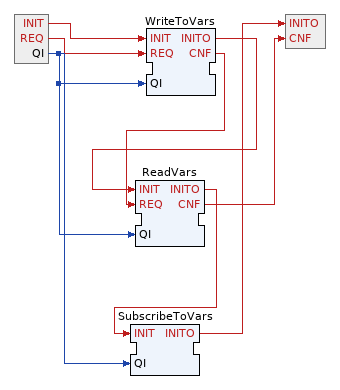
      [picture p47: application OpcUaBothWorking.bytestringNodeIdTestRemote]
      SUBAPPLICATION WriteToVars
        EVENT_INPUT
          INIT;
          REQ;
        END_EVENT
        EVENT_OUTPUT
          INITO;
          CNF;
        END_EVENT
        VAR_INPUT
          QI : BOOL;
        END_VAR
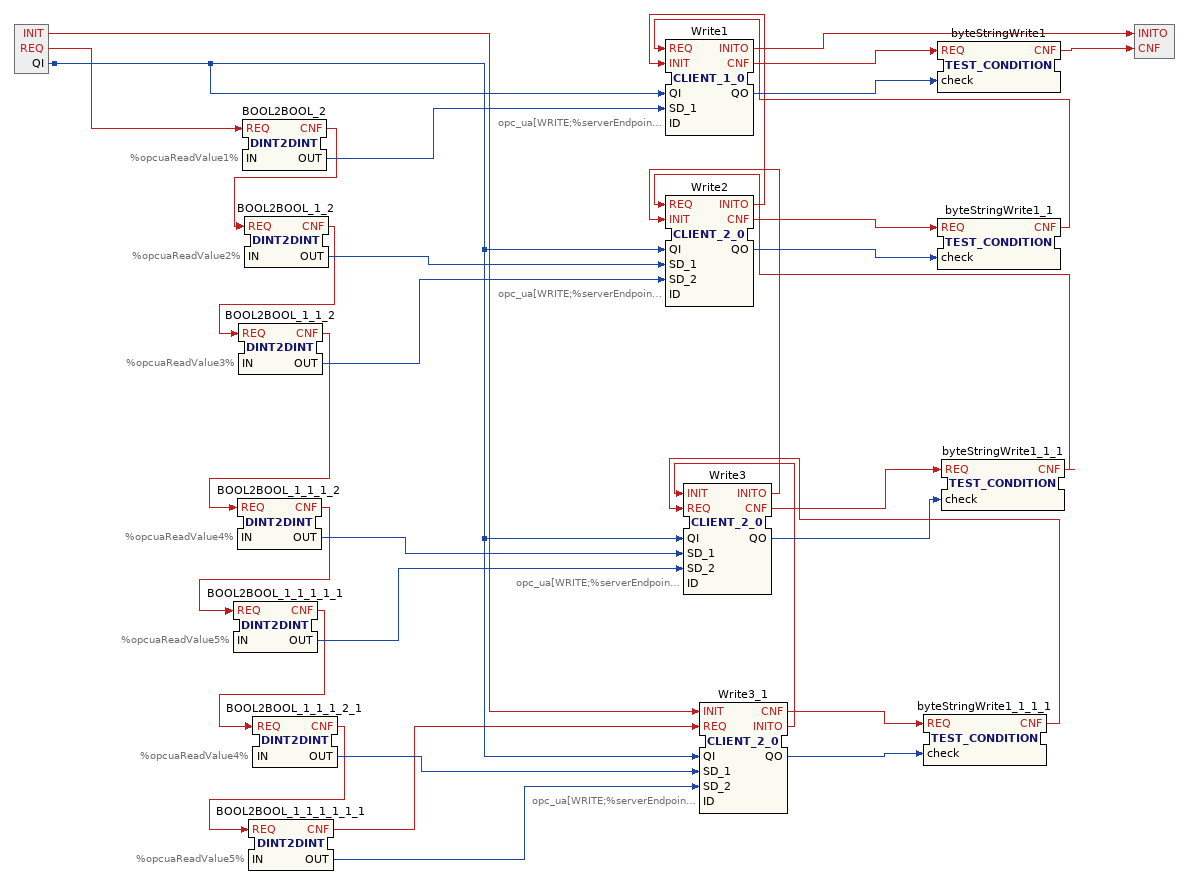
        FBS
          BOOL2BOOL_1_1_2 : DINT2DINT(IN := %opcuaReadValue3%);
          BOOL2BOOL_1_1_1_1_1 : DINT2DINT(IN := %opcuaReadValue5%);
          BOOL2BOOL_1_1_1_2 : DINT2DINT(IN := %opcuaReadValue4%);
          BOOL2BOOL_2 : DINT2DINT(IN := %opcuaReadValue1%);
          BOOL2BOOL_1_2 : DINT2DINT(IN := %opcuaReadValue2%);
          BOOL2BOOL_1_1_1_1_1_1 : DINT2DINT(IN := %opcuaReadValue5%);
          BOOL2BOOL_1_1_1_2_1 : DINT2DINT(IN := %opcuaReadValue4%);
          byteStringWrite1 : TEST_CONDITION;
          byteStringWrite1_1 : TEST_CONDITION;
          byteStringWrite1_1_1 : TEST_CONDITION;
          byteStringWrite1_1_1_1 : TEST_CONDITION;
          Write1 : CLIENT_1_0(ID := opc_ua[WRITE;%serverEndpoint%;%opcuaFolderTestWithNodeIdByteString1%]);
          Write2 : CLIENT_2_0(ID := opc_ua[WRITE;%serverEndpoint%;%opcuaFolderTestWithNodeIdByteString2%]);
          Write3_1 : CLIENT_2_0(ID := opc_ua[WRITE;%serverEndpoint%;,1:b=byteStringNodeId3;,1:b=byteStringNodeId4]);
          Write3 : CLIENT_2_0(ID := opc_ua[WRITE;%serverEndpoint%;%opcuaFolderTestWithNodeIdByteString3%]);
        END_FBS
        EVENT_CONNECTIONS
          BOOL2BOOL_1_2.CNF TO BOOL2BOOL_1_1_2.REQ;
          BOOL2BOOL_1_1_2.CNF TO BOOL2BOOL_1_1_1_2.REQ;
          BOOL2BOOL_1_1_1_2.CNF TO BOOL2BOOL_1_1_1_1_1.REQ;
          BOOL2BOOL_2.CNF TO BOOL2BOOL_1_2.REQ;
          REQ TO BOOL2BOOL_2.REQ;
          BOOL2BOOL_1_1_1_2_1.CNF TO BOOL2BOOL_1_1_1_1_1_1.REQ;
          BOOL2BOOL_1_1_1_1_1.CNF TO BOOL2BOOL_1_1_1_2_1.REQ;
          byteStringWrite1.CNF TO CNF;
          byteStringWrite1_1.CNF TO Write1.REQ;
          Write1.INITO TO INITO;
          Write1.CNF TO byteStringWrite1.REQ;
          byteStringWrite1_1_1.CNF TO Write2.REQ;
          Write2.INITO TO Write1.INIT;
          Write2.CNF TO byteStringWrite1_1.REQ;
          INIT TO Write3_1.INIT;
          BOOL2BOOL_1_1_1_1_1_1.CNF TO Write3_1.REQ;
          Write3_1.CNF TO byteStringWrite1_1_1_1.REQ;
          Write3_1.INITO TO Write3.INIT;
          byteStringWrite1_1_1_1.CNF TO Write3.REQ;
          Write3.INITO TO Write2.INIT;
          Write3.CNF TO byteStringWrite1_1_1.REQ;
        END_CONNECTIONS
        DATA_CONNECTIONS
          QI TO Write1.QI;
          BOOL2BOOL_2.OUT TO Write1.SD_1;
          Write1.QO TO byteStringWrite1.check;
          QI TO Write2.QI;
          BOOL2BOOL_1_2.OUT TO Write2.SD_1;
          BOOL2BOOL_1_1_2.OUT TO Write2.SD_2;
          Write2.QO TO byteStringWrite1_1.check;
          QI TO Write3_1.QI;
          BOOL2BOOL_1_1_1_2_1.OUT TO Write3_1.SD_1;
          BOOL2BOOL_1_1_1_1_1_1.OUT TO Write3_1.SD_2;
          Write3_1.QO TO byteStringWrite1_1_1_1.check;
          QI TO Write3.QI;
          BOOL2BOOL_1_1_1_2.OUT TO Write3.SD_1;
          BOOL2BOOL_1_1_1_1_1.OUT TO Write3.SD_2;
          Write3.QO TO byteStringWrite1_1_1.check;
        END_CONNECTIONS
      END_SUBAPPLICATION
      SUBAPPLICATION ReadVars
        EVENT_INPUT
          INIT;
          REQ;
        END_EVENT
        EVENT_OUTPUT
          INITO;
          CNF;
        END_EVENT
        VAR_INPUT
          QI : BOOL;
        END_VAR
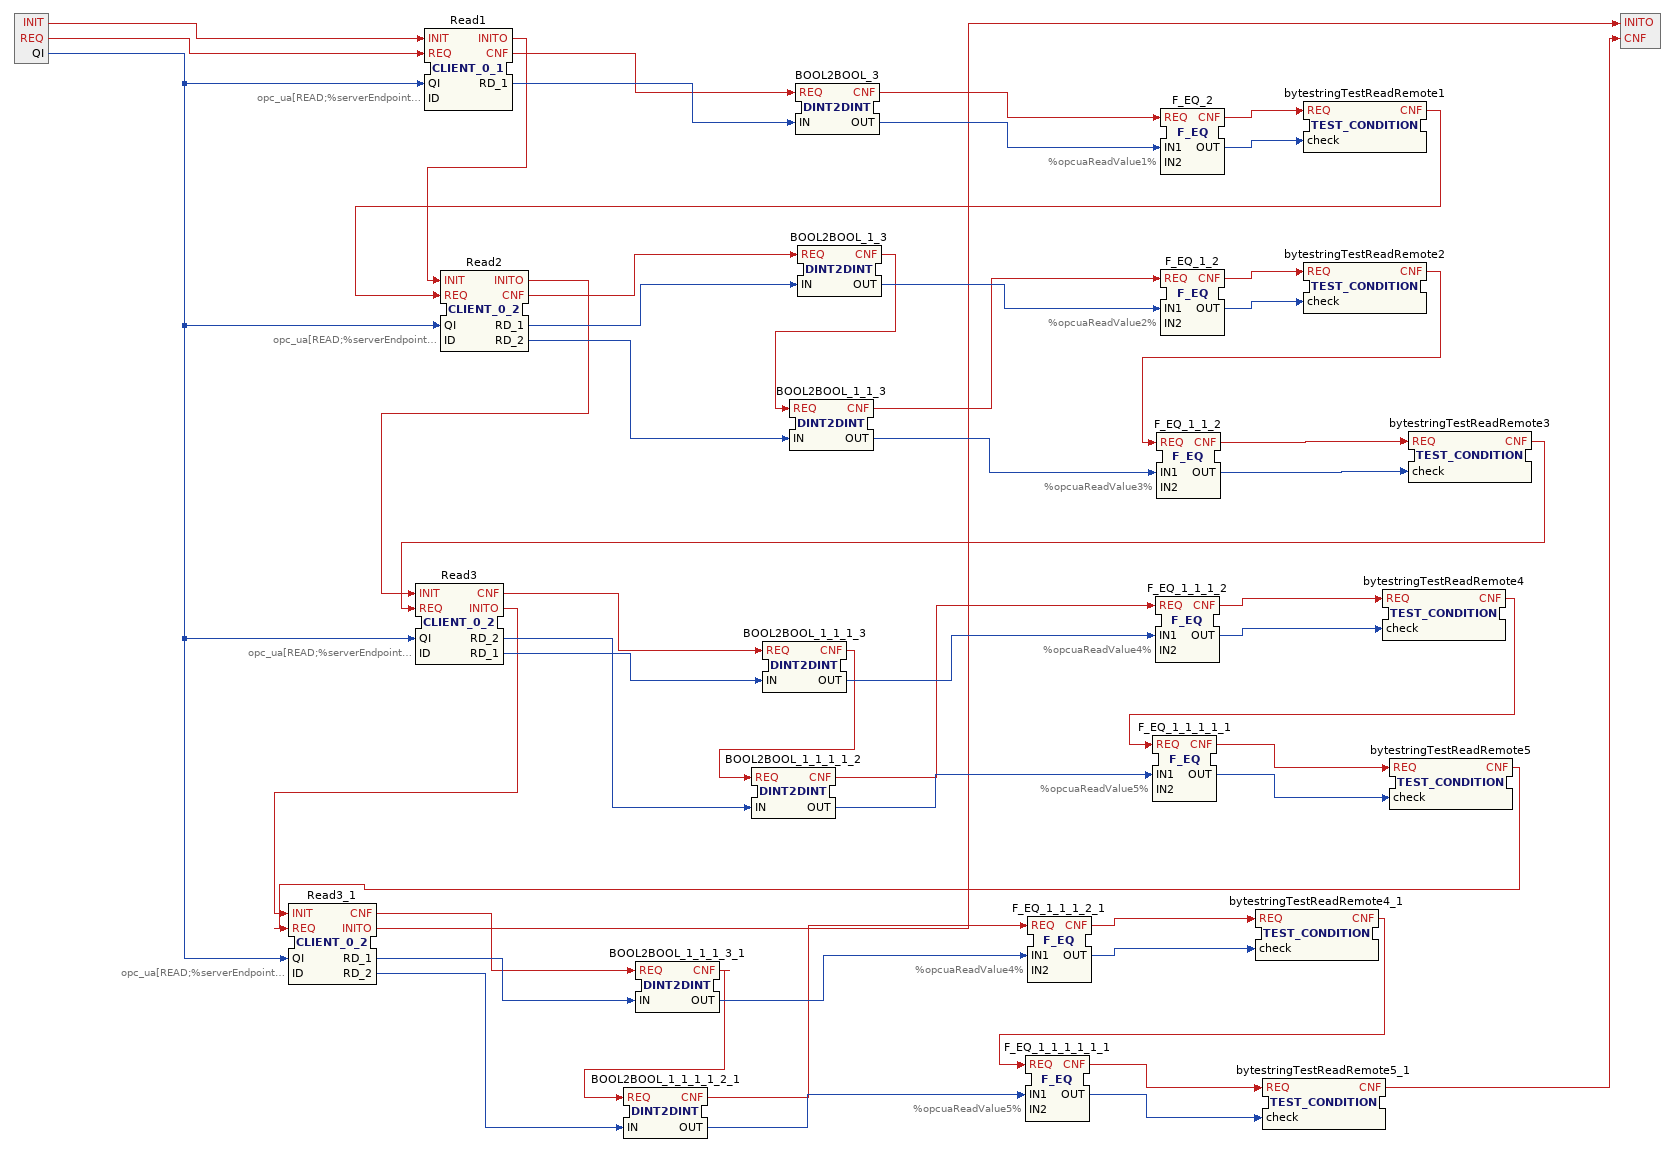
        FBS
          Read1 : CLIENT_0_1(ID := opc_ua[READ;%serverEndpoint%;%opcuaFolderTestWithNodeIdByteString1%]);
          Read2 : CLIENT_0_2(ID := opc_ua[READ;%serverEndpoint%;%opcuaFolderTestWithNodeIdByteString2%]);
          F_EQ_1_1_1_2 : F_EQ(IN2 := %opcuaReadValue4%);
          bytestringTestReadRemote4 : TEST_CONDITION;
          BOOL2BOOL_1_3 : DINT2DINT;
          F_EQ_1_1_1_1_1 : F_EQ(IN2 := %opcuaReadValue5%);
          bytestringTestReadRemote3 : TEST_CONDITION;
          BOOL2BOOL_1_1_3 : DINT2DINT;
          BOOL2BOOL_1_1_1_1_2 : DINT2DINT;
          BOOL2BOOL_1_1_1_3 : DINT2DINT;
          bytestringTestReadRemote2 : TEST_CONDITION;
          F_EQ_1_1_2 : F_EQ(IN2 := %opcuaReadValue3%);
          F_EQ_2 : F_EQ(IN2 := %opcuaReadValue1%);
          F_EQ_1_2 : F_EQ(IN2 := %opcuaReadValue2%);
          Read3 : CLIENT_0_2(ID := opc_ua[READ;%serverEndpoint%;%opcuaFolderTestWithNodeIdByteString3%]);
          bytestringTestReadRemote5 : TEST_CONDITION;
          bytestringTestReadRemote1 : TEST_CONDITION;
          BOOL2BOOL_3 : DINT2DINT;
          BOOL2BOOL_1_1_1_3_1 : DINT2DINT;
          Read3_1 : CLIENT_0_2(ID := opc_ua[READ;%serverEndpoint%;,1:b=byteStringNodeId3;,1:b=byteStringNodeId4]);
          bytestringTestReadRemote4_1 : TEST_CONDITION;
          F_EQ_1_1_1_2_1 : F_EQ(IN2 := %opcuaReadValue4%);
          BOOL2BOOL_1_1_1_1_2_1 : DINT2DINT;
          bytestringTestReadRemote5_1 : TEST_CONDITION;
          F_EQ_1_1_1_1_1_1 : F_EQ(IN2 := %opcuaReadValue5%);
        END_FBS
        EVENT_CONNECTIONS
          Read1.INITO TO Read2.INIT;
          Read1.CNF TO BOOL2BOOL_3.REQ;
          bytestringTestReadRemote1.CNF TO Read2.REQ;
          Read2.INITO TO Read3.INIT;
          Read2.CNF TO BOOL2BOOL_1_3.REQ;
          BOOL2BOOL_1_1_1_1_2.CNF TO F_EQ_1_1_1_2.REQ;
          F_EQ_1_1_1_2.CNF TO bytestringTestReadRemote4.REQ;
          bytestringTestReadRemote4.CNF TO F_EQ_1_1_1_1_1.REQ;
          BOOL2BOOL_1_3.CNF TO BOOL2BOOL_1_1_3.REQ;
          F_EQ_1_1_1_1_1.CNF TO bytestringTestReadRemote5.REQ;
          F_EQ_1_1_2.CNF TO bytestringTestReadRemote3.REQ;
          bytestringTestReadRemote3.CNF TO Read3.REQ;
          BOOL2BOOL_1_1_3.CNF TO F_EQ_1_2.REQ;
          BOOL2BOOL_1_1_1_3.CNF TO BOOL2BOOL_1_1_1_1_2.REQ;
          Read3.CNF TO BOOL2BOOL_1_1_1_3.REQ;
          F_EQ_1_2.CNF TO bytestringTestReadRemote2.REQ;
          bytestringTestReadRemote2.CNF TO F_EQ_1_1_2.REQ;
          BOOL2BOOL_3.CNF TO F_EQ_2.REQ;
          F_EQ_2.CNF TO bytestringTestReadRemote1.REQ;
          INIT TO Read1.INIT;
          REQ TO Read1.REQ;
          bytestringTestReadRemote4_1.CNF TO F_EQ_1_1_1_1_1_1.REQ;
          BOOL2BOOL_1_1_1_1_2_1.CNF TO F_EQ_1_1_1_2_1.REQ;
          F_EQ_1_1_1_1_1_1.CNF TO bytestringTestReadRemote5_1.REQ;
          F_EQ_1_1_1_2_1.CNF TO bytestringTestReadRemote4_1.REQ;
          BOOL2BOOL_1_1_1_3_1.CNF TO BOOL2BOOL_1_1_1_1_2_1.REQ;
          Read3_1.CNF TO BOOL2BOOL_1_1_1_3_1.REQ;
          Read3_1.INITO TO INITO;
          Read3.INITO TO Read3_1.INIT;
          bytestringTestReadRemote5_1.CNF TO CNF;
          bytestringTestReadRemote5.CNF TO Read3_1.REQ;
        END_CONNECTIONS
        DATA_CONNECTIONS
          Read1.RD_1 TO BOOL2BOOL_3.IN;
          Read2.RD_1 TO BOOL2BOOL_1_3.IN;
          Read2.RD_2 TO BOOL2BOOL_1_1_3.IN;
          BOOL2BOOL_1_1_1_3.OUT TO F_EQ_1_1_1_2.IN1;
          F_EQ_1_1_1_2.OUT TO bytestringTestReadRemote4.check;
          BOOL2BOOL_1_3.OUT TO F_EQ_1_2.IN1;
          BOOL2BOOL_1_1_1_1_2.OUT TO F_EQ_1_1_1_1_1.IN1;
          F_EQ_1_1_1_1_1.OUT TO bytestringTestReadRemote5.check;
          F_EQ_1_1_2.OUT TO bytestringTestReadRemote3.check;
          BOOL2BOOL_1_1_3.OUT TO F_EQ_1_1_2.IN1;
          Read3.RD_2 TO BOOL2BOOL_1_1_1_1_2.IN;
          Read3.RD_1 TO BOOL2BOOL_1_1_1_3.IN;
          F_EQ_1_2.OUT TO bytestringTestReadRemote2.check;
          BOOL2BOOL_3.OUT TO F_EQ_2.IN1;
          F_EQ_2.OUT TO bytestringTestReadRemote1.check;
          QI TO Read1.QI;
          QI TO Read2.QI;
          QI TO Read3.QI;
          BOOL2BOOL_1_1_1_1_2_1.OUT TO F_EQ_1_1_1_1_1_1.IN1;
          BOOL2BOOL_1_1_1_3_1.OUT TO F_EQ_1_1_1_2_1.IN1;
          F_EQ_1_1_1_2_1.OUT TO bytestringTestReadRemote4_1.check;
          Read3_1.RD_1 TO BOOL2BOOL_1_1_1_3_1.IN;
          F_EQ_1_1_1_1_1_1.OUT TO bytestringTestReadRemote5_1.check;
          Read3_1.RD_2 TO BOOL2BOOL_1_1_1_1_2_1.IN;
          QI TO Read3_1.QI;
        END_CONNECTIONS
      END_SUBAPPLICATION
      SUBAPPLICATION SubscribeToVars
        EVENT_INPUT
          INIT;
        END_EVENT
        EVENT_OUTPUT
          INITO;
        END_EVENT
        VAR_INPUT
          QI : BOOL;
        END_VAR
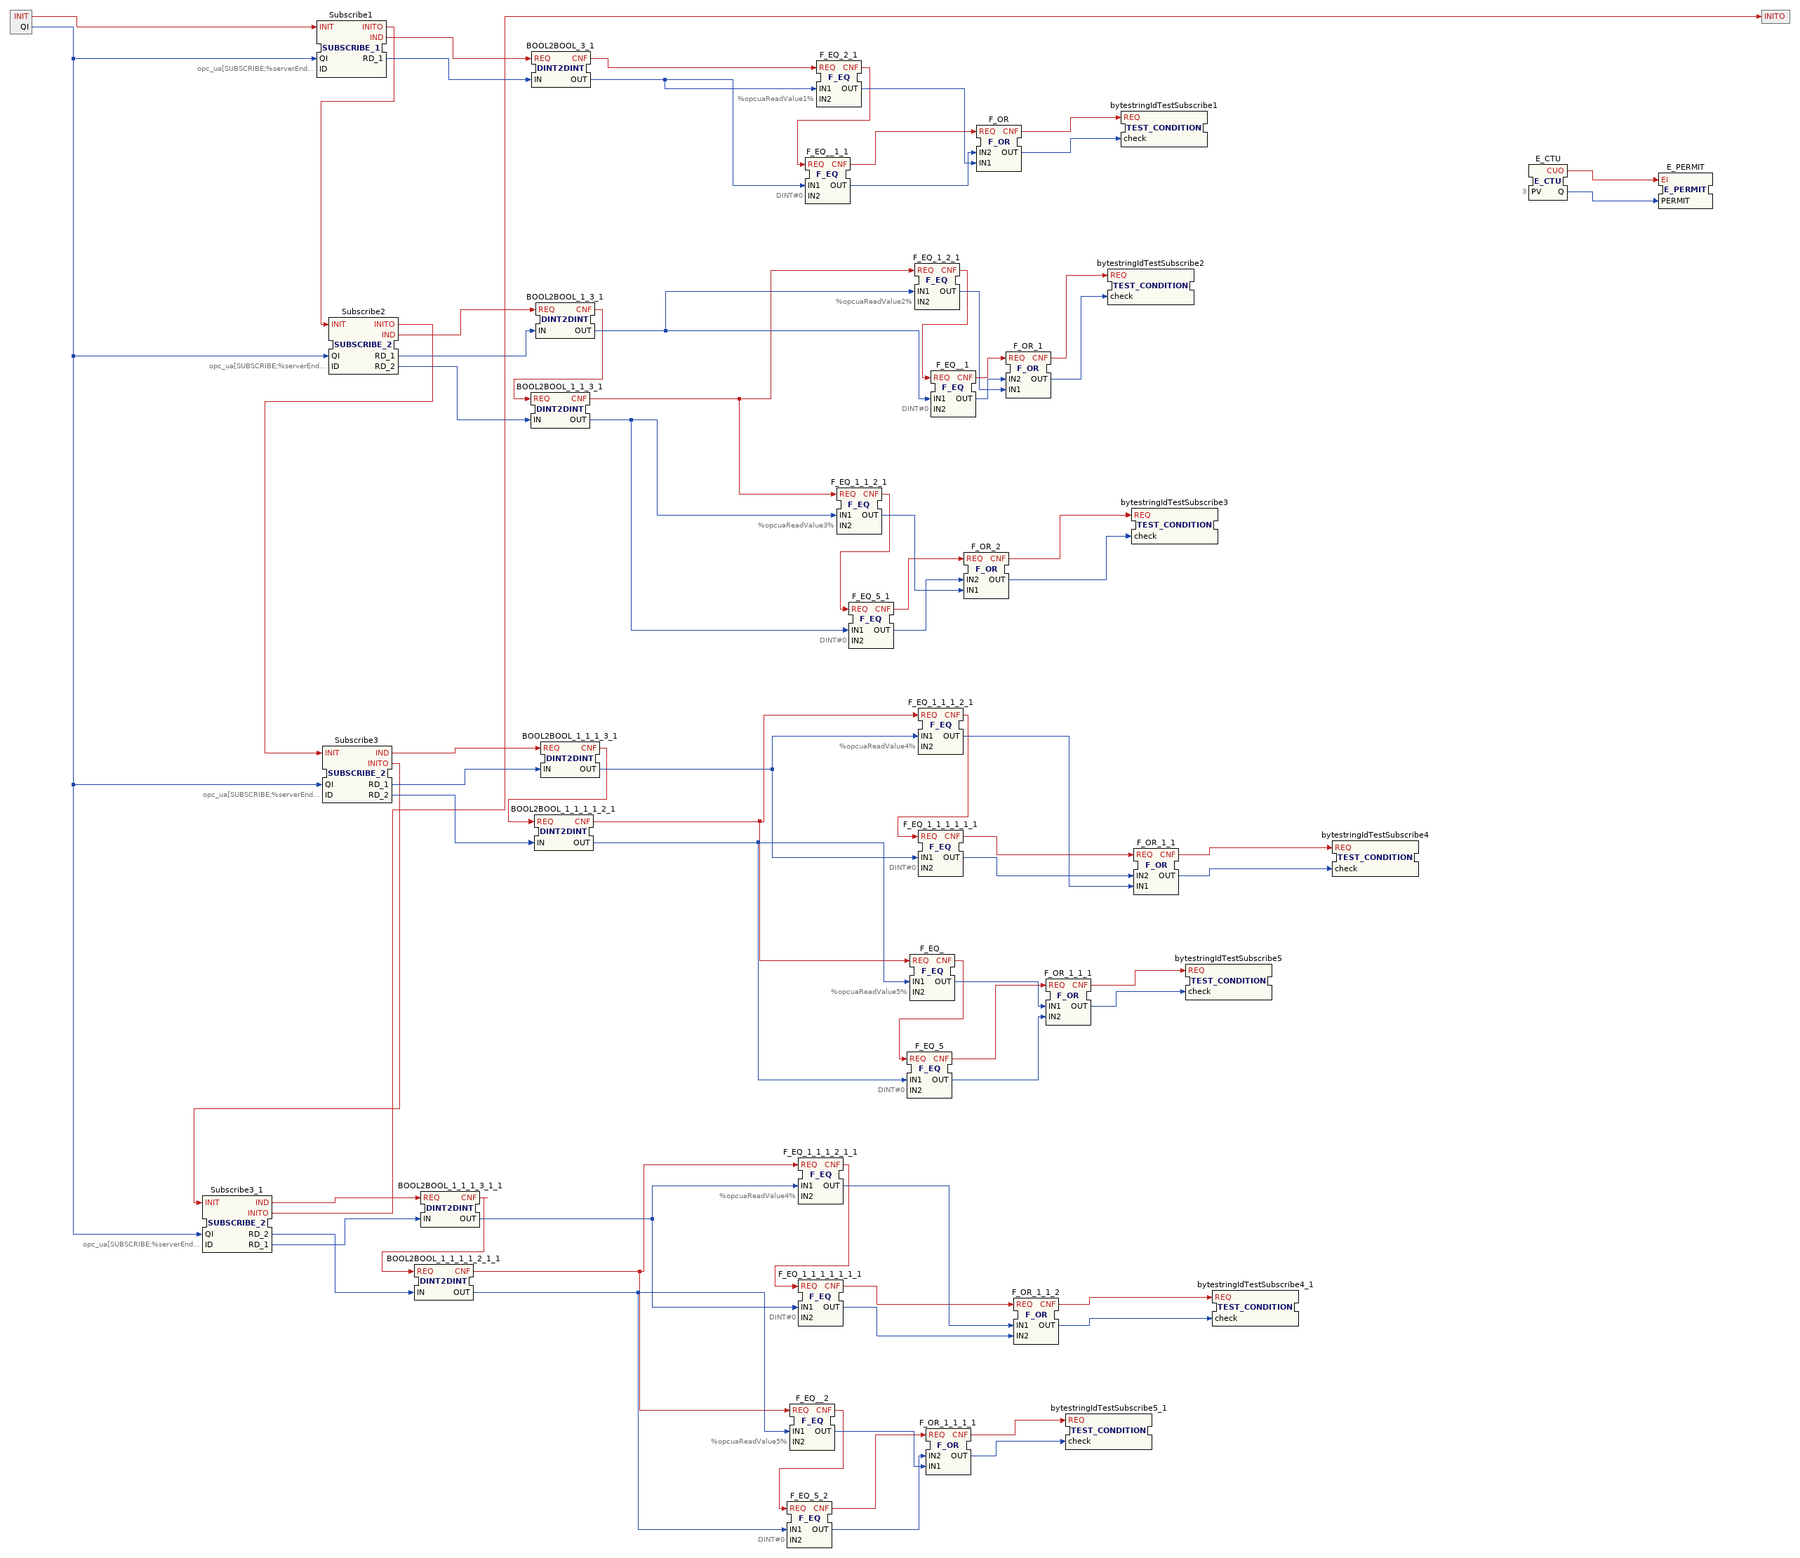
        FBS
          F_EQ_2_1 : F_EQ(IN2 := %opcuaReadValue1%);
          bytestringIdTestSubscribe4 : TEST_CONDITION;
          Subscribe3 : SUBSCRIBE_2(ID := opc_ua[SUBSCRIBE;%serverEndpoint%;%opcuaFolderTestWithNodeIdByteString3%]);
          F_EQ_1_1_1_2_1 : F_EQ(IN2 := %opcuaReadValue4%);
          bytestringIdTestSubscribe3 : TEST_CONDITION;
          F_EQ_1_1_1_1_1_1 : F_EQ(IN2 := DINT#0);
          F_EQ_1_1_2_1 : F_EQ(IN2 := %opcuaReadValue3%);
          bytestringIdTestSubscribe1 : TEST_CONDITION;
          bytestringIdTestSubscribe2 : TEST_CONDITION;
          Subscribe1 : SUBSCRIBE_1(ID := opc_ua[SUBSCRIBE;%serverEndpoint%;%opcuaFolderTestWithNodeIdByteString1%]);
          Subscribe2 : SUBSCRIBE_2(ID := opc_ua[SUBSCRIBE;%serverEndpoint%;%opcuaFolderTestWithNodeIdByteString2%]);
          BOOL2BOOL_1_1_3_1 : DINT2DINT;
          F_EQ_1_2_1 : F_EQ(IN2 := %opcuaReadValue2%);
          BOOL2BOOL_3_1 : DINT2DINT;
          BOOL2BOOL_1_1_1_3_1 : DINT2DINT;
          BOOL2BOOL_1_1_1_1_2_1 : DINT2DINT;
          BOOL2BOOL_1_3_1 : DINT2DINT;
          E_CTU : E_CTU(PV := 3);
          E_PERMIT : E_PERMIT;
          F_EQ_ : F_EQ(IN2 := %opcuaReadValue5%);
          bytestringIdTestSubscribe5 : TEST_CONDITION;
          F_EQ_5 : F_EQ(IN2 := DINT#0);
          F_EQ_5_1 : F_EQ(IN2 := DINT#0);
          F_EQ__1 : F_EQ(IN2 := DINT#0);
          F_EQ__1_1 : F_EQ(IN2 := DINT#0);
          F_OR : F_OR;
          F_OR_1 : F_OR;
          F_OR_2 : F_OR;
          F_OR_1_1 : F_OR;
          F_OR_1_1_1 : F_OR;
          F_EQ_5_2 : F_EQ(IN2 := DINT#0);
          F_EQ_1_1_1_1_1_1_1 : F_EQ(IN2 := DINT#0);
          Subscribe3_1 : SUBSCRIBE_2(ID := opc_ua[SUBSCRIBE;%serverEndpoint%;,1:b=byteStringNodeId3;,1:b=byteStringNodeId4]);
          F_OR_1_1_1_1 : F_OR;
          F_OR_1_1_2 : F_OR;
          BOOL2BOOL_1_1_1_3_1_1 : DINT2DINT;
          F_EQ__2 : F_EQ(IN2 := %opcuaReadValue5%);
          BOOL2BOOL_1_1_1_1_2_1_1 : DINT2DINT;
          bytestringIdTestSubscribe5_1 : TEST_CONDITION;
          bytestringIdTestSubscribe4_1 : TEST_CONDITION;
          F_EQ_1_1_1_2_1_1 : F_EQ(IN2 := %opcuaReadValue4%);
        END_FBS
        EVENT_CONNECTIONS
          Subscribe2.INITO TO Subscribe3.INIT;
          Subscribe3.IND TO BOOL2BOOL_1_1_1_3_1.REQ;
          Subscribe1.INITO TO Subscribe2.INIT;
          Subscribe1.IND TO BOOL2BOOL_3_1.REQ;
          Subscribe2.IND TO BOOL2BOOL_1_3_1.REQ;
          BOOL2BOOL_1_3_1.CNF TO BOOL2BOOL_1_1_3_1.REQ;
          BOOL2BOOL_1_1_1_3_1.CNF TO BOOL2BOOL_1_1_1_1_2_1.REQ;
          INIT TO Subscribe1.INIT;
          E_CTU.CUO TO E_PERMIT.EI;
          F_EQ__1_1.CNF TO F_OR.REQ;
          BOOL2BOOL_3_1.CNF TO F_EQ_2_1.REQ;
          F_EQ_2_1.CNF TO F_EQ__1_1.REQ;
          F_OR.CNF TO bytestringIdTestSubscribe1.REQ;
          F_OR_2.CNF TO bytestringIdTestSubscribe3.REQ;
          F_OR_1.CNF TO bytestringIdTestSubscribe2.REQ;
          F_EQ__1.CNF TO F_OR_1.REQ;
          F_EQ_1_2_1.CNF TO F_EQ__1.REQ;
          BOOL2BOOL_1_1_3_1.CNF TO F_EQ_1_2_1.REQ;
          BOOL2BOOL_1_1_3_1.CNF TO F_EQ_1_1_2_1.REQ;
          F_EQ_1_1_2_1.CNF TO F_EQ_5_1.REQ;
          F_EQ_5_1.CNF TO F_OR_2.REQ;
          F_OR_1_1.CNF TO bytestringIdTestSubscribe4.REQ;
          F_EQ_1_1_1_1_1_1.CNF TO F_OR_1_1.REQ;
          F_EQ_1_1_1_2_1.CNF TO F_EQ_1_1_1_1_1_1.REQ;
          BOOL2BOOL_1_1_1_1_2_1.CNF TO F_EQ_1_1_1_2_1.REQ;
          F_OR_1_1_1.CNF TO bytestringIdTestSubscribe5.REQ;
          BOOL2BOOL_1_1_1_1_2_1.CNF TO F_EQ_.REQ;
          F_EQ_.CNF TO F_EQ_5.REQ;
          F_EQ_5.CNF TO F_OR_1_1_1.REQ;
          BOOL2BOOL_1_1_1_3_1_1.CNF TO BOOL2BOOL_1_1_1_1_2_1_1.REQ;
          BOOL2BOOL_1_1_1_1_2_1_1.CNF TO F_EQ_1_1_1_2_1_1.REQ;
          F_EQ_1_1_1_1_1_1_1.CNF TO F_OR_1_1_2.REQ;
          BOOL2BOOL_1_1_1_1_2_1_1.CNF TO F_EQ__2.REQ;
          F_EQ_5_2.CNF TO F_OR_1_1_1_1.REQ;
          F_OR_1_1_1_1.CNF TO bytestringIdTestSubscribe5_1.REQ;
          F_EQ_1_1_1_2_1_1.CNF TO F_EQ_1_1_1_1_1_1_1.REQ;
          F_EQ__2.CNF TO F_EQ_5_2.REQ;
          Subscribe3_1.IND TO BOOL2BOOL_1_1_1_3_1_1.REQ;
          F_OR_1_1_2.CNF TO bytestringIdTestSubscribe4_1.REQ;
          Subscribe3_1.INITO TO INITO;
          Subscribe3.INITO TO Subscribe3_1.INIT;
        END_CONNECTIONS
        DATA_CONNECTIONS
          BOOL2BOOL_3_1.OUT TO F_EQ_2_1.IN1;
          Subscribe3.RD_1 TO BOOL2BOOL_1_1_1_3_1.IN;
          Subscribe3.RD_2 TO BOOL2BOOL_1_1_1_1_2_1.IN;
          BOOL2BOOL_1_1_3_1.OUT TO F_EQ_1_1_2_1.IN1;
          Subscribe1.RD_1 TO BOOL2BOOL_3_1.IN;
          Subscribe2.RD_1 TO BOOL2BOOL_1_3_1.IN;
          Subscribe2.RD_2 TO BOOL2BOOL_1_1_3_1.IN;
          BOOL2BOOL_1_3_1.OUT TO F_EQ_1_2_1.IN1;
          QI TO Subscribe3.QI;
          QI TO Subscribe1.QI;
          QI TO Subscribe2.QI;
          E_CTU.Q TO E_PERMIT.PERMIT;
          BOOL2BOOL_1_1_1_1_2_1.OUT TO F_EQ_5.IN1;
          BOOL2BOOL_1_3_1.OUT TO F_EQ__1.IN1;
          BOOL2BOOL_1_1_3_1.OUT TO F_EQ_5_1.IN1;
          BOOL2BOOL_3_1.OUT TO F_EQ__1_1.IN1;
          BOOL2BOOL_1_1_1_3_1.OUT TO F_EQ_1_1_1_2_1.IN1;
          F_EQ__1_1.OUT TO F_OR.IN2;
          F_EQ_2_1.OUT TO F_OR.IN1;
          F_OR.OUT TO bytestringIdTestSubscribe1.check;
          F_EQ_5_1.OUT TO F_OR_2.IN2;
          F_EQ__1.OUT TO F_OR_1.IN2;
          F_EQ_1_2_1.OUT TO F_OR_1.IN1;
          F_OR_1.OUT TO bytestringIdTestSubscribe2.check;
          F_OR_2.OUT TO bytestringIdTestSubscribe3.check;
          F_OR_1_1.OUT TO bytestringIdTestSubscribe4.check;
          F_EQ_1_1_1_1_1_1.OUT TO F_OR_1_1.IN2;
          F_EQ_1_1_1_2_1.OUT TO F_OR_1_1.IN1;
          F_OR_1_1_1.OUT TO bytestringIdTestSubscribe5.check;
          F_EQ_.OUT TO F_OR_1_1_1.IN1;
          F_EQ_5.OUT TO F_OR_1_1_1.IN2;
          BOOL2BOOL_1_1_1_1_2_1.OUT TO F_EQ_.IN1;
          F_EQ_1_1_2_1.OUT TO F_OR_2.IN1;
          BOOL2BOOL_1_1_1_3_1.OUT TO F_EQ_1_1_1_1_1_1.IN1;
          BOOL2BOOL_1_1_1_3_1_1.OUT TO F_EQ_1_1_1_2_1_1.IN1;
          BOOL2BOOL_1_1_1_1_2_1_1.OUT TO F_EQ_5_2.IN1;
          F_EQ_1_1_1_2_1_1.OUT TO F_OR_1_1_2.IN1;
          Subscribe3_1.RD_2 TO BOOL2BOOL_1_1_1_1_2_1_1.IN;
          F_OR_1_1_1_1.OUT TO bytestringIdTestSubscribe5_1.check;
          F_EQ_5_2.OUT TO F_OR_1_1_1_1.IN2;
          Subscribe3_1.RD_1 TO BOOL2BOOL_1_1_1_3_1_1.IN;
          F_EQ_1_1_1_1_1_1_1.OUT TO F_OR_1_1_2.IN2;
          BOOL2BOOL_1_1_1_3_1_1.OUT TO F_EQ_1_1_1_1_1_1_1.IN1;
          BOOL2BOOL_1_1_1_1_2_1_1.OUT TO F_EQ__2.IN1;
          F_OR_1_1_2.OUT TO bytestringIdTestSubscribe4_1.check;
          F_EQ__2.OUT TO F_OR_1_1_1_1.IN1;
          QI TO Subscribe3_1.QI;
        END_CONNECTIONS
      END_SUBAPPLICATION
      EVENT_CONNECTIONS
        WriteToVars.INITO TO ReadVars.INIT;
        INIT TO WriteToVars.INIT;
        REQ TO WriteToVars.REQ;
        ReadVars.CNF TO CNF;
        SubscribeToVars.INITO TO INITO;
        ReadVars.INITO TO SubscribeToVars.INIT;
        WriteToVars.CNF TO ReadVars.REQ;
      END_CONNECTIONS
      DATA_CONNECTIONS
        QI TO ReadVars.QI;
        QI TO WriteToVars.QI;
        QI TO SubscribeToVars.QI;
      END_CONNECTIONS
    END_SUBAPPLICATION
    SUBAPPLICATION LocaMethods
      EVENT_INPUT
        INIT;
      END_EVENT
      EVENT_OUTPUT
        INITO;
      END_EVENT
      VAR_INPUT
        QI : BOOL;
      END_VAR
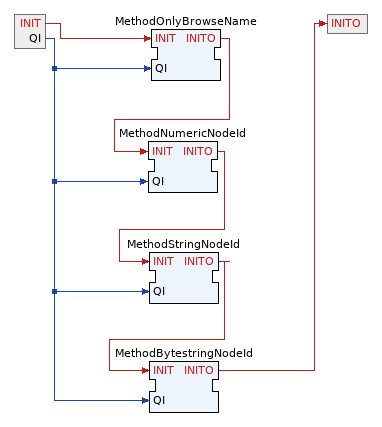
      SUBAPPLICATION MethodOnlyBrowseName
        EVENT_INPUT
          INIT;
        END_EVENT
        EVENT_OUTPUT
          INITO;
        END_EVENT
        VAR_INPUT
          QI : BOOL;
        END_VAR
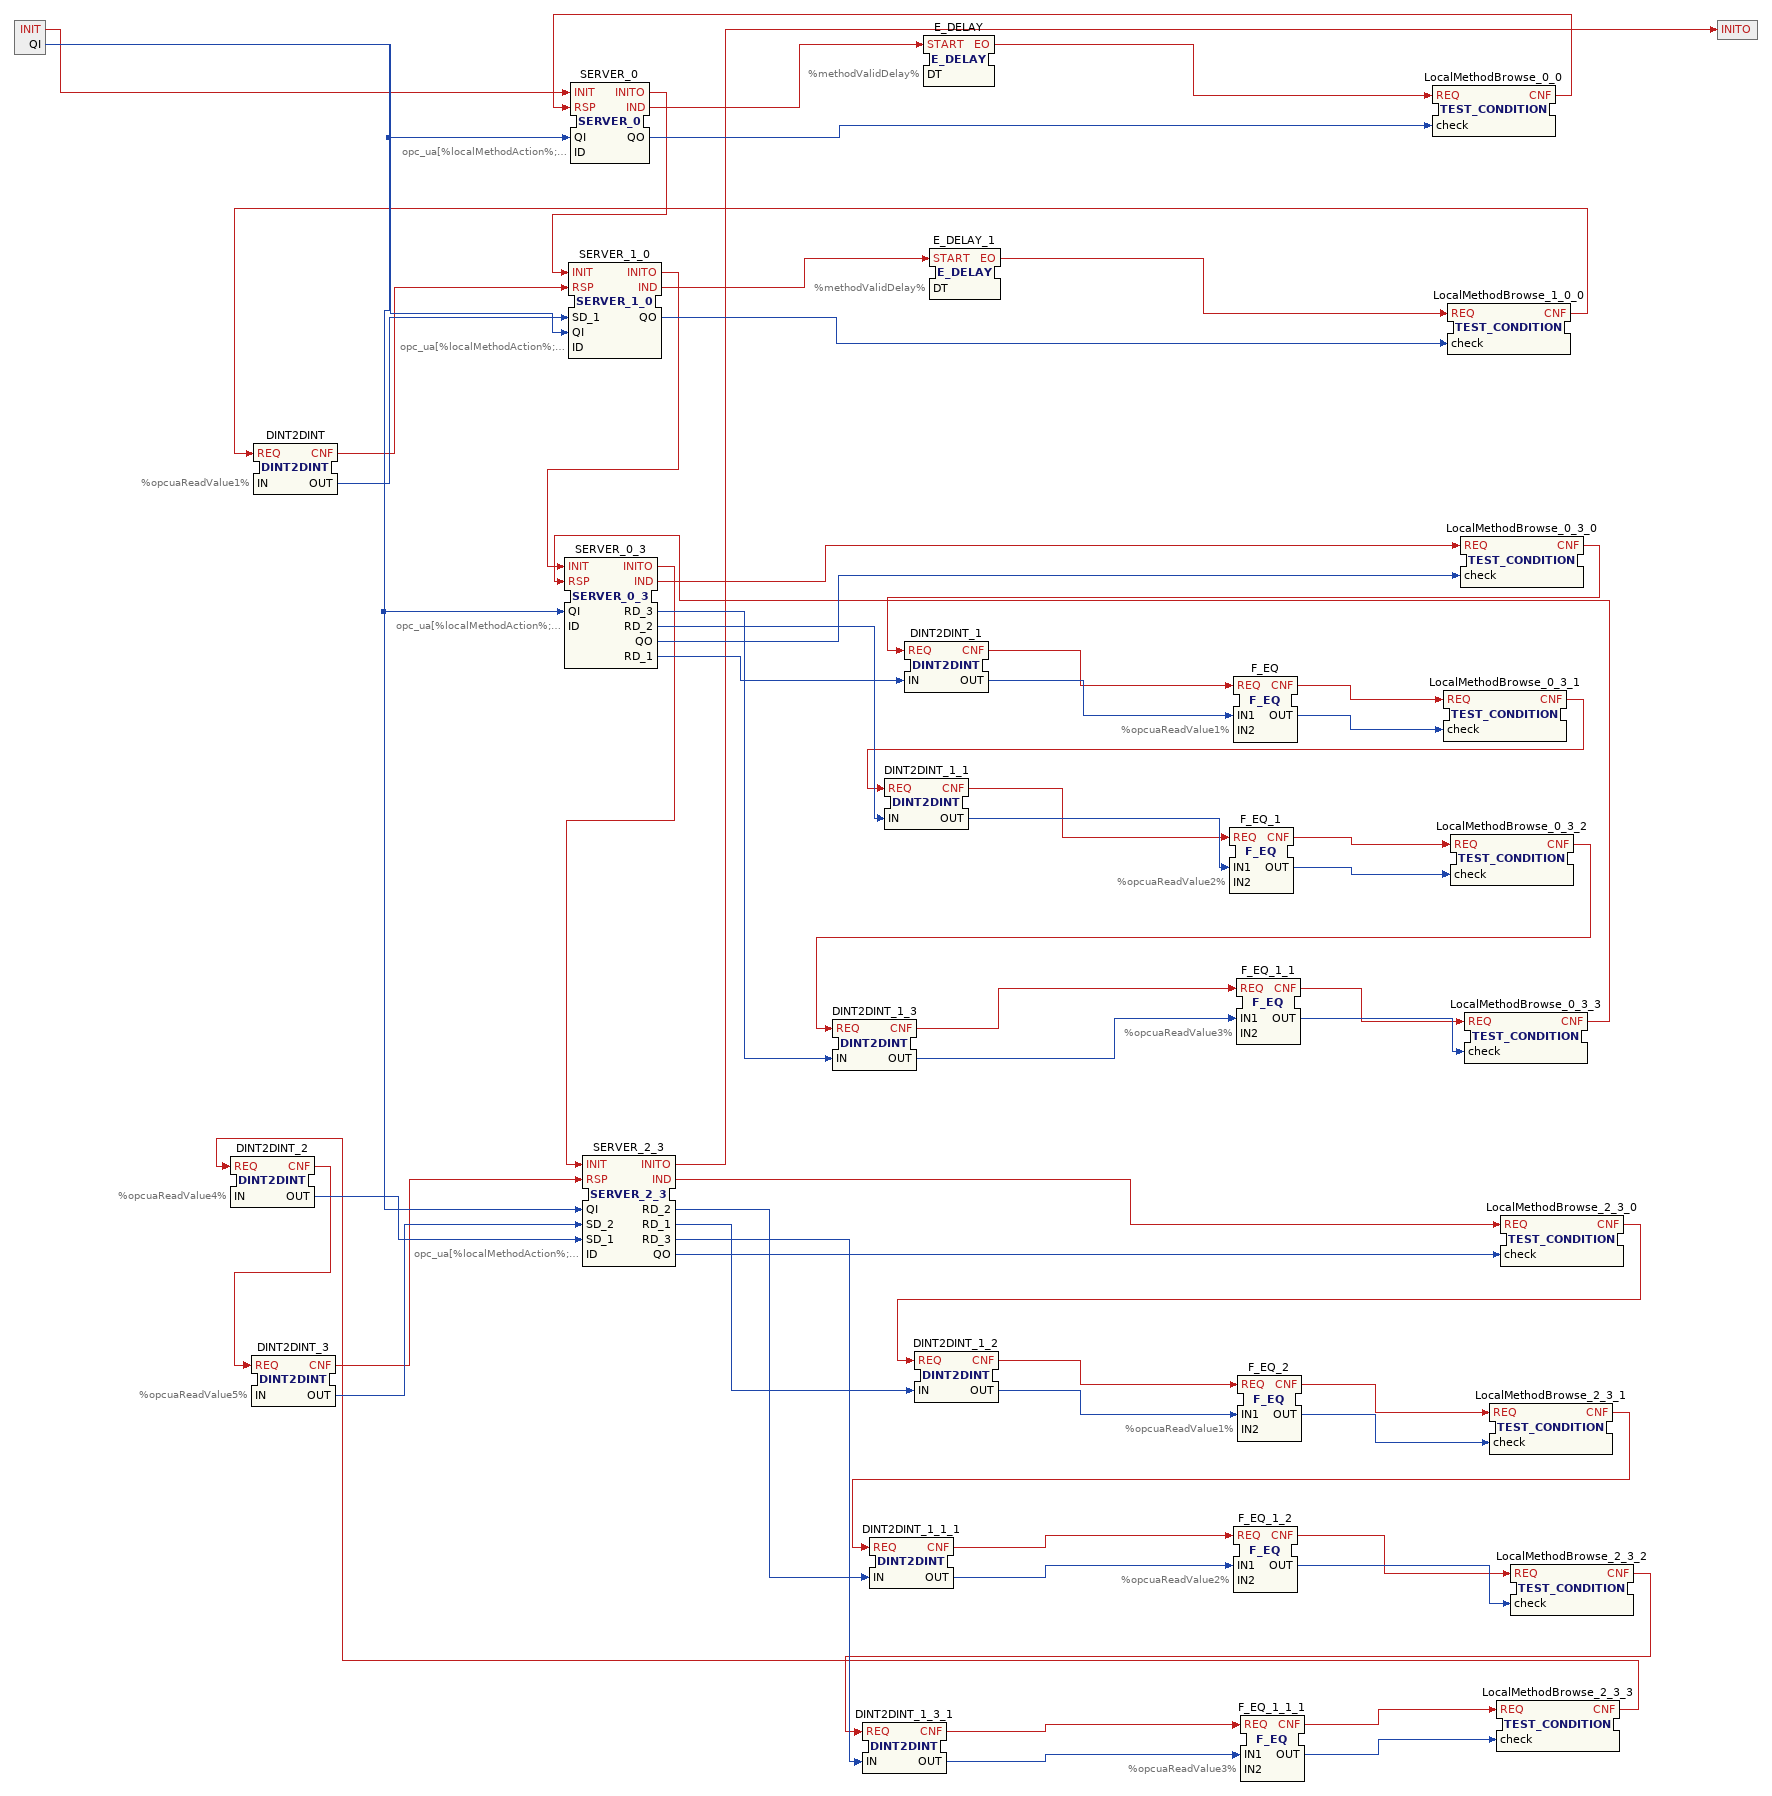
        FBS
          DINT2DINT_1_1_1 : DINT2DINT;
          DINT2DINT_1_2 : DINT2DINT;
          SERVER_0 : SERVER_0(ID := opc_ua[%localMethodAction%;%opcuaMethodCreation1%]);
          DINT2DINT_1_3 : DINT2DINT;
          DINT2DINT_1_1 : DINT2DINT;
          SERVER_0_3 : SERVER_0_3(ID := opc_ua[%localMethodAction%;%opcuaMethodCreation3%]);
          DINT2DINT_1_3_1 : DINT2DINT;
          SERVER_2_3 : SERVER_2_3(ID := opc_ua[%localMethodAction%;%opcuaMethodCreation4%]);
          LocalMethodBrowse_2_3_0 : TEST_CONDITION;
          LocalMethodBrowse_0_3_0 : TEST_CONDITION;
          SERVER_1_0 : SERVER_1_0(ID := opc_ua[%localMethodAction%;%opcuaMethodCreation2%]);
          LocalMethodBrowse_0_0 : TEST_CONDITION;
          LocalMethodBrowse_1_0_0 : TEST_CONDITION;
          DINT2DINT : DINT2DINT(IN := %opcuaReadValue1%);
          DINT2DINT_1 : DINT2DINT;
          DINT2DINT_2 : DINT2DINT(IN := %opcuaReadValue4%);
          DINT2DINT_3 : DINT2DINT(IN := %opcuaReadValue5%);
          LocalMethodBrowse_0_3_1 : TEST_CONDITION;
          LocalMethodBrowse_2_3_2 : TEST_CONDITION;
          LocalMethodBrowse_0_3_2 : TEST_CONDITION;
          LocalMethodBrowse_0_3_3 : TEST_CONDITION;
          LocalMethodBrowse_2_3_3 : TEST_CONDITION;
          F_EQ : F_EQ(IN2 := %opcuaReadValue1%);
          F_EQ_1 : F_EQ(IN2 := %opcuaReadValue2%);
          F_EQ_1_1 : F_EQ(IN2 := %opcuaReadValue3%);
          LocalMethodBrowse_2_3_1 : TEST_CONDITION;
          F_EQ_1_2 : F_EQ(IN2 := %opcuaReadValue2%);
          F_EQ_2 : F_EQ(IN2 := %opcuaReadValue1%);
          F_EQ_1_1_1 : F_EQ(IN2 := %opcuaReadValue3%);
          E_DELAY : E_DELAY(DT := %methodValidDelay%);
          E_DELAY_1 : E_DELAY(DT := %methodValidDelay%);
        END_FBS
        EVENT_CONNECTIONS
          INIT TO SERVER_0.INIT;
          SERVER_0.INITO TO SERVER_1_0.INIT;
          SERVER_1_0.INITO TO SERVER_0_3.INIT;
          SERVER_0_3.INITO TO SERVER_2_3.INIT;
          LocalMethodBrowse_0_0.CNF TO SERVER_0.RSP;
          SERVER_2_3.INITO TO INITO;
          LocalMethodBrowse_1_0_0.CNF TO DINT2DINT.REQ;
          DINT2DINT.CNF TO SERVER_1_0.RSP;
          SERVER_0_3.IND TO LocalMethodBrowse_0_3_0.REQ;
          LocalMethodBrowse_0_3_0.CNF TO DINT2DINT_1.REQ;
          DINT2DINT_1.CNF TO F_EQ.REQ;
          F_EQ.CNF TO LocalMethodBrowse_0_3_1.REQ;
          F_EQ_1.CNF TO LocalMethodBrowse_0_3_2.REQ;
          F_EQ_1_1.CNF TO LocalMethodBrowse_0_3_3.REQ;
          LocalMethodBrowse_0_3_1.CNF TO DINT2DINT_1_1.REQ;
          DINT2DINT_1_1.CNF TO F_EQ_1.REQ;
          LocalMethodBrowse_0_3_2.CNF TO DINT2DINT_1_3.REQ;
          DINT2DINT_1_3.CNF TO F_EQ_1_1.REQ;
          LocalMethodBrowse_0_3_3.CNF TO SERVER_0_3.RSP;
          SERVER_2_3.IND TO LocalMethodBrowse_2_3_0.REQ;
          LocalMethodBrowse_2_3_0.CNF TO DINT2DINT_1_2.REQ;
          DINT2DINT_1_2.CNF TO F_EQ_2.REQ;
          F_EQ_2.CNF TO LocalMethodBrowse_2_3_1.REQ;
          LocalMethodBrowse_2_3_1.CNF TO DINT2DINT_1_1_1.REQ;
          DINT2DINT_1_1_1.CNF TO F_EQ_1_2.REQ;
          F_EQ_1_2.CNF TO LocalMethodBrowse_2_3_2.REQ;
          LocalMethodBrowse_2_3_2.CNF TO DINT2DINT_1_3_1.REQ;
          DINT2DINT_1_3_1.CNF TO F_EQ_1_1_1.REQ;
          F_EQ_1_1_1.CNF TO LocalMethodBrowse_2_3_3.REQ;
          LocalMethodBrowse_2_3_3.CNF TO DINT2DINT_2.REQ;
          DINT2DINT_2.CNF TO DINT2DINT_3.REQ;
          DINT2DINT_3.CNF TO SERVER_2_3.RSP;
          SERVER_0.IND TO E_DELAY.START;
          E_DELAY.EO TO LocalMethodBrowse_0_0.REQ;
          SERVER_1_0.IND TO E_DELAY_1.START;
          E_DELAY_1.EO TO LocalMethodBrowse_1_0_0.REQ;
        END_CONNECTIONS
        DATA_CONNECTIONS
          SERVER_2_3.RD_2 TO DINT2DINT_1_1_1.IN;
          SERVER_2_3.RD_1 TO DINT2DINT_1_2.IN;
          SERVER_0.QO TO LocalMethodBrowse_0_0.check;
          SERVER_0_3.RD_3 TO DINT2DINT_1_3.IN;
          SERVER_0_3.RD_2 TO DINT2DINT_1_1.IN;
          SERVER_0_3.QO TO LocalMethodBrowse_0_3_0.check;
          SERVER_0_3.RD_1 TO DINT2DINT_1.IN;
          SERVER_2_3.RD_3 TO DINT2DINT_1_3_1.IN;
          SERVER_2_3.QO TO LocalMethodBrowse_2_3_0.check;
          DINT2DINT.OUT TO SERVER_1_0.SD_1;
          SERVER_1_0.QO TO LocalMethodBrowse_1_0_0.check;
          QI TO SERVER_0.QI;
          QI TO SERVER_1_0.QI;
          QI TO SERVER_0_3.QI;
          QI TO SERVER_2_3.QI;
          DINT2DINT_3.OUT TO SERVER_2_3.SD_2;
          DINT2DINT_2.OUT TO SERVER_2_3.SD_1;
          F_EQ.OUT TO LocalMethodBrowse_0_3_1.check;
          DINT2DINT_1.OUT TO F_EQ.IN1;
          F_EQ_1_1.OUT TO LocalMethodBrowse_0_3_3.check;
          F_EQ_1.OUT TO LocalMethodBrowse_0_3_2.check;
          DINT2DINT_1_1.OUT TO F_EQ_1.IN1;
          DINT2DINT_1_3.OUT TO F_EQ_1_1.IN1;
          F_EQ_1_2.OUT TO LocalMethodBrowse_2_3_2.check;
          F_EQ_2.OUT TO LocalMethodBrowse_2_3_1.check;
          DINT2DINT_1_2.OUT TO F_EQ_2.IN1;
          DINT2DINT_1_1_1.OUT TO F_EQ_1_2.IN1;
          DINT2DINT_1_3_1.OUT TO F_EQ_1_1_1.IN1;
          F_EQ_1_1_1.OUT TO LocalMethodBrowse_2_3_3.check;
        END_CONNECTIONS
      END_SUBAPPLICATION
      SUBAPPLICATION MethodNumericNodeId
        EVENT_INPUT
          INIT;
        END_EVENT
        EVENT_OUTPUT
          INITO;
        END_EVENT
        VAR_INPUT
          QI : BOOL;
        END_VAR
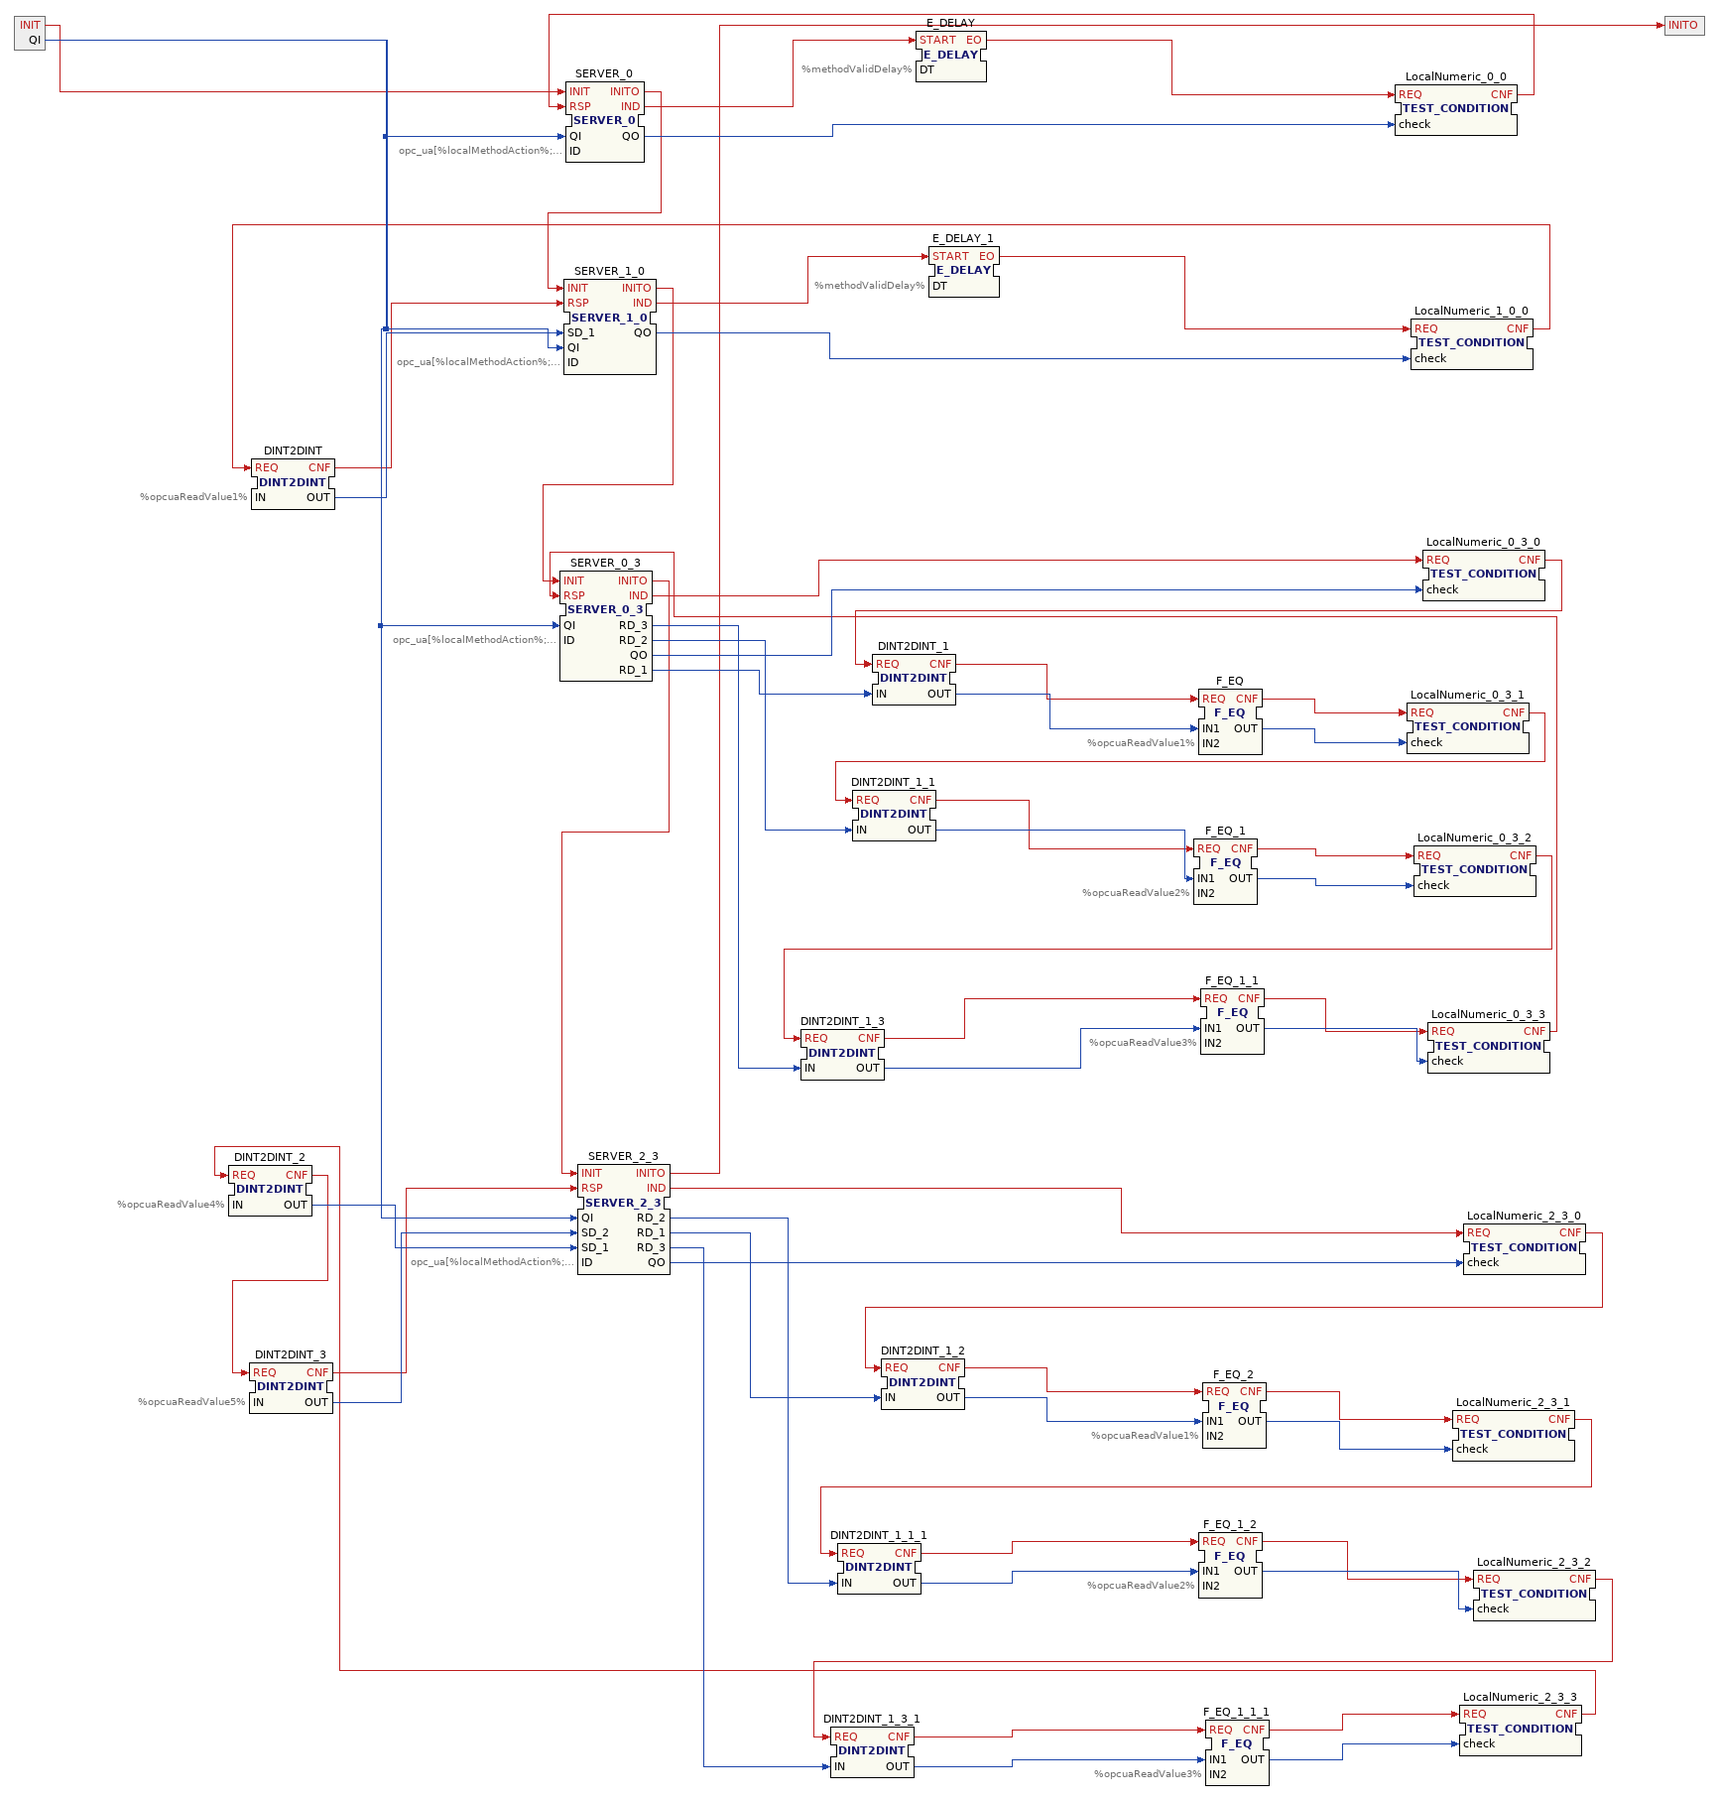
        FBS
          DINT2DINT_1_1_1 : DINT2DINT;
          DINT2DINT_1_2 : DINT2DINT;
          SERVER_0 : SERVER_0(ID := opc_ua[%localMethodAction%;%opcuaMethodCreation5%]);
          DINT2DINT_1_3 : DINT2DINT;
          DINT2DINT_1_1 : DINT2DINT;
          SERVER_0_3 : SERVER_0_3(ID := opc_ua[%localMethodAction%;%opcuaMethodCreation7%]);
          DINT2DINT_1_3_1 : DINT2DINT;
          SERVER_2_3 : SERVER_2_3(ID := opc_ua[%localMethodAction%;%opcuaMethodCreation8%]);
          LocalNumeric_2_3_0 : TEST_CONDITION;
          LocalNumeric_0_3_0 : TEST_CONDITION;
          SERVER_1_0 : SERVER_1_0(ID := opc_ua[%localMethodAction%;%opcuaMethodCreation6%]);
          LocalNumeric_0_0 : TEST_CONDITION;
          LocalNumeric_1_0_0 : TEST_CONDITION;
          DINT2DINT : DINT2DINT(IN := %opcuaReadValue1%);
          DINT2DINT_1 : DINT2DINT;
          DINT2DINT_2 : DINT2DINT(IN := %opcuaReadValue4%);
          DINT2DINT_3 : DINT2DINT(IN := %opcuaReadValue5%);
          LocalNumeric_0_3_1 : TEST_CONDITION;
          LocalNumeric_2_3_2 : TEST_CONDITION;
          LocalNumeric_0_3_2 : TEST_CONDITION;
          LocalNumeric_0_3_3 : TEST_CONDITION;
          LocalNumeric_2_3_3 : TEST_CONDITION;
          F_EQ : F_EQ(IN2 := %opcuaReadValue1%);
          F_EQ_1 : F_EQ(IN2 := %opcuaReadValue2%);
          F_EQ_1_1 : F_EQ(IN2 := %opcuaReadValue3%);
          LocalNumeric_2_3_1 : TEST_CONDITION;
          F_EQ_1_2 : F_EQ(IN2 := %opcuaReadValue2%);
          F_EQ_2 : F_EQ(IN2 := %opcuaReadValue1%);
          F_EQ_1_1_1 : F_EQ(IN2 := %opcuaReadValue3%);
          E_DELAY : E_DELAY(DT := %methodValidDelay%);
          E_DELAY_1 : E_DELAY(DT := %methodValidDelay%);
        END_FBS
        EVENT_CONNECTIONS
          INIT TO SERVER_0.INIT;
          SERVER_0.INITO TO SERVER_1_0.INIT;
          SERVER_1_0.INITO TO SERVER_0_3.INIT;
          SERVER_0_3.INITO TO SERVER_2_3.INIT;
          LocalNumeric_0_0.CNF TO SERVER_0.RSP;
          SERVER_2_3.INITO TO INITO;
          LocalNumeric_1_0_0.CNF TO DINT2DINT.REQ;
          DINT2DINT.CNF TO SERVER_1_0.RSP;
          SERVER_0_3.IND TO LocalNumeric_0_3_0.REQ;
          LocalNumeric_0_3_0.CNF TO DINT2DINT_1.REQ;
          DINT2DINT_1.CNF TO F_EQ.REQ;
          F_EQ.CNF TO LocalNumeric_0_3_1.REQ;
          F_EQ_1.CNF TO LocalNumeric_0_3_2.REQ;
          F_EQ_1_1.CNF TO LocalNumeric_0_3_3.REQ;
          LocalNumeric_0_3_1.CNF TO DINT2DINT_1_1.REQ;
          DINT2DINT_1_1.CNF TO F_EQ_1.REQ;
          LocalNumeric_0_3_2.CNF TO DINT2DINT_1_3.REQ;
          DINT2DINT_1_3.CNF TO F_EQ_1_1.REQ;
          LocalNumeric_0_3_3.CNF TO SERVER_0_3.RSP;
          SERVER_2_3.IND TO LocalNumeric_2_3_0.REQ;
          LocalNumeric_2_3_0.CNF TO DINT2DINT_1_2.REQ;
          DINT2DINT_1_2.CNF TO F_EQ_2.REQ;
          F_EQ_2.CNF TO LocalNumeric_2_3_1.REQ;
          LocalNumeric_2_3_1.CNF TO DINT2DINT_1_1_1.REQ;
          DINT2DINT_1_1_1.CNF TO F_EQ_1_2.REQ;
          F_EQ_1_2.CNF TO LocalNumeric_2_3_2.REQ;
          LocalNumeric_2_3_2.CNF TO DINT2DINT_1_3_1.REQ;
          DINT2DINT_1_3_1.CNF TO F_EQ_1_1_1.REQ;
          F_EQ_1_1_1.CNF TO LocalNumeric_2_3_3.REQ;
          LocalNumeric_2_3_3.CNF TO DINT2DINT_2.REQ;
          DINT2DINT_2.CNF TO DINT2DINT_3.REQ;
          DINT2DINT_3.CNF TO SERVER_2_3.RSP;
          SERVER_0.IND TO E_DELAY.START;
          E_DELAY.EO TO LocalNumeric_0_0.REQ;
          SERVER_1_0.IND TO E_DELAY_1.START;
          E_DELAY_1.EO TO LocalNumeric_1_0_0.REQ;
        END_CONNECTIONS
        DATA_CONNECTIONS
          SERVER_2_3.RD_2 TO DINT2DINT_1_1_1.IN;
          SERVER_2_3.RD_1 TO DINT2DINT_1_2.IN;
          SERVER_0.QO TO LocalNumeric_0_0.check;
          SERVER_0_3.RD_3 TO DINT2DINT_1_3.IN;
          SERVER_0_3.RD_2 TO DINT2DINT_1_1.IN;
          SERVER_0_3.QO TO LocalNumeric_0_3_0.check;
          SERVER_0_3.RD_1 TO DINT2DINT_1.IN;
          SERVER_2_3.RD_3 TO DINT2DINT_1_3_1.IN;
          SERVER_2_3.QO TO LocalNumeric_2_3_0.check;
          DINT2DINT.OUT TO SERVER_1_0.SD_1;
          SERVER_1_0.QO TO LocalNumeric_1_0_0.check;
          QI TO SERVER_0.QI;
          QI TO SERVER_1_0.QI;
          QI TO SERVER_0_3.QI;
          QI TO SERVER_2_3.QI;
          DINT2DINT_3.OUT TO SERVER_2_3.SD_2;
          DINT2DINT_2.OUT TO SERVER_2_3.SD_1;
          F_EQ.OUT TO LocalNumeric_0_3_1.check;
          DINT2DINT_1.OUT TO F_EQ.IN1;
          F_EQ_1_1.OUT TO LocalNumeric_0_3_3.check;
          F_EQ_1.OUT TO LocalNumeric_0_3_2.check;
          DINT2DINT_1_1.OUT TO F_EQ_1.IN1;
          DINT2DINT_1_3.OUT TO F_EQ_1_1.IN1;
          F_EQ_1_2.OUT TO LocalNumeric_2_3_2.check;
          F_EQ_2.OUT TO LocalNumeric_2_3_1.check;
          DINT2DINT_1_2.OUT TO F_EQ_2.IN1;
          DINT2DINT_1_1_1.OUT TO F_EQ_1_2.IN1;
          DINT2DINT_1_3_1.OUT TO F_EQ_1_1_1.IN1;
          F_EQ_1_1_1.OUT TO LocalNumeric_2_3_3.check;
        END_CONNECTIONS
      END_SUBAPPLICATION
      SUBAPPLICATION MethodStringNodeId
        EVENT_INPUT
          INIT;
        END_EVENT
        EVENT_OUTPUT
          INITO;
        END_EVENT
        VAR_INPUT
          QI : BOOL;
        END_VAR
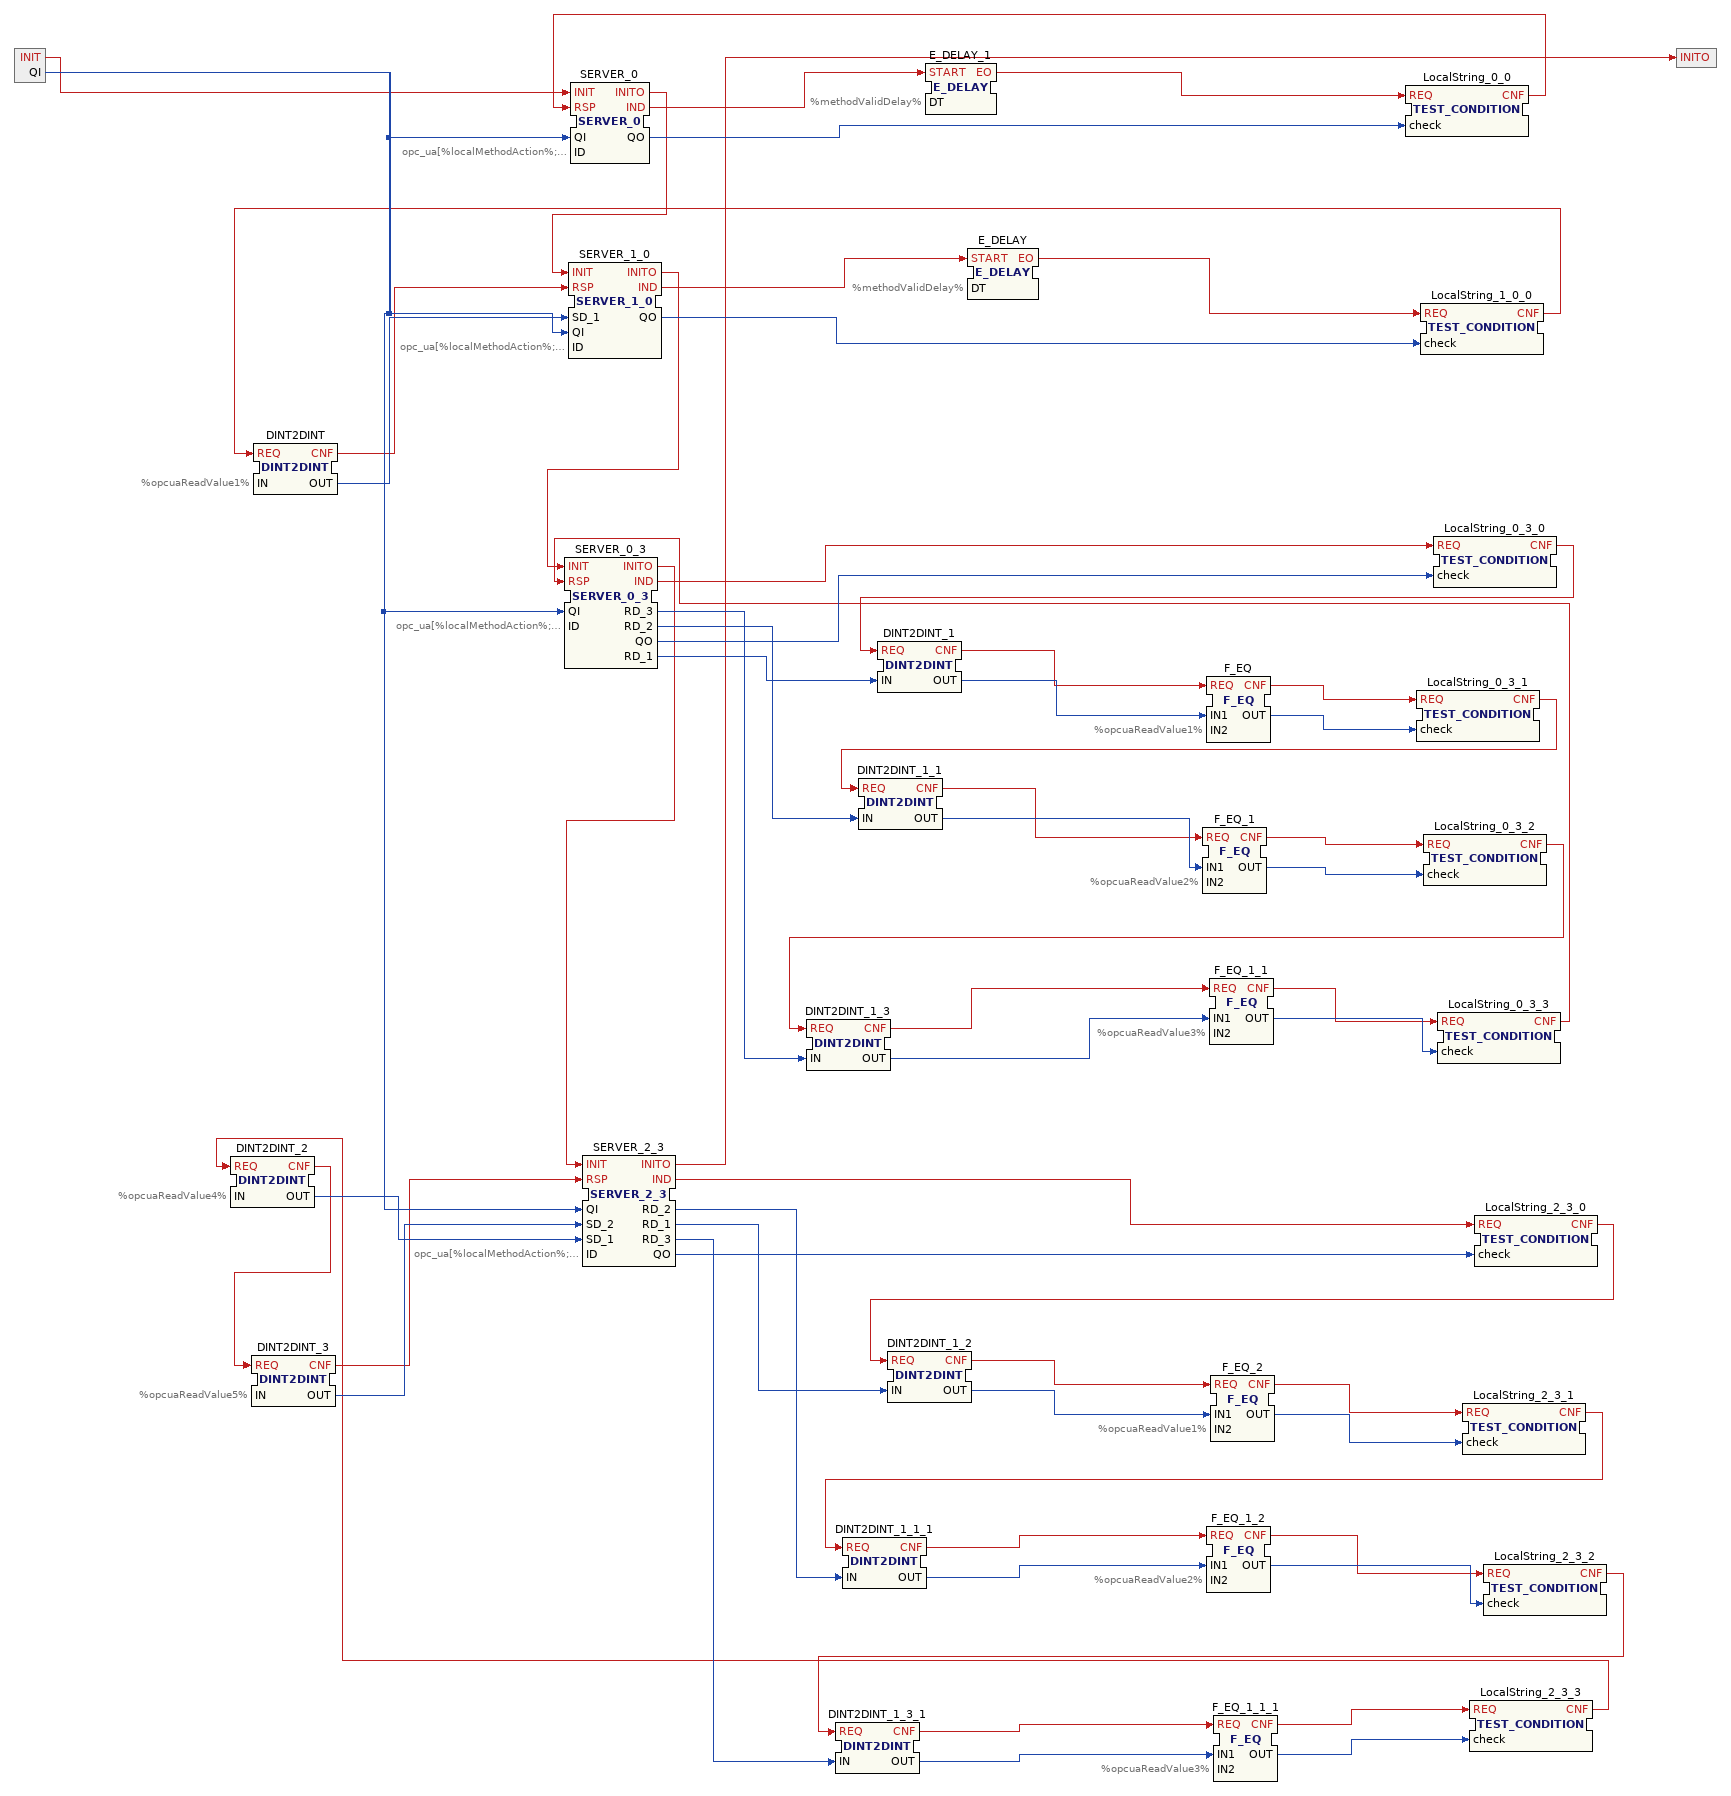
        FBS
          DINT2DINT_1_1_1 : DINT2DINT;
          DINT2DINT_1_2 : DINT2DINT;
          SERVER_0 : SERVER_0(ID := opc_ua[%localMethodAction%;%opcuaMethodCreation9%]);
          DINT2DINT_1_3 : DINT2DINT;
          DINT2DINT_1_1 : DINT2DINT;
          SERVER_0_3 : SERVER_0_3(ID := opc_ua[%localMethodAction%;%opcuaMethodCreation11%]);
          DINT2DINT_1_3_1 : DINT2DINT;
          SERVER_2_3 : SERVER_2_3(ID := opc_ua[%localMethodAction%;%opcuaMethodCreation12%]);
          LocalString_2_3_0 : TEST_CONDITION;
          LocalString_0_3_0 : TEST_CONDITION;
          SERVER_1_0 : SERVER_1_0(ID := opc_ua[%localMethodAction%;%opcuaMethodCreation10%]);
          LocalString_0_0 : TEST_CONDITION;
          LocalString_1_0_0 : TEST_CONDITION;
          DINT2DINT : DINT2DINT(IN := %opcuaReadValue1%);
          DINT2DINT_1 : DINT2DINT;
          DINT2DINT_2 : DINT2DINT(IN := %opcuaReadValue4%);
          DINT2DINT_3 : DINT2DINT(IN := %opcuaReadValue5%);
          LocalString_0_3_1 : TEST_CONDITION;
          LocalString_2_3_2 : TEST_CONDITION;
          LocalString_0_3_2 : TEST_CONDITION;
          LocalString_0_3_3 : TEST_CONDITION;
          LocalString_2_3_3 : TEST_CONDITION;
          F_EQ : F_EQ(IN2 := %opcuaReadValue1%);
          F_EQ_1 : F_EQ(IN2 := %opcuaReadValue2%);
          F_EQ_1_1 : F_EQ(IN2 := %opcuaReadValue3%);
          LocalString_2_3_1 : TEST_CONDITION;
          F_EQ_1_2 : F_EQ(IN2 := %opcuaReadValue2%);
          F_EQ_2 : F_EQ(IN2 := %opcuaReadValue1%);
          F_EQ_1_1_1 : F_EQ(IN2 := %opcuaReadValue3%);
          E_DELAY : E_DELAY(DT := %methodValidDelay%);
          E_DELAY_1 : E_DELAY(DT := %methodValidDelay%);
        END_FBS
        EVENT_CONNECTIONS
          INIT TO SERVER_0.INIT;
          SERVER_0.INITO TO SERVER_1_0.INIT;
          SERVER_1_0.INITO TO SERVER_0_3.INIT;
          SERVER_0_3.INITO TO SERVER_2_3.INIT;
          LocalString_0_0.CNF TO SERVER_0.RSP;
          SERVER_2_3.INITO TO INITO;
          LocalString_1_0_0.CNF TO DINT2DINT.REQ;
          DINT2DINT.CNF TO SERVER_1_0.RSP;
          SERVER_0_3.IND TO LocalString_0_3_0.REQ;
          LocalString_0_3_0.CNF TO DINT2DINT_1.REQ;
          DINT2DINT_1.CNF TO F_EQ.REQ;
          F_EQ.CNF TO LocalString_0_3_1.REQ;
          F_EQ_1.CNF TO LocalString_0_3_2.REQ;
          F_EQ_1_1.CNF TO LocalString_0_3_3.REQ;
          LocalString_0_3_1.CNF TO DINT2DINT_1_1.REQ;
          DINT2DINT_1_1.CNF TO F_EQ_1.REQ;
          LocalString_0_3_2.CNF TO DINT2DINT_1_3.REQ;
          DINT2DINT_1_3.CNF TO F_EQ_1_1.REQ;
          LocalString_0_3_3.CNF TO SERVER_0_3.RSP;
          SERVER_2_3.IND TO LocalString_2_3_0.REQ;
          LocalString_2_3_0.CNF TO DINT2DINT_1_2.REQ;
          DINT2DINT_1_2.CNF TO F_EQ_2.REQ;
          F_EQ_2.CNF TO LocalString_2_3_1.REQ;
          LocalString_2_3_1.CNF TO DINT2DINT_1_1_1.REQ;
          DINT2DINT_1_1_1.CNF TO F_EQ_1_2.REQ;
          F_EQ_1_2.CNF TO LocalString_2_3_2.REQ;
          LocalString_2_3_2.CNF TO DINT2DINT_1_3_1.REQ;
          DINT2DINT_1_3_1.CNF TO F_EQ_1_1_1.REQ;
          F_EQ_1_1_1.CNF TO LocalString_2_3_3.REQ;
          LocalString_2_3_3.CNF TO DINT2DINT_2.REQ;
          DINT2DINT_2.CNF TO DINT2DINT_3.REQ;
          DINT2DINT_3.CNF TO SERVER_2_3.RSP;
          SERVER_0.IND TO E_DELAY_1.START;
          E_DELAY_1.EO TO LocalString_0_0.REQ;
          SERVER_1_0.IND TO E_DELAY.START;
          E_DELAY.EO TO LocalString_1_0_0.REQ;
        END_CONNECTIONS
        DATA_CONNECTIONS
          SERVER_2_3.RD_2 TO DINT2DINT_1_1_1.IN;
          SERVER_2_3.RD_1 TO DINT2DINT_1_2.IN;
          SERVER_0.QO TO LocalString_0_0.check;
          SERVER_0_3.RD_3 TO DINT2DINT_1_3.IN;
          SERVER_0_3.RD_2 TO DINT2DINT_1_1.IN;
          SERVER_0_3.QO TO LocalString_0_3_0.check;
          SERVER_0_3.RD_1 TO DINT2DINT_1.IN;
          SERVER_2_3.RD_3 TO DINT2DINT_1_3_1.IN;
          SERVER_2_3.QO TO LocalString_2_3_0.check;
          DINT2DINT.OUT TO SERVER_1_0.SD_1;
          SERVER_1_0.QO TO LocalString_1_0_0.check;
          QI TO SERVER_0.QI;
          QI TO SERVER_1_0.QI;
          QI TO SERVER_0_3.QI;
          QI TO SERVER_2_3.QI;
          DINT2DINT_3.OUT TO SERVER_2_3.SD_2;
          DINT2DINT_2.OUT TO SERVER_2_3.SD_1;
          F_EQ.OUT TO LocalString_0_3_1.check;
          DINT2DINT_1.OUT TO F_EQ.IN1;
          F_EQ_1_1.OUT TO LocalString_0_3_3.check;
          F_EQ_1.OUT TO LocalString_0_3_2.check;
          DINT2DINT_1_1.OUT TO F_EQ_1.IN1;
          DINT2DINT_1_3.OUT TO F_EQ_1_1.IN1;
          F_EQ_1_2.OUT TO LocalString_2_3_2.check;
          F_EQ_2.OUT TO LocalString_2_3_1.check;
          DINT2DINT_1_2.OUT TO F_EQ_2.IN1;
          DINT2DINT_1_1_1.OUT TO F_EQ_1_2.IN1;
          DINT2DINT_1_3_1.OUT TO F_EQ_1_1_1.IN1;
          F_EQ_1_1_1.OUT TO LocalString_2_3_3.check;
        END_CONNECTIONS
      END_SUBAPPLICATION
      SUBAPPLICATION MethodBytestringNodeId
        EVENT_INPUT
          INIT;
        END_EVENT
        EVENT_OUTPUT
          INITO;
        END_EVENT
        VAR_INPUT
          QI : BOOL;
        END_VAR
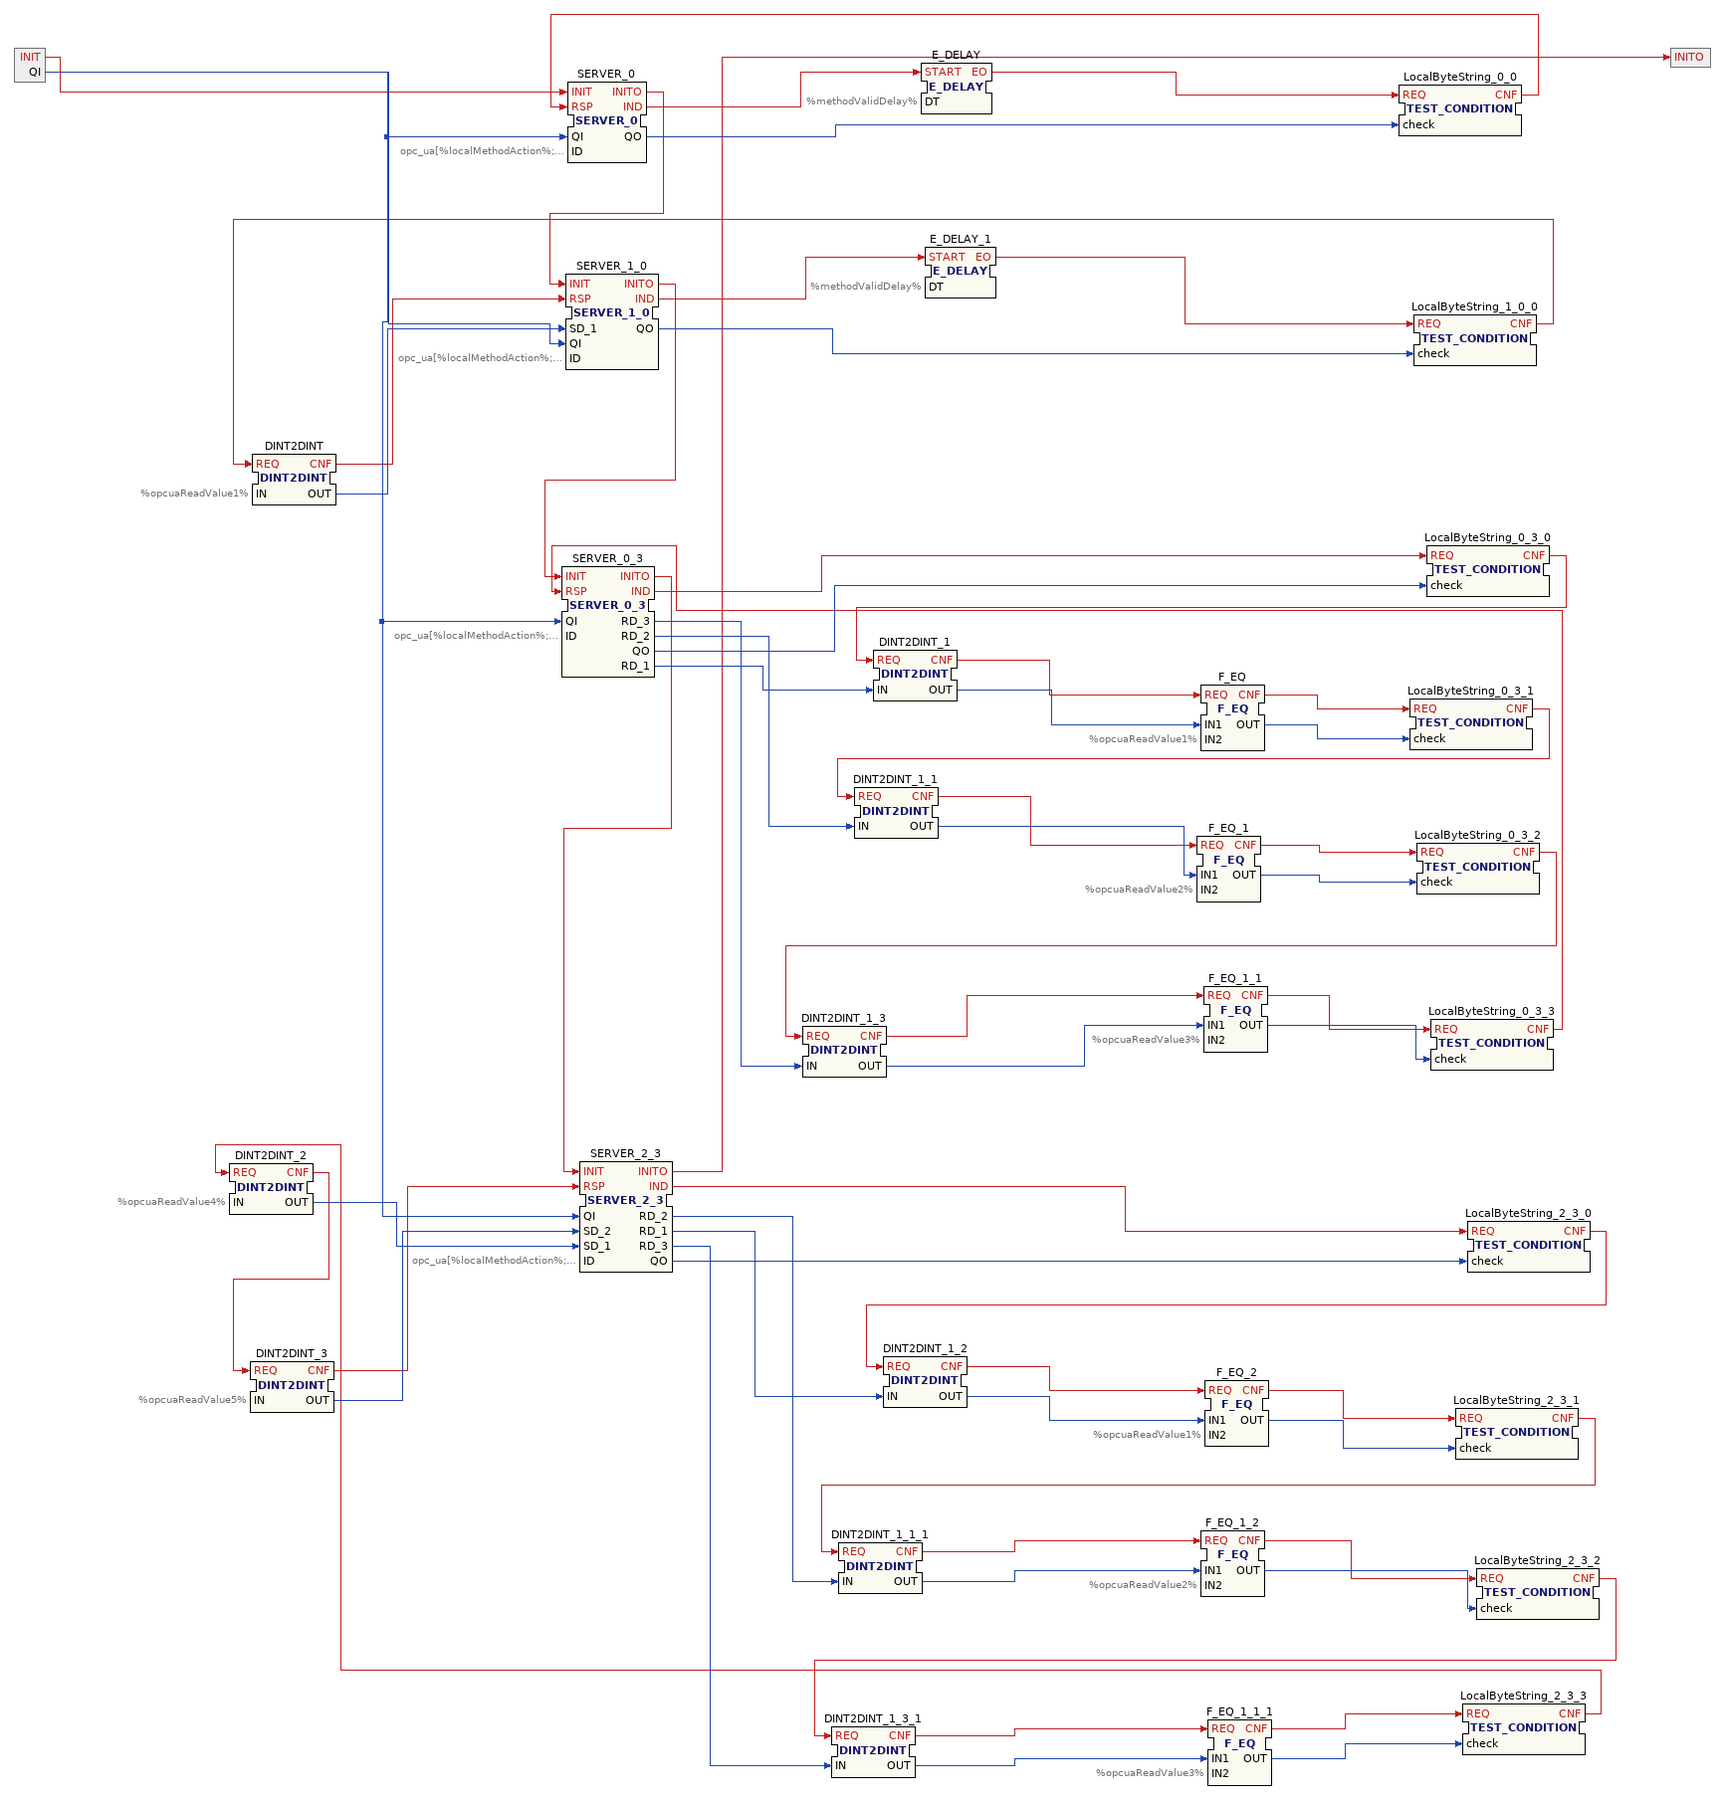
        FBS
          DINT2DINT_1_1_1 : DINT2DINT;
          DINT2DINT_1_2 : DINT2DINT;
          SERVER_0 : SERVER_0(ID := opc_ua[%localMethodAction%;%opcuaMethodCreation13%]);
          DINT2DINT_1_3 : DINT2DINT;
          DINT2DINT_1_1 : DINT2DINT;
          SERVER_0_3 : SERVER_0_3(ID := opc_ua[%localMethodAction%;%opcuaMethodCreation15%]);
          DINT2DINT_1_3_1 : DINT2DINT;
          SERVER_2_3 : SERVER_2_3(ID := opc_ua[%localMethodAction%;%opcuaMethodCreation16%]);
          LocalByteString_2_3_0 : TEST_CONDITION;
          LocalByteString_0_3_0 : TEST_CONDITION;
          SERVER_1_0 : SERVER_1_0(ID := opc_ua[%localMethodAction%;%opcuaMethodCreation14%]);
          LocalByteString_0_0 : TEST_CONDITION;
          LocalByteString_1_0_0 : TEST_CONDITION;
          DINT2DINT : DINT2DINT(IN := %opcuaReadValue1%);
          DINT2DINT_1 : DINT2DINT;
          DINT2DINT_2 : DINT2DINT(IN := %opcuaReadValue4%);
          DINT2DINT_3 : DINT2DINT(IN := %opcuaReadValue5%);
          LocalByteString_0_3_1 : TEST_CONDITION;
          LocalByteString_2_3_2 : TEST_CONDITION;
          LocalByteString_0_3_2 : TEST_CONDITION;
          LocalByteString_0_3_3 : TEST_CONDITION;
          LocalByteString_2_3_3 : TEST_CONDITION;
          F_EQ : F_EQ(IN2 := %opcuaReadValue1%);
          F_EQ_1 : F_EQ(IN2 := %opcuaReadValue2%);
          F_EQ_1_1 : F_EQ(IN2 := %opcuaReadValue3%);
          LocalByteString_2_3_1 : TEST_CONDITION;
          F_EQ_1_2 : F_EQ(IN2 := %opcuaReadValue2%);
          F_EQ_2 : F_EQ(IN2 := %opcuaReadValue1%);
          F_EQ_1_1_1 : F_EQ(IN2 := %opcuaReadValue3%);
          E_DELAY : E_DELAY(DT := %methodValidDelay%);
          E_DELAY_1 : E_DELAY(DT := %methodValidDelay%);
        END_FBS
        EVENT_CONNECTIONS
          INIT TO SERVER_0.INIT;
          SERVER_0.INITO TO SERVER_1_0.INIT;
          SERVER_1_0.INITO TO SERVER_0_3.INIT;
          SERVER_0_3.INITO TO SERVER_2_3.INIT;
          LocalByteString_0_0.CNF TO SERVER_0.RSP;
          SERVER_2_3.INITO TO INITO;
          LocalByteString_1_0_0.CNF TO DINT2DINT.REQ;
          DINT2DINT.CNF TO SERVER_1_0.RSP;
          SERVER_0_3.IND TO LocalByteString_0_3_0.REQ;
          LocalByteString_0_3_0.CNF TO DINT2DINT_1.REQ;
          DINT2DINT_1.CNF TO F_EQ.REQ;
          F_EQ.CNF TO LocalByteString_0_3_1.REQ;
          F_EQ_1.CNF TO LocalByteString_0_3_2.REQ;
          F_EQ_1_1.CNF TO LocalByteString_0_3_3.REQ;
          LocalByteString_0_3_1.CNF TO DINT2DINT_1_1.REQ;
          DINT2DINT_1_1.CNF TO F_EQ_1.REQ;
          LocalByteString_0_3_2.CNF TO DINT2DINT_1_3.REQ;
          DINT2DINT_1_3.CNF TO F_EQ_1_1.REQ;
          LocalByteString_0_3_3.CNF TO SERVER_0_3.RSP;
          SERVER_2_3.IND TO LocalByteString_2_3_0.REQ;
          LocalByteString_2_3_0.CNF TO DINT2DINT_1_2.REQ;
          DINT2DINT_1_2.CNF TO F_EQ_2.REQ;
          F_EQ_2.CNF TO LocalByteString_2_3_1.REQ;
          LocalByteString_2_3_1.CNF TO DINT2DINT_1_1_1.REQ;
          DINT2DINT_1_1_1.CNF TO F_EQ_1_2.REQ;
          F_EQ_1_2.CNF TO LocalByteString_2_3_2.REQ;
          LocalByteString_2_3_2.CNF TO DINT2DINT_1_3_1.REQ;
          DINT2DINT_1_3_1.CNF TO F_EQ_1_1_1.REQ;
          F_EQ_1_1_1.CNF TO LocalByteString_2_3_3.REQ;
          LocalByteString_2_3_3.CNF TO DINT2DINT_2.REQ;
          DINT2DINT_2.CNF TO DINT2DINT_3.REQ;
          DINT2DINT_3.CNF TO SERVER_2_3.RSP;
          SERVER_1_0.IND TO E_DELAY_1.START;
          E_DELAY_1.EO TO LocalByteString_1_0_0.REQ;
          SERVER_0.IND TO E_DELAY.START;
          E_DELAY.EO TO LocalByteString_0_0.REQ;
        END_CONNECTIONS
        DATA_CONNECTIONS
          SERVER_2_3.RD_2 TO DINT2DINT_1_1_1.IN;
          SERVER_2_3.RD_1 TO DINT2DINT_1_2.IN;
          SERVER_0.QO TO LocalByteString_0_0.check;
          SERVER_0_3.RD_3 TO DINT2DINT_1_3.IN;
          SERVER_0_3.RD_2 TO DINT2DINT_1_1.IN;
          SERVER_0_3.QO TO LocalByteString_0_3_0.check;
          SERVER_0_3.RD_1 TO DINT2DINT_1.IN;
          SERVER_2_3.RD_3 TO DINT2DINT_1_3_1.IN;
          SERVER_2_3.QO TO LocalByteString_2_3_0.check;
          DINT2DINT.OUT TO SERVER_1_0.SD_1;
          SERVER_1_0.QO TO LocalByteString_1_0_0.check;
          QI TO SERVER_0.QI;
          QI TO SERVER_1_0.QI;
          QI TO SERVER_0_3.QI;
          QI TO SERVER_2_3.QI;
          DINT2DINT_3.OUT TO SERVER_2_3.SD_2;
          DINT2DINT_2.OUT TO SERVER_2_3.SD_1;
          F_EQ.OUT TO LocalByteString_0_3_1.check;
          DINT2DINT_1.OUT TO F_EQ.IN1;
          F_EQ_1_1.OUT TO LocalByteString_0_3_3.check;
          F_EQ_1.OUT TO LocalByteString_0_3_2.check;
          DINT2DINT_1_1.OUT TO F_EQ_1.IN1;
          DINT2DINT_1_3.OUT TO F_EQ_1_1.IN1;
          F_EQ_1_2.OUT TO LocalByteString_2_3_2.check;
          F_EQ_2.OUT TO LocalByteString_2_3_1.check;
          DINT2DINT_1_2.OUT TO F_EQ_2.IN1;
          DINT2DINT_1_1_1.OUT TO F_EQ_1_2.IN1;
          DINT2DINT_1_3_1.OUT TO F_EQ_1_1_1.IN1;
          F_EQ_1_1_1.OUT TO LocalByteString_2_3_3.check;
        END_CONNECTIONS
      END_SUBAPPLICATION
      EVENT_CONNECTIONS
        INIT TO MethodOnlyBrowseName.INIT;
        MethodNumericNodeId.INITO TO MethodStringNodeId.INIT;
        MethodStringNodeId.INITO TO MethodBytestringNodeId.INIT;
        MethodBytestringNodeId.INITO TO INITO;
        MethodOnlyBrowseName.INITO TO MethodNumericNodeId.INIT;
      END_CONNECTIONS
      DATA_CONNECTIONS
        QI TO MethodOnlyBrowseName.QI;
        QI TO MethodNumericNodeId.QI;
        QI TO MethodStringNodeId.QI;
        QI TO MethodBytestringNodeId.QI;
      END_CONNECTIONS
    END_SUBAPPLICATION
    SUBAPPLICATION RemoteMethods
      EVENT_INPUT
        INIT;
        REQ;
      END_EVENT
      EVENT_OUTPUT
        INITO;
        CNF;
      END_EVENT
      VAR_INPUT
        QI : BOOL;
      END_VAR
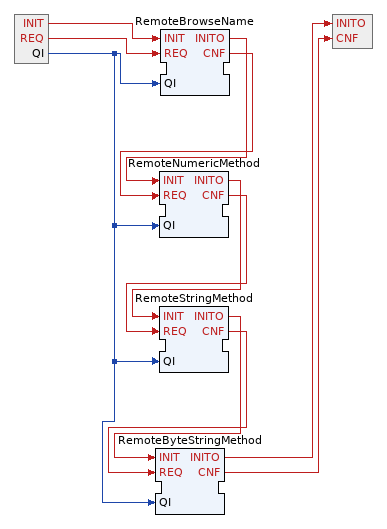
      SUBAPPLICATION RemoteBrowseName
        EVENT_INPUT
          INIT;
          REQ;
        END_EVENT
        EVENT_OUTPUT
          INITO;
          CNF;
        END_EVENT
        VAR_INPUT
          QI : BOOL;
        END_VAR
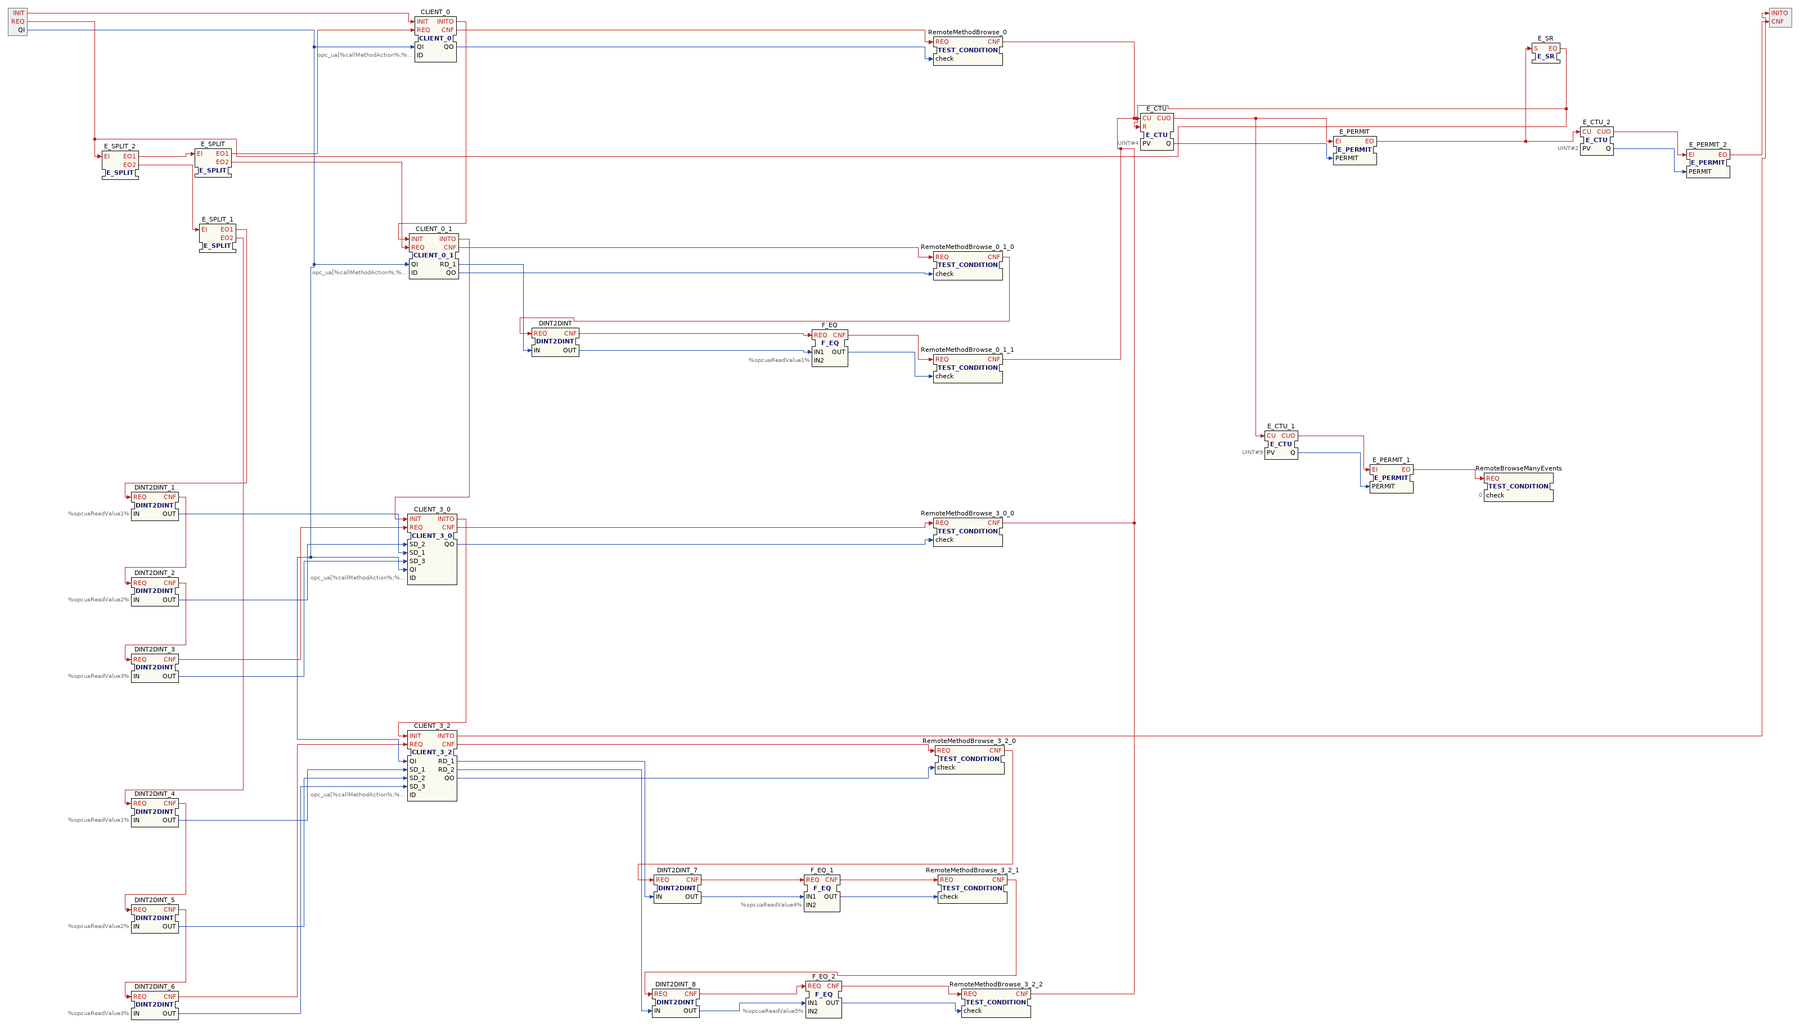
        FBS
          DINT2DINT_4 : DINT2DINT(IN := %opcuaReadValue1%);
          CLIENT_0 : CLIENT_0(ID := opc_ua[%callMethodAction%;%serverEndpoint%;%opcuaMethodCreation1%]);
          DINT2DINT_2 : DINT2DINT(IN := %opcuaReadValue2%);
          CLIENT_0_1 : CLIENT_0_1(ID := opc_ua[%callMethodAction%;%serverEndpoint%;%opcuaMethodCreation2%]);
          DINT2DINT : DINT2DINT;
          DINT2DINT_1 : DINT2DINT(IN := %opcuaReadValue1%);
          CLIENT_3_0 : CLIENT_3_0(ID := opc_ua[%callMethodAction%;%serverEndpoint%;%opcuaMethodCreation3%]);
          CLIENT_3_2 : CLIENT_3_2(ID := opc_ua[%callMethodAction%;%serverEndpoint%;%opcuaMethodCreation4%]);
          DINT2DINT_3 : DINT2DINT(IN := %opcuaReadValue3%);
          DINT2DINT_5 : DINT2DINT(IN := %opcuaReadValue2%);
          DINT2DINT_6 : DINT2DINT(IN := %opcuaReadValue3%);
          DINT2DINT_7 : DINT2DINT;
          DINT2DINT_8 : DINT2DINT;
          RemoteMethodBrowse_3_2_1 : TEST_CONDITION;
          RemoteMethodBrowse_3_2_2 : TEST_CONDITION;
          RemoteMethodBrowse_0 : TEST_CONDITION;
          RemoteMethodBrowse_0_1_0 : TEST_CONDITION;
          RemoteMethodBrowse_0_1_1 : TEST_CONDITION;
          RemoteMethodBrowse_3_2_0 : TEST_CONDITION;
          RemoteMethodBrowse_3_0_0 : TEST_CONDITION;
          F_EQ : F_EQ(IN2 := %opcuaReadValue1%);
          F_EQ_1 : F_EQ(IN2 := %opcuaReadValue4%);
          F_EQ_2 : F_EQ(IN2 := %opcuaReadValue5%);
          E_SPLIT : E_SPLIT;
          E_SPLIT_1 : E_SPLIT;
          E_CTU : E_CTU(PV := UINT#4);
          E_PERMIT : E_PERMIT;
          E_CTU_1 : E_CTU(PV := UINT#9);
          E_PERMIT_1 : E_PERMIT;
          RemoteBrowseManyEvents : TEST_CONDITION(check := 0);
          E_SPLIT_2 : E_SPLIT;
          E_PERMIT_2 : E_PERMIT;
          E_CTU_2 : E_CTU(PV := UINT#2);
          E_SR : E_SR;
        END_FBS
        EVENT_CONNECTIONS
          DINT2DINT_1.CNF TO DINT2DINT_2.REQ;
          DINT2DINT_2.CNF TO DINT2DINT_3.REQ;
          CLIENT_0_1.INITO TO CLIENT_3_0.INIT;
          INIT TO CLIENT_0.INIT;
          CLIENT_0.INITO TO CLIENT_0_1.INIT;
          CLIENT_3_0.INITO TO CLIENT_3_2.INIT;
          CLIENT_3_2.INITO TO INITO;
          CLIENT_0.CNF TO RemoteMethodBrowse_0.REQ;
          F_EQ.CNF TO RemoteMethodBrowse_0_1_1.REQ;
          CLIENT_3_0.CNF TO RemoteMethodBrowse_3_0_0.REQ;
          DINT2DINT_8.CNF TO F_EQ_2.REQ;
          DINT2DINT_7.CNF TO F_EQ_1.REQ;
          RemoteMethodBrowse_3_2_0.CNF TO DINT2DINT_7.REQ;
          F_EQ_1.CNF TO RemoteMethodBrowse_3_2_1.REQ;
          RemoteMethodBrowse_3_2_1.CNF TO DINT2DINT_8.REQ;
          F_EQ_2.CNF TO RemoteMethodBrowse_3_2_2.REQ;
          CLIENT_3_2.CNF TO RemoteMethodBrowse_3_2_0.REQ;
          DINT2DINT_4.CNF TO DINT2DINT_5.REQ;
          DINT2DINT_5.CNF TO DINT2DINT_6.REQ;
          DINT2DINT_6.CNF TO CLIENT_3_2.REQ;
          CLIENT_0_1.CNF TO RemoteMethodBrowse_0_1_0.REQ;
          RemoteMethodBrowse_0_1_0.CNF TO DINT2DINT.REQ;
          DINT2DINT.CNF TO F_EQ.REQ;
          DINT2DINT_3.CNF TO CLIENT_3_0.REQ;
          E_SPLIT.EO1 TO CLIENT_0.REQ;
          RemoteMethodBrowse_3_2_2.CNF TO E_CTU.CU;
          E_CTU.CUO TO E_CTU_1.CU;
          E_CTU.CUO TO E_PERMIT.EI;
          E_CTU_1.CUO TO E_PERMIT_1.EI;
          E_PERMIT_1.EO TO RemoteBrowseManyEvents.REQ;
          RemoteMethodBrowse_0.CNF TO E_CTU.CU;
          E_SPLIT.EO2 TO CLIENT_0_1.REQ;
          RemoteMethodBrowse_0_1_1.CNF TO E_CTU.CU;
          E_SPLIT_1.EO1 TO DINT2DINT_1.REQ;
          RemoteMethodBrowse_3_0_0.CNF TO E_CTU.CU;
          E_SPLIT_1.EO2 TO DINT2DINT_4.REQ;
          REQ TO E_SPLIT_2.EI;
          E_SPLIT_2.EO1 TO E_SPLIT.EI;
          E_SPLIT_2.EO2 TO E_SPLIT_1.EI;
          E_PERMIT.EO TO E_CTU_2.CU;
          E_CTU_2.CUO TO E_PERMIT_2.EI;
          E_PERMIT_2.EO TO CNF;
          E_PERMIT.EO TO E_SR.S;
          E_SR.EO TO E_CTU.R;
          E_SR.EO TO E_SPLIT_2.EI;
        END_CONNECTIONS
        DATA_CONNECTIONS
          DINT2DINT_2.OUT TO CLIENT_3_0.SD_2;
          CLIENT_0_1.RD_1 TO DINT2DINT.IN;
          DINT2DINT_1.OUT TO CLIENT_3_0.SD_1;
          DINT2DINT_3.OUT TO CLIENT_3_0.SD_3;
          QI TO CLIENT_0_1.QI;
          QI TO CLIENT_3_0.QI;
          QI TO CLIENT_3_2.QI;
          QI TO CLIENT_0.QI;
          DINT2DINT_4.OUT TO CLIENT_3_2.SD_1;
          DINT2DINT_5.OUT TO CLIENT_3_2.SD_2;
          CLIENT_3_2.RD_1 TO DINT2DINT_7.IN;
          CLIENT_3_2.RD_2 TO DINT2DINT_8.IN;
          DINT2DINT_6.OUT TO CLIENT_3_2.SD_3;
          CLIENT_0.QO TO RemoteMethodBrowse_0.check;
          CLIENT_0_1.QO TO RemoteMethodBrowse_0_1_0.check;
          F_EQ.OUT TO RemoteMethodBrowse_0_1_1.check;
          DINT2DINT.OUT TO F_EQ.IN1;
          CLIENT_3_0.QO TO RemoteMethodBrowse_3_0_0.check;
          DINT2DINT_7.OUT TO F_EQ_1.IN1;
          DINT2DINT_8.OUT TO F_EQ_2.IN1;
          F_EQ_1.OUT TO RemoteMethodBrowse_3_2_1.check;
          F_EQ_2.OUT TO RemoteMethodBrowse_3_2_2.check;
          CLIENT_3_2.QO TO RemoteMethodBrowse_3_2_0.check;
          E_CTU.Q TO E_PERMIT.PERMIT;
          E_CTU_1.Q TO E_PERMIT_1.PERMIT;
          E_CTU_2.Q TO E_PERMIT_2.PERMIT;
        END_CONNECTIONS
      END_SUBAPPLICATION
      SUBAPPLICATION RemoteNumericMethod
        EVENT_INPUT
          INIT;
          REQ;
        END_EVENT
        EVENT_OUTPUT
          INITO;
          CNF;
        END_EVENT
        VAR_INPUT
          QI : BOOL;
        END_VAR
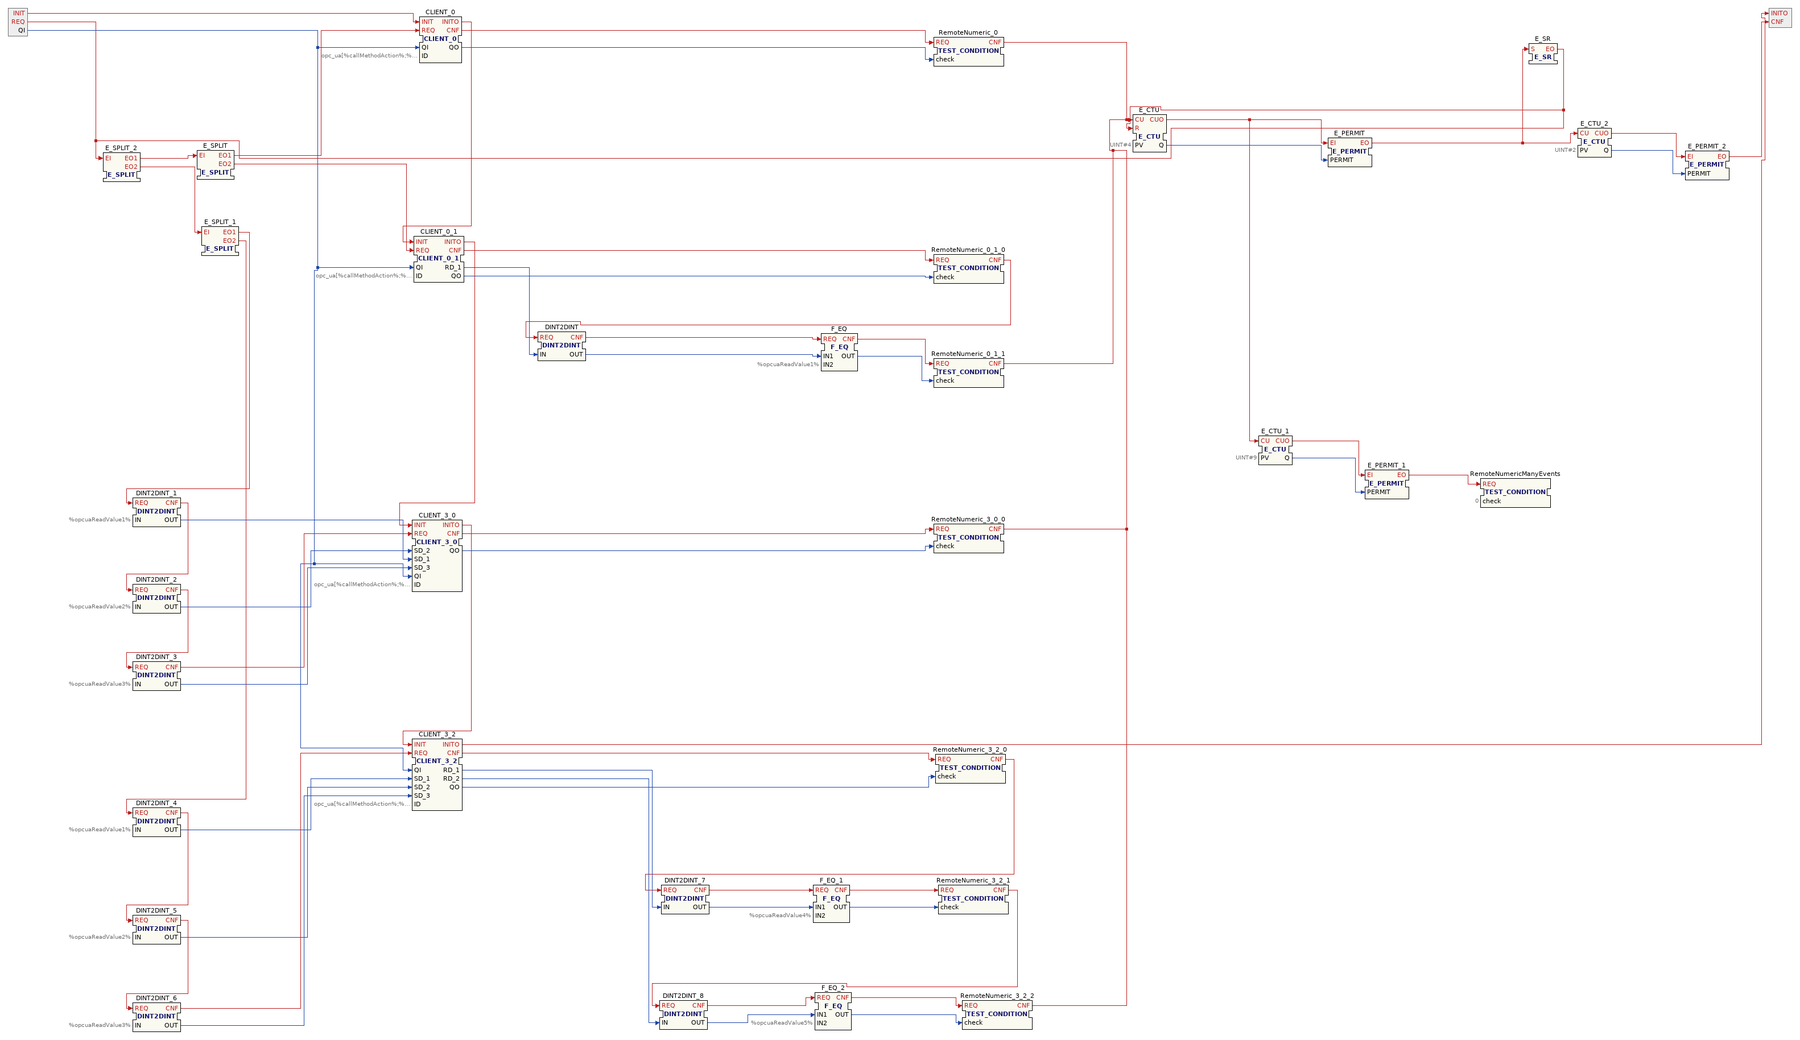
        FBS
          DINT2DINT_4 : DINT2DINT(IN := %opcuaReadValue1%);
          CLIENT_0 : CLIENT_0(ID := opc_ua[%callMethodAction%;%serverEndpoint%;%opcuaMethodCreation5%]);
          DINT2DINT_2 : DINT2DINT(IN := %opcuaReadValue2%);
          CLIENT_0_1 : CLIENT_0_1(ID := opc_ua[%callMethodAction%;%serverEndpoint%;%opcuaMethodCreation6%]);
          DINT2DINT : DINT2DINT;
          DINT2DINT_1 : DINT2DINT(IN := %opcuaReadValue1%);
          CLIENT_3_0 : CLIENT_3_0(ID := opc_ua[%callMethodAction%;%serverEndpoint%;%opcuaMethodCreation7%]);
          CLIENT_3_2 : CLIENT_3_2(ID := opc_ua[%callMethodAction%;%serverEndpoint%;%opcuaMethodCreation8%]);
          DINT2DINT_3 : DINT2DINT(IN := %opcuaReadValue3%);
          DINT2DINT_5 : DINT2DINT(IN := %opcuaReadValue2%);
          DINT2DINT_6 : DINT2DINT(IN := %opcuaReadValue3%);
          DINT2DINT_7 : DINT2DINT;
          DINT2DINT_8 : DINT2DINT;
          RemoteNumeric_3_2_1 : TEST_CONDITION;
          RemoteNumeric_3_2_2 : TEST_CONDITION;
          RemoteNumeric_0 : TEST_CONDITION;
          RemoteNumeric_0_1_0 : TEST_CONDITION;
          RemoteNumeric_0_1_1 : TEST_CONDITION;
          RemoteNumeric_3_2_0 : TEST_CONDITION;
          RemoteNumeric_3_0_0 : TEST_CONDITION;
          F_EQ : F_EQ(IN2 := %opcuaReadValue1%);
          F_EQ_1 : F_EQ(IN2 := %opcuaReadValue4%);
          F_EQ_2 : F_EQ(IN2 := %opcuaReadValue5%);
          E_SPLIT : E_SPLIT;
          E_SPLIT_1 : E_SPLIT;
          E_CTU : E_CTU(PV := UINT#4);
          E_PERMIT : E_PERMIT;
          E_CTU_1 : E_CTU(PV := UINT#9);
          E_PERMIT_1 : E_PERMIT;
          RemoteNumericManyEvents : TEST_CONDITION(check := 0);
          E_SPLIT_2 : E_SPLIT;
          E_PERMIT_2 : E_PERMIT;
          E_CTU_2 : E_CTU(PV := UINT#2);
          E_SR : E_SR;
        END_FBS
        EVENT_CONNECTIONS
          DINT2DINT_1.CNF TO DINT2DINT_2.REQ;
          DINT2DINT_2.CNF TO DINT2DINT_3.REQ;
          CLIENT_0_1.INITO TO CLIENT_3_0.INIT;
          INIT TO CLIENT_0.INIT;
          CLIENT_0.INITO TO CLIENT_0_1.INIT;
          CLIENT_3_0.INITO TO CLIENT_3_2.INIT;
          CLIENT_3_2.INITO TO INITO;
          CLIENT_0.CNF TO RemoteNumeric_0.REQ;
          F_EQ.CNF TO RemoteNumeric_0_1_1.REQ;
          CLIENT_3_0.CNF TO RemoteNumeric_3_0_0.REQ;
          DINT2DINT_8.CNF TO F_EQ_2.REQ;
          DINT2DINT_7.CNF TO F_EQ_1.REQ;
          RemoteNumeric_3_2_0.CNF TO DINT2DINT_7.REQ;
          F_EQ_1.CNF TO RemoteNumeric_3_2_1.REQ;
          RemoteNumeric_3_2_1.CNF TO DINT2DINT_8.REQ;
          F_EQ_2.CNF TO RemoteNumeric_3_2_2.REQ;
          CLIENT_3_2.CNF TO RemoteNumeric_3_2_0.REQ;
          DINT2DINT_4.CNF TO DINT2DINT_5.REQ;
          DINT2DINT_5.CNF TO DINT2DINT_6.REQ;
          DINT2DINT_6.CNF TO CLIENT_3_2.REQ;
          CLIENT_0_1.CNF TO RemoteNumeric_0_1_0.REQ;
          RemoteNumeric_0_1_0.CNF TO DINT2DINT.REQ;
          DINT2DINT.CNF TO F_EQ.REQ;
          DINT2DINT_3.CNF TO CLIENT_3_0.REQ;
          E_SPLIT.EO1 TO CLIENT_0.REQ;
          RemoteNumeric_3_2_2.CNF TO E_CTU.CU;
          E_CTU.CUO TO E_CTU_1.CU;
          E_CTU.CUO TO E_PERMIT.EI;
          E_CTU_1.CUO TO E_PERMIT_1.EI;
          E_PERMIT_1.EO TO RemoteNumericManyEvents.REQ;
          RemoteNumeric_0.CNF TO E_CTU.CU;
          E_SPLIT.EO2 TO CLIENT_0_1.REQ;
          RemoteNumeric_0_1_1.CNF TO E_CTU.CU;
          E_SPLIT_1.EO1 TO DINT2DINT_1.REQ;
          RemoteNumeric_3_0_0.CNF TO E_CTU.CU;
          E_SPLIT_1.EO2 TO DINT2DINT_4.REQ;
          REQ TO E_SPLIT_2.EI;
          E_SPLIT_2.EO1 TO E_SPLIT.EI;
          E_SPLIT_2.EO2 TO E_SPLIT_1.EI;
          E_PERMIT.EO TO E_CTU_2.CU;
          E_CTU_2.CUO TO E_PERMIT_2.EI;
          E_PERMIT_2.EO TO CNF;
          E_PERMIT.EO TO E_SR.S;
          E_SR.EO TO E_CTU.R;
          E_SR.EO TO E_SPLIT_2.EI;
        END_CONNECTIONS
        DATA_CONNECTIONS
          DINT2DINT_2.OUT TO CLIENT_3_0.SD_2;
          CLIENT_0_1.RD_1 TO DINT2DINT.IN;
          DINT2DINT_1.OUT TO CLIENT_3_0.SD_1;
          DINT2DINT_3.OUT TO CLIENT_3_0.SD_3;
          QI TO CLIENT_0_1.QI;
          QI TO CLIENT_3_0.QI;
          QI TO CLIENT_3_2.QI;
          QI TO CLIENT_0.QI;
          DINT2DINT_4.OUT TO CLIENT_3_2.SD_1;
          DINT2DINT_5.OUT TO CLIENT_3_2.SD_2;
          CLIENT_3_2.RD_1 TO DINT2DINT_7.IN;
          CLIENT_3_2.RD_2 TO DINT2DINT_8.IN;
          DINT2DINT_6.OUT TO CLIENT_3_2.SD_3;
          CLIENT_0.QO TO RemoteNumeric_0.check;
          CLIENT_0_1.QO TO RemoteNumeric_0_1_0.check;
          F_EQ.OUT TO RemoteNumeric_0_1_1.check;
          DINT2DINT.OUT TO F_EQ.IN1;
          CLIENT_3_0.QO TO RemoteNumeric_3_0_0.check;
          DINT2DINT_7.OUT TO F_EQ_1.IN1;
          DINT2DINT_8.OUT TO F_EQ_2.IN1;
          F_EQ_1.OUT TO RemoteNumeric_3_2_1.check;
          F_EQ_2.OUT TO RemoteNumeric_3_2_2.check;
          CLIENT_3_2.QO TO RemoteNumeric_3_2_0.check;
          E_CTU.Q TO E_PERMIT.PERMIT;
          E_CTU_1.Q TO E_PERMIT_1.PERMIT;
          E_CTU_2.Q TO E_PERMIT_2.PERMIT;
        END_CONNECTIONS
      END_SUBAPPLICATION
      SUBAPPLICATION RemoteStringMethod
        EVENT_INPUT
          INIT;
          REQ;
        END_EVENT
        EVENT_OUTPUT
          INITO;
          CNF;
        END_EVENT
        VAR_INPUT
          QI : BOOL;
        END_VAR
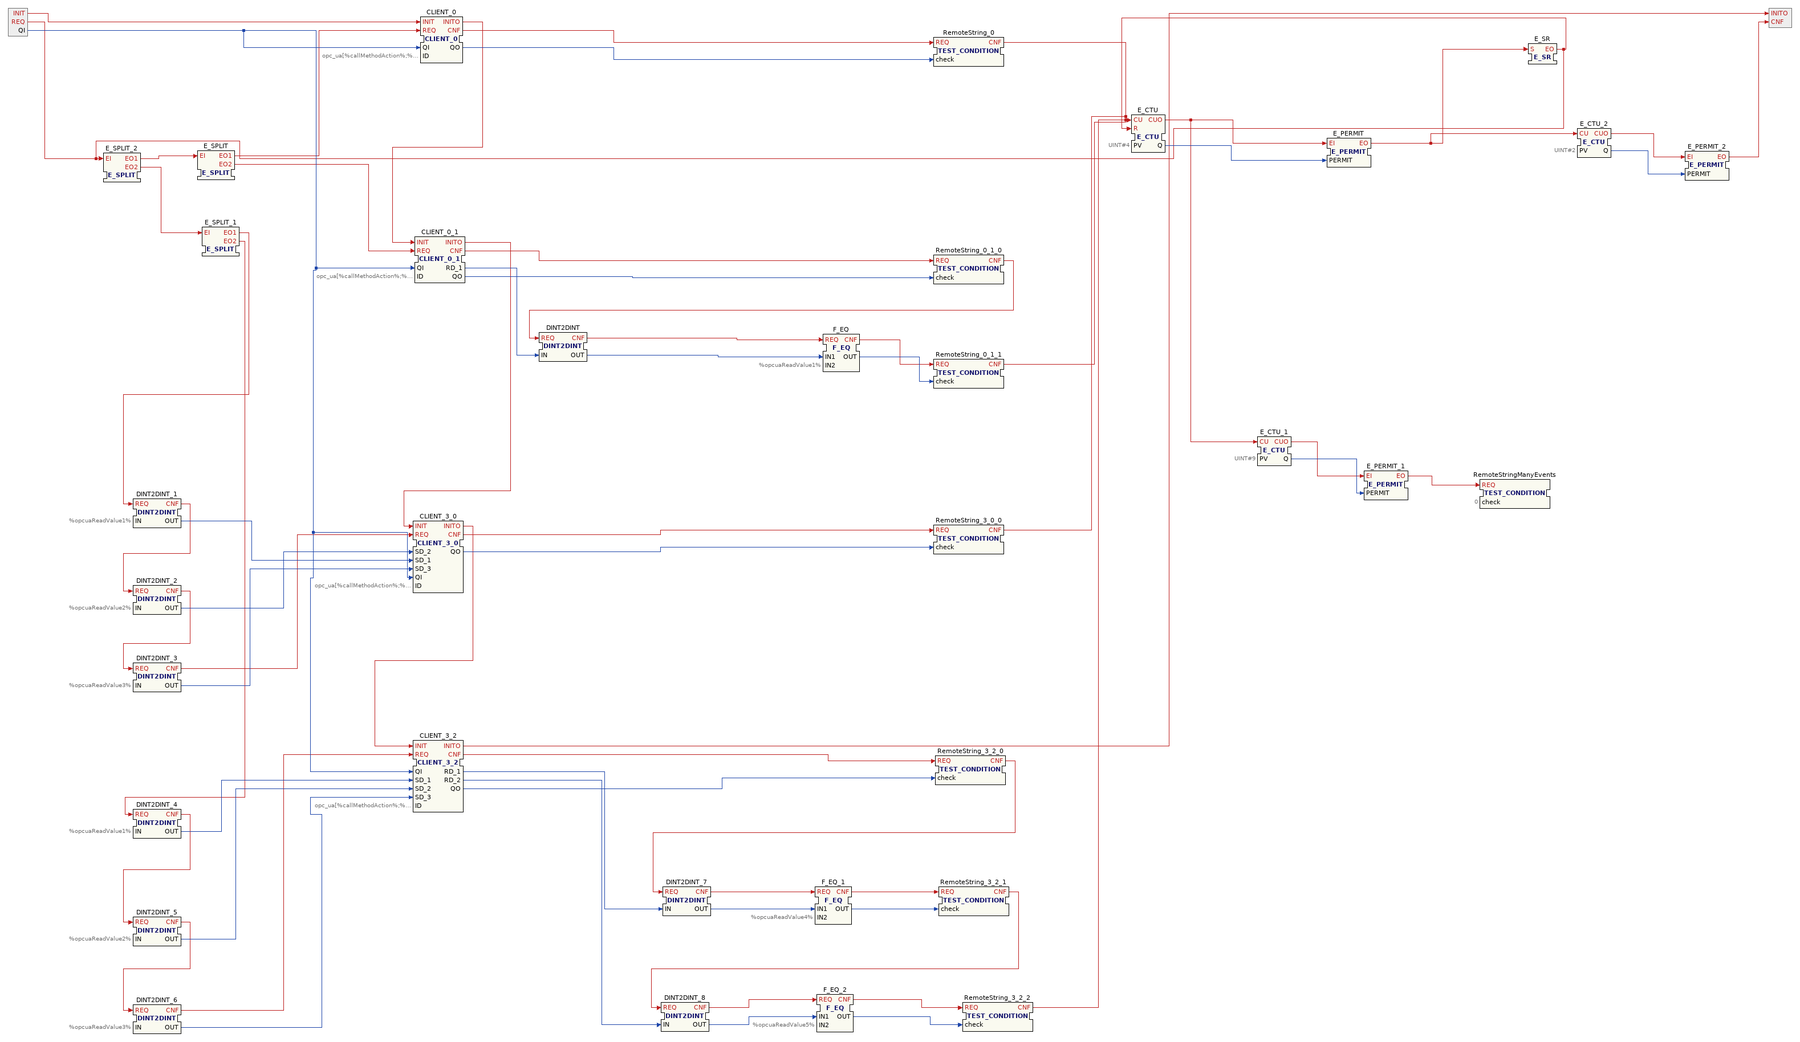
        FBS
          DINT2DINT_4 : DINT2DINT(IN := %opcuaReadValue1%);
          CLIENT_0 : CLIENT_0(ID := opc_ua[%callMethodAction%;%serverEndpoint%;%opcuaMethodCreation9%]);
          DINT2DINT_2 : DINT2DINT(IN := %opcuaReadValue2%);
          CLIENT_0_1 : CLIENT_0_1(ID := opc_ua[%callMethodAction%;%serverEndpoint%;%opcuaMethodCreation10%]);
          DINT2DINT : DINT2DINT;
          DINT2DINT_1 : DINT2DINT(IN := %opcuaReadValue1%);
          CLIENT_3_0 : CLIENT_3_0(ID := opc_ua[%callMethodAction%;%serverEndpoint%;%opcuaMethodCreation11%]);
          CLIENT_3_2 : CLIENT_3_2(ID := opc_ua[%callMethodAction%;%serverEndpoint%;%opcuaMethodCreation12%]);
          DINT2DINT_3 : DINT2DINT(IN := %opcuaReadValue3%);
          DINT2DINT_5 : DINT2DINT(IN := %opcuaReadValue2%);
          DINT2DINT_6 : DINT2DINT(IN := %opcuaReadValue3%);
          DINT2DINT_7 : DINT2DINT;
          DINT2DINT_8 : DINT2DINT;
          RemoteString_3_2_1 : TEST_CONDITION;
          RemoteString_3_2_2 : TEST_CONDITION;
          RemoteString_0 : TEST_CONDITION;
          RemoteString_0_1_0 : TEST_CONDITION;
          RemoteString_0_1_1 : TEST_CONDITION;
          RemoteString_3_2_0 : TEST_CONDITION;
          RemoteString_3_0_0 : TEST_CONDITION;
          F_EQ : F_EQ(IN2 := %opcuaReadValue1%);
          F_EQ_1 : F_EQ(IN2 := %opcuaReadValue4%);
          F_EQ_2 : F_EQ(IN2 := %opcuaReadValue5%);
          E_SPLIT : E_SPLIT;
          E_SPLIT_1 : E_SPLIT;
          E_CTU : E_CTU(PV := UINT#4);
          E_PERMIT : E_PERMIT;
          E_CTU_1 : E_CTU(PV := UINT#9);
          E_PERMIT_1 : E_PERMIT;
          RemoteStringManyEvents : TEST_CONDITION(check := 0);
          E_SPLIT_2 : E_SPLIT;
          E_PERMIT_2 : E_PERMIT;
          E_CTU_2 : E_CTU(PV := UINT#2);
          E_SR : E_SR;
        END_FBS
        EVENT_CONNECTIONS
          DINT2DINT_1.CNF TO DINT2DINT_2.REQ;
          DINT2DINT_2.CNF TO DINT2DINT_3.REQ;
          CLIENT_0_1.INITO TO CLIENT_3_0.INIT;
          INIT TO CLIENT_0.INIT;
          CLIENT_0.INITO TO CLIENT_0_1.INIT;
          CLIENT_3_0.INITO TO CLIENT_3_2.INIT;
          CLIENT_3_2.INITO TO INITO;
          CLIENT_0.CNF TO RemoteString_0.REQ;
          F_EQ.CNF TO RemoteString_0_1_1.REQ;
          CLIENT_3_0.CNF TO RemoteString_3_0_0.REQ;
          DINT2DINT_8.CNF TO F_EQ_2.REQ;
          DINT2DINT_7.CNF TO F_EQ_1.REQ;
          RemoteString_3_2_0.CNF TO DINT2DINT_7.REQ;
          F_EQ_1.CNF TO RemoteString_3_2_1.REQ;
          RemoteString_3_2_1.CNF TO DINT2DINT_8.REQ;
          F_EQ_2.CNF TO RemoteString_3_2_2.REQ;
          CLIENT_3_2.CNF TO RemoteString_3_2_0.REQ;
          DINT2DINT_4.CNF TO DINT2DINT_5.REQ;
          DINT2DINT_5.CNF TO DINT2DINT_6.REQ;
          DINT2DINT_6.CNF TO CLIENT_3_2.REQ;
          CLIENT_0_1.CNF TO RemoteString_0_1_0.REQ;
          RemoteString_0_1_0.CNF TO DINT2DINT.REQ;
          DINT2DINT.CNF TO F_EQ.REQ;
          DINT2DINT_3.CNF TO CLIENT_3_0.REQ;
          E_SPLIT.EO1 TO CLIENT_0.REQ;
          RemoteString_3_2_2.CNF TO E_CTU.CU;
          E_CTU.CUO TO E_CTU_1.CU;
          E_CTU.CUO TO E_PERMIT.EI;
          E_CTU_1.CUO TO E_PERMIT_1.EI;
          E_PERMIT_1.EO TO RemoteStringManyEvents.REQ;
          RemoteString_0.CNF TO E_CTU.CU;
          E_SPLIT.EO2 TO CLIENT_0_1.REQ;
          RemoteString_0_1_1.CNF TO E_CTU.CU;
          E_SPLIT_1.EO1 TO DINT2DINT_1.REQ;
          RemoteString_3_0_0.CNF TO E_CTU.CU;
          E_SPLIT_1.EO2 TO DINT2DINT_4.REQ;
          REQ TO E_SPLIT_2.EI;
          E_SPLIT_2.EO1 TO E_SPLIT.EI;
          E_SPLIT_2.EO2 TO E_SPLIT_1.EI;
          E_PERMIT.EO TO E_CTU_2.CU;
          E_CTU_2.CUO TO E_PERMIT_2.EI;
          E_PERMIT_2.EO TO CNF;
          E_PERMIT.EO TO E_SR.S;
          E_SR.EO TO E_CTU.R;
          E_SR.EO TO E_SPLIT_2.EI;
        END_CONNECTIONS
        DATA_CONNECTIONS
          DINT2DINT_2.OUT TO CLIENT_3_0.SD_2;
          CLIENT_0_1.RD_1 TO DINT2DINT.IN;
          DINT2DINT_1.OUT TO CLIENT_3_0.SD_1;
          DINT2DINT_3.OUT TO CLIENT_3_0.SD_3;
          QI TO CLIENT_0_1.QI;
          QI TO CLIENT_3_0.QI;
          QI TO CLIENT_3_2.QI;
          QI TO CLIENT_0.QI;
          DINT2DINT_4.OUT TO CLIENT_3_2.SD_1;
          DINT2DINT_5.OUT TO CLIENT_3_2.SD_2;
          CLIENT_3_2.RD_1 TO DINT2DINT_7.IN;
          CLIENT_3_2.RD_2 TO DINT2DINT_8.IN;
          DINT2DINT_6.OUT TO CLIENT_3_2.SD_3;
          CLIENT_0.QO TO RemoteString_0.check;
          CLIENT_0_1.QO TO RemoteString_0_1_0.check;
          F_EQ.OUT TO RemoteString_0_1_1.check;
          DINT2DINT.OUT TO F_EQ.IN1;
          CLIENT_3_0.QO TO RemoteString_3_0_0.check;
          DINT2DINT_7.OUT TO F_EQ_1.IN1;
          DINT2DINT_8.OUT TO F_EQ_2.IN1;
          F_EQ_1.OUT TO RemoteString_3_2_1.check;
          F_EQ_2.OUT TO RemoteString_3_2_2.check;
          CLIENT_3_2.QO TO RemoteString_3_2_0.check;
          E_CTU.Q TO E_PERMIT.PERMIT;
          E_CTU_1.Q TO E_PERMIT_1.PERMIT;
          E_CTU_2.Q TO E_PERMIT_2.PERMIT;
        END_CONNECTIONS
      END_SUBAPPLICATION
      SUBAPPLICATION RemoteByteStringMethod
        EVENT_INPUT
          INIT;
          REQ;
        END_EVENT
        EVENT_OUTPUT
          INITO;
          CNF;
        END_EVENT
        VAR_INPUT
          QI : BOOL;
        END_VAR
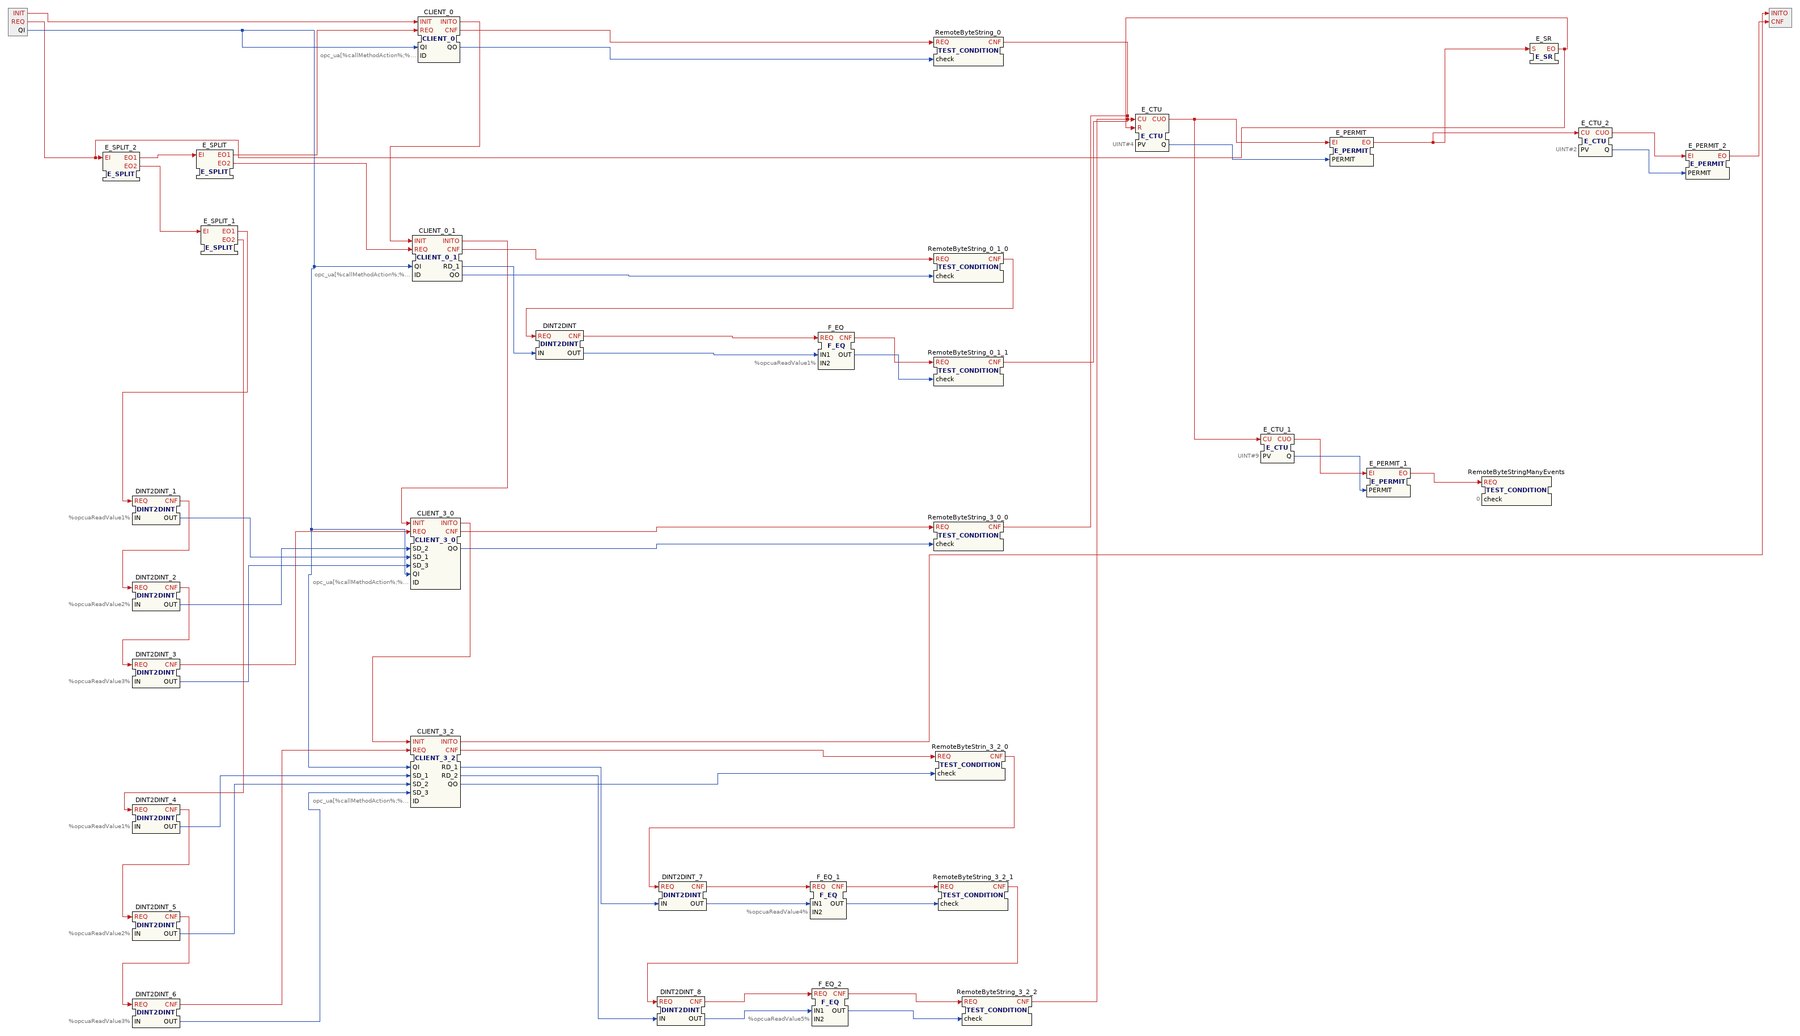
        FBS
          DINT2DINT_4 : DINT2DINT(IN := %opcuaReadValue1%);
          CLIENT_0 : CLIENT_0(ID := opc_ua[%callMethodAction%;%serverEndpoint%;%opcuaMethodCreation13%]);
          DINT2DINT_2 : DINT2DINT(IN := %opcuaReadValue2%);
          CLIENT_0_1 : CLIENT_0_1(ID := opc_ua[%callMethodAction%;%serverEndpoint%;%opcuaMethodCreation14%]);
          DINT2DINT : DINT2DINT;
          DINT2DINT_1 : DINT2DINT(IN := %opcuaReadValue1%);
          CLIENT_3_0 : CLIENT_3_0(ID := opc_ua[%callMethodAction%;%serverEndpoint%;%opcuaMethodCreation15%]);
          CLIENT_3_2 : CLIENT_3_2(ID := opc_ua[%callMethodAction%;%serverEndpoint%;%opcuaMethodCreation16%]);
          DINT2DINT_3 : DINT2DINT(IN := %opcuaReadValue3%);
          DINT2DINT_5 : DINT2DINT(IN := %opcuaReadValue2%);
          DINT2DINT_6 : DINT2DINT(IN := %opcuaReadValue3%);
          DINT2DINT_7 : DINT2DINT;
          DINT2DINT_8 : DINT2DINT;
          RemoteByteString_3_2_1 : TEST_CONDITION;
          RemoteByteString_3_2_2 : TEST_CONDITION;
          RemoteByteString_0 : TEST_CONDITION;
          RemoteByteString_0_1_0 : TEST_CONDITION;
          RemoteByteString_0_1_1 : TEST_CONDITION;
          RemoteByteStrin_3_2_0 : TEST_CONDITION;
          RemoteByteString_3_0_0 : TEST_CONDITION;
          F_EQ : F_EQ(IN2 := %opcuaReadValue1%);
          F_EQ_1 : F_EQ(IN2 := %opcuaReadValue4%);
          F_EQ_2 : F_EQ(IN2 := %opcuaReadValue5%);
          E_SPLIT : E_SPLIT;
          E_SPLIT_1 : E_SPLIT;
          E_CTU : E_CTU(PV := UINT#4);
          E_PERMIT : E_PERMIT;
          E_CTU_1 : E_CTU(PV := UINT#9);
          E_PERMIT_1 : E_PERMIT;
          RemoteByteStringManyEvents : TEST_CONDITION(check := 0);
          E_SPLIT_2 : E_SPLIT;
          E_PERMIT_2 : E_PERMIT;
          E_CTU_2 : E_CTU(PV := UINT#2);
          E_SR : E_SR;
        END_FBS
        EVENT_CONNECTIONS
          DINT2DINT_1.CNF TO DINT2DINT_2.REQ;
          DINT2DINT_2.CNF TO DINT2DINT_3.REQ;
          CLIENT_0_1.INITO TO CLIENT_3_0.INIT;
          INIT TO CLIENT_0.INIT;
          CLIENT_0.INITO TO CLIENT_0_1.INIT;
          CLIENT_3_0.INITO TO CLIENT_3_2.INIT;
          CLIENT_3_2.INITO TO INITO;
          CLIENT_0.CNF TO RemoteByteString_0.REQ;
          F_EQ.CNF TO RemoteByteString_0_1_1.REQ;
          CLIENT_3_0.CNF TO RemoteByteString_3_0_0.REQ;
          DINT2DINT_8.CNF TO F_EQ_2.REQ;
          DINT2DINT_7.CNF TO F_EQ_1.REQ;
          RemoteByteStrin_3_2_0.CNF TO DINT2DINT_7.REQ;
          F_EQ_1.CNF TO RemoteByteString_3_2_1.REQ;
          RemoteByteString_3_2_1.CNF TO DINT2DINT_8.REQ;
          F_EQ_2.CNF TO RemoteByteString_3_2_2.REQ;
          CLIENT_3_2.CNF TO RemoteByteStrin_3_2_0.REQ;
          DINT2DINT_4.CNF TO DINT2DINT_5.REQ;
          DINT2DINT_5.CNF TO DINT2DINT_6.REQ;
          DINT2DINT_6.CNF TO CLIENT_3_2.REQ;
          CLIENT_0_1.CNF TO RemoteByteString_0_1_0.REQ;
          RemoteByteString_0_1_0.CNF TO DINT2DINT.REQ;
          DINT2DINT.CNF TO F_EQ.REQ;
          DINT2DINT_3.CNF TO CLIENT_3_0.REQ;
          E_SPLIT.EO1 TO CLIENT_0.REQ;
          RemoteByteString_3_2_2.CNF TO E_CTU.CU;
          E_CTU.CUO TO E_CTU_1.CU;
          E_CTU.CUO TO E_PERMIT.EI;
          E_CTU_1.CUO TO E_PERMIT_1.EI;
          E_PERMIT_1.EO TO RemoteByteStringManyEvents.REQ;
          RemoteByteString_0.CNF TO E_CTU.CU;
          E_SPLIT.EO2 TO CLIENT_0_1.REQ;
          RemoteByteString_0_1_1.CNF TO E_CTU.CU;
          E_SPLIT_1.EO1 TO DINT2DINT_1.REQ;
          RemoteByteString_3_0_0.CNF TO E_CTU.CU;
          E_SPLIT_1.EO2 TO DINT2DINT_4.REQ;
          REQ TO E_SPLIT_2.EI;
          E_SPLIT_2.EO1 TO E_SPLIT.EI;
          E_SPLIT_2.EO2 TO E_SPLIT_1.EI;
          E_PERMIT.EO TO E_CTU_2.CU;
          E_CTU_2.CUO TO E_PERMIT_2.EI;
          E_PERMIT_2.EO TO CNF;
          E_PERMIT.EO TO E_SR.S;
          E_SR.EO TO E_CTU.R;
          E_SR.EO TO E_SPLIT_2.EI;
        END_CONNECTIONS
        DATA_CONNECTIONS
          DINT2DINT_2.OUT TO CLIENT_3_0.SD_2;
          CLIENT_0_1.RD_1 TO DINT2DINT.IN;
          DINT2DINT_1.OUT TO CLIENT_3_0.SD_1;
          DINT2DINT_3.OUT TO CLIENT_3_0.SD_3;
          QI TO CLIENT_0_1.QI;
          QI TO CLIENT_3_0.QI;
          QI TO CLIENT_3_2.QI;
          QI TO CLIENT_0.QI;
          DINT2DINT_4.OUT TO CLIENT_3_2.SD_1;
          DINT2DINT_5.OUT TO CLIENT_3_2.SD_2;
          CLIENT_3_2.RD_1 TO DINT2DINT_7.IN;
          CLIENT_3_2.RD_2 TO DINT2DINT_8.IN;
          DINT2DINT_6.OUT TO CLIENT_3_2.SD_3;
          CLIENT_0.QO TO RemoteByteString_0.check;
          CLIENT_0_1.QO TO RemoteByteString_0_1_0.check;
          F_EQ.OUT TO RemoteByteString_0_1_1.check;
          DINT2DINT.OUT TO F_EQ.IN1;
          CLIENT_3_0.QO TO RemoteByteString_3_0_0.check;
          DINT2DINT_7.OUT TO F_EQ_1.IN1;
          DINT2DINT_8.OUT TO F_EQ_2.IN1;
          F_EQ_1.OUT TO RemoteByteString_3_2_1.check;
          F_EQ_2.OUT TO RemoteByteString_3_2_2.check;
          CLIENT_3_2.QO TO RemoteByteStrin_3_2_0.check;
          E_CTU.Q TO E_PERMIT.PERMIT;
          E_CTU_1.Q TO E_PERMIT_1.PERMIT;
          E_CTU_2.Q TO E_PERMIT_2.PERMIT;
        END_CONNECTIONS
      END_SUBAPPLICATION
      EVENT_CONNECTIONS
        INIT TO RemoteBrowseName.INIT;
        REQ TO RemoteBrowseName.REQ;
        RemoteBrowseName.INITO TO RemoteNumericMethod.INIT;
        RemoteNumericMethod.INITO TO RemoteStringMethod.INIT;
        RemoteStringMethod.INITO TO RemoteByteStringMethod.INIT;
        RemoteByteStringMethod.CNF TO CNF;
        RemoteByteStringMethod.INITO TO INITO;
        RemoteStringMethod.CNF TO RemoteByteStringMethod.REQ;
        RemoteNumericMethod.CNF TO RemoteStringMethod.REQ;
        RemoteBrowseName.CNF TO RemoteNumericMethod.REQ;
      END_CONNECTIONS
      DATA_CONNECTIONS
        QI TO RemoteBrowseName.QI;
        QI TO RemoteNumericMethod.QI;
        QI TO RemoteStringMethod.QI;
        QI TO RemoteByteStringMethod.QI;
      END_CONNECTIONS
    END_SUBAPPLICATION
    SUBAPPLICATION numericNodeIdTest
      EVENT_INPUT
        INIT;
      END_EVENT
      EVENT_OUTPUT
        INITO;
      END_EVENT
      VAR_INPUT
        QI : BOOL;
      END_VAR
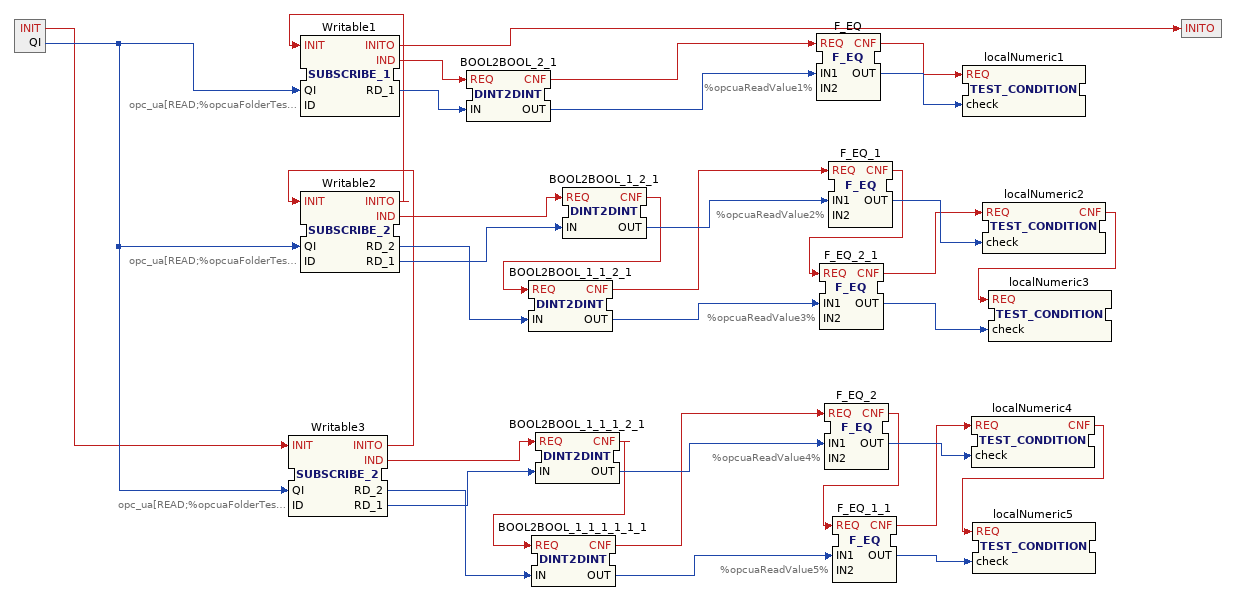
      FBS
        BOOL2BOOL_1_2_1 : DINT2DINT;
        BOOL2BOOL_2_1 : DINT2DINT;
        BOOL2BOOL_1_1_2_1 : DINT2DINT;
        BOOL2BOOL_1_1_1_2_1 : DINT2DINT;
        BOOL2BOOL_1_1_1_1_1_1 : DINT2DINT;
        Writable1 : SUBSCRIBE_1(ID := opc_ua[READ;%opcuaFolderTestWithNodeIdNumeric1%]);
        Writable2 : SUBSCRIBE_2(ID := opc_ua[READ;%opcuaFolderTestWithNodeIdNumeric2%]);
        Writable3 : SUBSCRIBE_2(ID := opc_ua[READ;%opcuaFolderTestWithNodeIdNumeric3%]);
        localNumeric1 : TEST_CONDITION;
        localNumeric2 : TEST_CONDITION;
        localNumeric3 : TEST_CONDITION;
        localNumeric4 : TEST_CONDITION;
        localNumeric5 : TEST_CONDITION;
        F_EQ : F_EQ(IN2 := %opcuaReadValue1%);
        F_EQ_1 : F_EQ(IN2 := %opcuaReadValue2%);
        F_EQ_2 : F_EQ(IN2 := %opcuaReadValue4%);
        F_EQ_1_1 : F_EQ(IN2 := %opcuaReadValue5%);
        F_EQ_2_1 : F_EQ(IN2 := %opcuaReadValue3%);
      END_FBS
      EVENT_CONNECTIONS
        Writable1.INITO TO INITO;
        Writable2.INITO TO Writable1.INIT;
        INIT TO Writable3.INIT;
        Writable3.INITO TO Writable2.INIT;
        Writable1.IND TO BOOL2BOOL_2_1.REQ;
        Writable2.IND TO BOOL2BOOL_1_2_1.REQ;
        BOOL2BOOL_1_2_1.CNF TO BOOL2BOOL_1_1_2_1.REQ;
        Writable3.IND TO BOOL2BOOL_1_1_1_2_1.REQ;
        BOOL2BOOL_1_1_1_2_1.CNF TO BOOL2BOOL_1_1_1_1_1_1.REQ;
        BOOL2BOOL_2_1.CNF TO F_EQ.REQ;
        F_EQ.CNF TO localNumeric1.REQ;
        BOOL2BOOL_1_1_2_1.CNF TO F_EQ_1.REQ;
        F_EQ_1.CNF TO F_EQ_2_1.REQ;
        F_EQ_2_1.CNF TO localNumeric2.REQ;
        BOOL2BOOL_1_1_1_1_1_1.CNF TO F_EQ_2.REQ;
        F_EQ_2.CNF TO F_EQ_1_1.REQ;
        F_EQ_1_1.CNF TO localNumeric4.REQ;
        localNumeric4.CNF TO localNumeric5.REQ;
        localNumeric2.CNF TO localNumeric3.REQ;
      END_CONNECTIONS
      DATA_CONNECTIONS
        QI TO Writable1.QI;
        QI TO Writable2.QI;
        QI TO Writable3.QI;
        Writable1.RD_1 TO BOOL2BOOL_2_1.IN;
        Writable3.RD_2 TO BOOL2BOOL_1_1_1_1_1_1.IN;
        Writable3.RD_1 TO BOOL2BOOL_1_1_1_2_1.IN;
        Writable2.RD_2 TO BOOL2BOOL_1_1_2_1.IN;
        Writable2.RD_1 TO BOOL2BOOL_1_2_1.IN;
        BOOL2BOOL_2_1.OUT TO F_EQ.IN1;
        F_EQ.OUT TO localNumeric1.check;
        BOOL2BOOL_1_1_2_1.OUT TO F_EQ_2_1.IN1;
        BOOL2BOOL_1_2_1.OUT TO F_EQ_1.IN1;
        BOOL2BOOL_1_1_1_2_1.OUT TO F_EQ_2.IN1;
        BOOL2BOOL_1_1_1_1_1_1.OUT TO F_EQ_1_1.IN1;
        F_EQ_1_1.OUT TO localNumeric5.check;
        F_EQ_2.OUT TO localNumeric4.check;
        F_EQ_2_1.OUT TO localNumeric3.check;
        F_EQ_1.OUT TO localNumeric2.check;
      END_CONNECTIONS
    END_SUBAPPLICATION
    SUBAPPLICATION stringNodeIdTest
      EVENT_INPUT
        INIT;
      END_EVENT
      EVENT_OUTPUT
        INITO;
      END_EVENT
      VAR_INPUT
        QI : BOOL;
      END_VAR
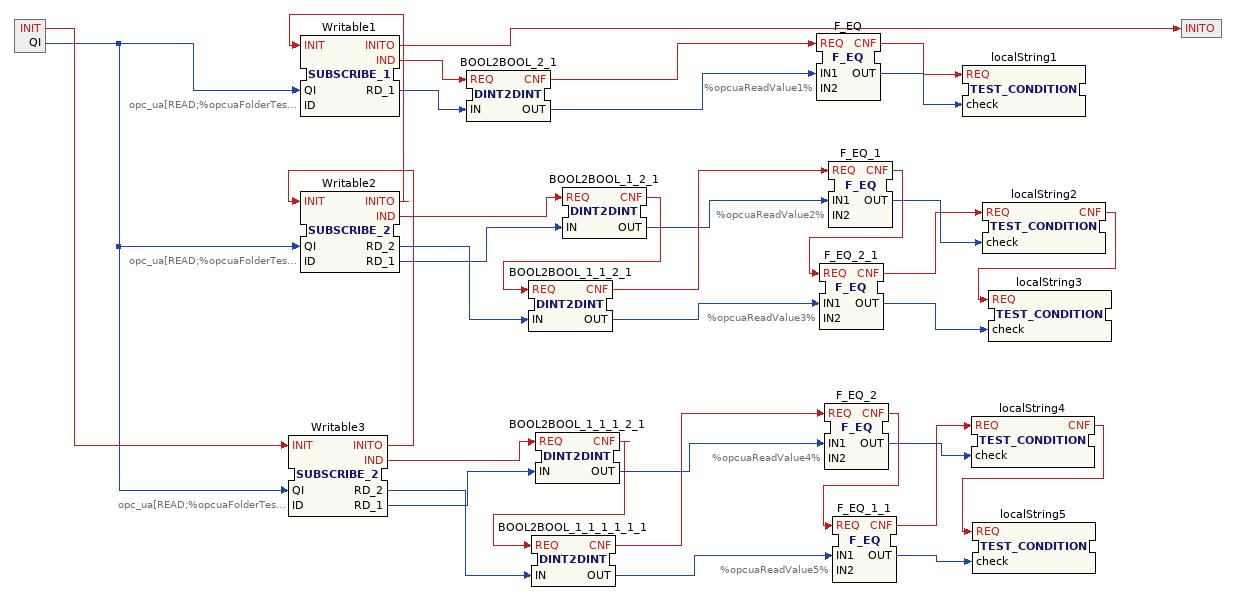
      FBS
        BOOL2BOOL_1_2_1 : DINT2DINT;
        BOOL2BOOL_2_1 : DINT2DINT;
        BOOL2BOOL_1_1_2_1 : DINT2DINT;
        BOOL2BOOL_1_1_1_2_1 : DINT2DINT;
        BOOL2BOOL_1_1_1_1_1_1 : DINT2DINT;
        Writable1 : SUBSCRIBE_1(ID := opc_ua[READ;%opcuaFolderTestWithNodeIdString1%]);
        Writable2 : SUBSCRIBE_2(ID := opc_ua[READ;%opcuaFolderTestWithNodeIdString2%]);
        Writable3 : SUBSCRIBE_2(ID := opc_ua[READ;%opcuaFolderTestWithNodeIdString3%]);
        localString1 : TEST_CONDITION;
        localString2 : TEST_CONDITION;
        localString3 : TEST_CONDITION;
        localString4 : TEST_CONDITION;
        localString5 : TEST_CONDITION;
        F_EQ : F_EQ(IN2 := %opcuaReadValue1%);
        F_EQ_1 : F_EQ(IN2 := %opcuaReadValue2%);
        F_EQ_2 : F_EQ(IN2 := %opcuaReadValue4%);
        F_EQ_1_1 : F_EQ(IN2 := %opcuaReadValue5%);
        F_EQ_2_1 : F_EQ(IN2 := %opcuaReadValue3%);
      END_FBS
      EVENT_CONNECTIONS
        Writable1.INITO TO INITO;
        Writable2.INITO TO Writable1.INIT;
        INIT TO Writable3.INIT;
        Writable3.INITO TO Writable2.INIT;
        Writable1.IND TO BOOL2BOOL_2_1.REQ;
        Writable2.IND TO BOOL2BOOL_1_2_1.REQ;
        BOOL2BOOL_1_2_1.CNF TO BOOL2BOOL_1_1_2_1.REQ;
        Writable3.IND TO BOOL2BOOL_1_1_1_2_1.REQ;
        BOOL2BOOL_1_1_1_2_1.CNF TO BOOL2BOOL_1_1_1_1_1_1.REQ;
        BOOL2BOOL_2_1.CNF TO F_EQ.REQ;
        F_EQ.CNF TO localString1.REQ;
        BOOL2BOOL_1_1_2_1.CNF TO F_EQ_1.REQ;
        F_EQ_1.CNF TO F_EQ_2_1.REQ;
        F_EQ_2_1.CNF TO localString2.REQ;
        BOOL2BOOL_1_1_1_1_1_1.CNF TO F_EQ_2.REQ;
        F_EQ_2.CNF TO F_EQ_1_1.REQ;
        F_EQ_1_1.CNF TO localString4.REQ;
        localString4.CNF TO localString5.REQ;
        localString2.CNF TO localString3.REQ;
      END_CONNECTIONS
      DATA_CONNECTIONS
        QI TO Writable1.QI;
        QI TO Writable2.QI;
        QI TO Writable3.QI;
        Writable1.RD_1 TO BOOL2BOOL_2_1.IN;
        Writable3.RD_2 TO BOOL2BOOL_1_1_1_1_1_1.IN;
        Writable3.RD_1 TO BOOL2BOOL_1_1_1_2_1.IN;
        Writable2.RD_2 TO BOOL2BOOL_1_1_2_1.IN;
        Writable2.RD_1 TO BOOL2BOOL_1_2_1.IN;
        BOOL2BOOL_2_1.OUT TO F_EQ.IN1;
        F_EQ.OUT TO localString1.check;
        BOOL2BOOL_1_1_2_1.OUT TO F_EQ_2_1.IN1;
        BOOL2BOOL_1_2_1.OUT TO F_EQ_1.IN1;
        BOOL2BOOL_1_1_1_2_1.OUT TO F_EQ_2.IN1;
        BOOL2BOOL_1_1_1_1_1_1.OUT TO F_EQ_1_1.IN1;
        F_EQ_1_1.OUT TO localString5.check;
        F_EQ_2.OUT TO localString4.check;
        F_EQ_2_1.OUT TO localString3.check;
        F_EQ_1.OUT TO localString2.check;
      END_CONNECTIONS
    END_SUBAPPLICATION
    SUBAPPLICATION byteStringNodeIdTest
      EVENT_INPUT
        INIT;
      END_EVENT
      EVENT_OUTPUT
        INITO;
      END_EVENT
      VAR_INPUT
        QI : BOOL;
      END_VAR
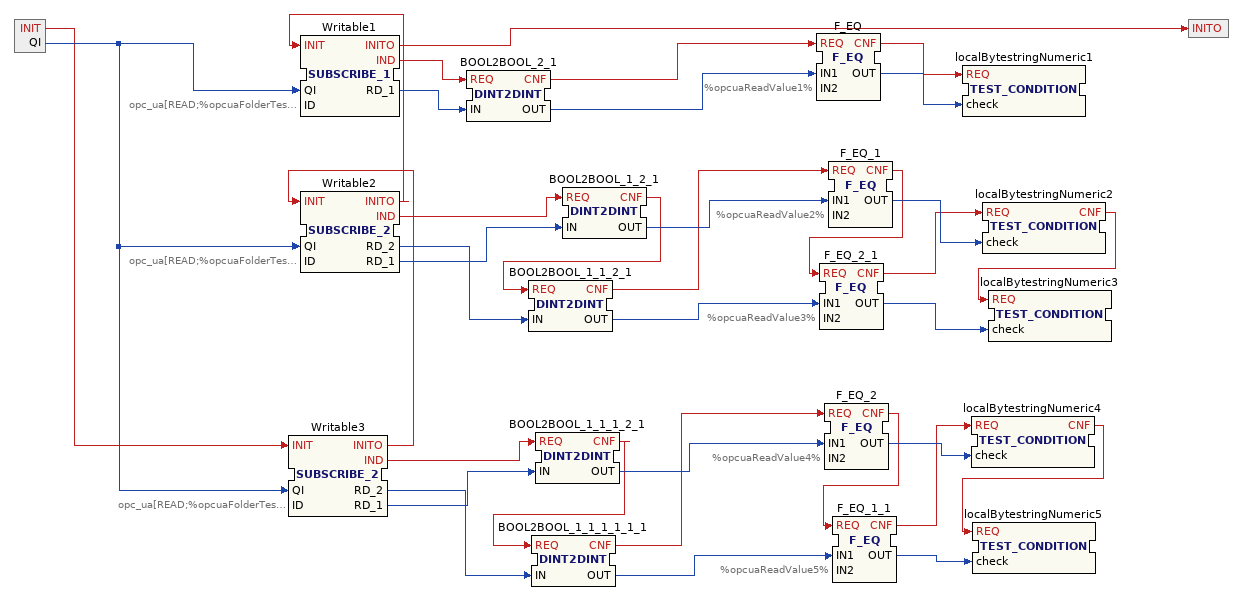
      FBS
        BOOL2BOOL_1_2_1 : DINT2DINT;
        BOOL2BOOL_2_1 : DINT2DINT;
        BOOL2BOOL_1_1_2_1 : DINT2DINT;
        BOOL2BOOL_1_1_1_2_1 : DINT2DINT;
        BOOL2BOOL_1_1_1_1_1_1 : DINT2DINT;
        Writable1 : SUBSCRIBE_1(ID := opc_ua[READ;%opcuaFolderTestWithNodeIdByteString1%]);
        Writable2 : SUBSCRIBE_2(ID := opc_ua[READ;%opcuaFolderTestWithNodeIdByteString2%]);
        Writable3 : SUBSCRIBE_2(ID := opc_ua[READ;%opcuaFolderTestWithNodeIdByteString3%]);
        localBytestringNumeric1 : TEST_CONDITION;
        localBytestringNumeric2 : TEST_CONDITION;
        localBytestringNumeric3 : TEST_CONDITION;
        localBytestringNumeric4 : TEST_CONDITION;
        localBytestringNumeric5 : TEST_CONDITION;
        F_EQ : F_EQ(IN2 := %opcuaReadValue1%);
        F_EQ_1 : F_EQ(IN2 := %opcuaReadValue2%);
        F_EQ_2 : F_EQ(IN2 := %opcuaReadValue4%);
        F_EQ_1_1 : F_EQ(IN2 := %opcuaReadValue5%);
        F_EQ_2_1 : F_EQ(IN2 := %opcuaReadValue3%);
      END_FBS
      EVENT_CONNECTIONS
        Writable1.INITO TO INITO;
        Writable2.INITO TO Writable1.INIT;
        INIT TO Writable3.INIT;
        Writable3.INITO TO Writable2.INIT;
        Writable1.IND TO BOOL2BOOL_2_1.REQ;
        Writable2.IND TO BOOL2BOOL_1_2_1.REQ;
        BOOL2BOOL_1_2_1.CNF TO BOOL2BOOL_1_1_2_1.REQ;
        Writable3.IND TO BOOL2BOOL_1_1_1_2_1.REQ;
        BOOL2BOOL_1_1_1_2_1.CNF TO BOOL2BOOL_1_1_1_1_1_1.REQ;
        BOOL2BOOL_2_1.CNF TO F_EQ.REQ;
        F_EQ.CNF TO localBytestringNumeric1.REQ;
        BOOL2BOOL_1_1_2_1.CNF TO F_EQ_1.REQ;
        F_EQ_1.CNF TO F_EQ_2_1.REQ;
        F_EQ_2_1.CNF TO localBytestringNumeric2.REQ;
        BOOL2BOOL_1_1_1_1_1_1.CNF TO F_EQ_2.REQ;
        F_EQ_2.CNF TO F_EQ_1_1.REQ;
        F_EQ_1_1.CNF TO localBytestringNumeric4.REQ;
        localBytestringNumeric4.CNF TO localBytestringNumeric5.REQ;
        localBytestringNumeric2.CNF TO localBytestringNumeric3.REQ;
      END_CONNECTIONS
      DATA_CONNECTIONS
        QI TO Writable1.QI;
        QI TO Writable2.QI;
        QI TO Writable3.QI;
        Writable1.RD_1 TO BOOL2BOOL_2_1.IN;
        Writable3.RD_2 TO BOOL2BOOL_1_1_1_1_1_1.IN;
        Writable3.RD_1 TO BOOL2BOOL_1_1_1_2_1.IN;
        Writable2.RD_2 TO BOOL2BOOL_1_1_2_1.IN;
        Writable2.RD_1 TO BOOL2BOOL_1_2_1.IN;
        BOOL2BOOL_2_1.OUT TO F_EQ.IN1;
        F_EQ.OUT TO localBytestringNumeric1.check;
        BOOL2BOOL_1_1_2_1.OUT TO F_EQ_2_1.IN1;
        BOOL2BOOL_1_2_1.OUT TO F_EQ_1.IN1;
        BOOL2BOOL_1_1_1_2_1.OUT TO F_EQ_2.IN1;
        BOOL2BOOL_1_1_1_1_1_1.OUT TO F_EQ_1_1.IN1;
        F_EQ_1_1.OUT TO localBytestringNumeric5.check;
        F_EQ_2.OUT TO localBytestringNumeric4.check;
        F_EQ_2_1.OUT TO localBytestringNumeric3.check;
        F_EQ_1.OUT TO localBytestringNumeric2.check;
      END_CONNECTIONS
    END_SUBAPPLICATION
    SUBAPPLICATION IsolatedCases
      EVENT_INPUT
        INIT;
      END_EVENT
      EVENT_OUTPUT
        INITO;
      END_EVENT
      VAR_INPUT
        QI : BOOL;
      END_VAR
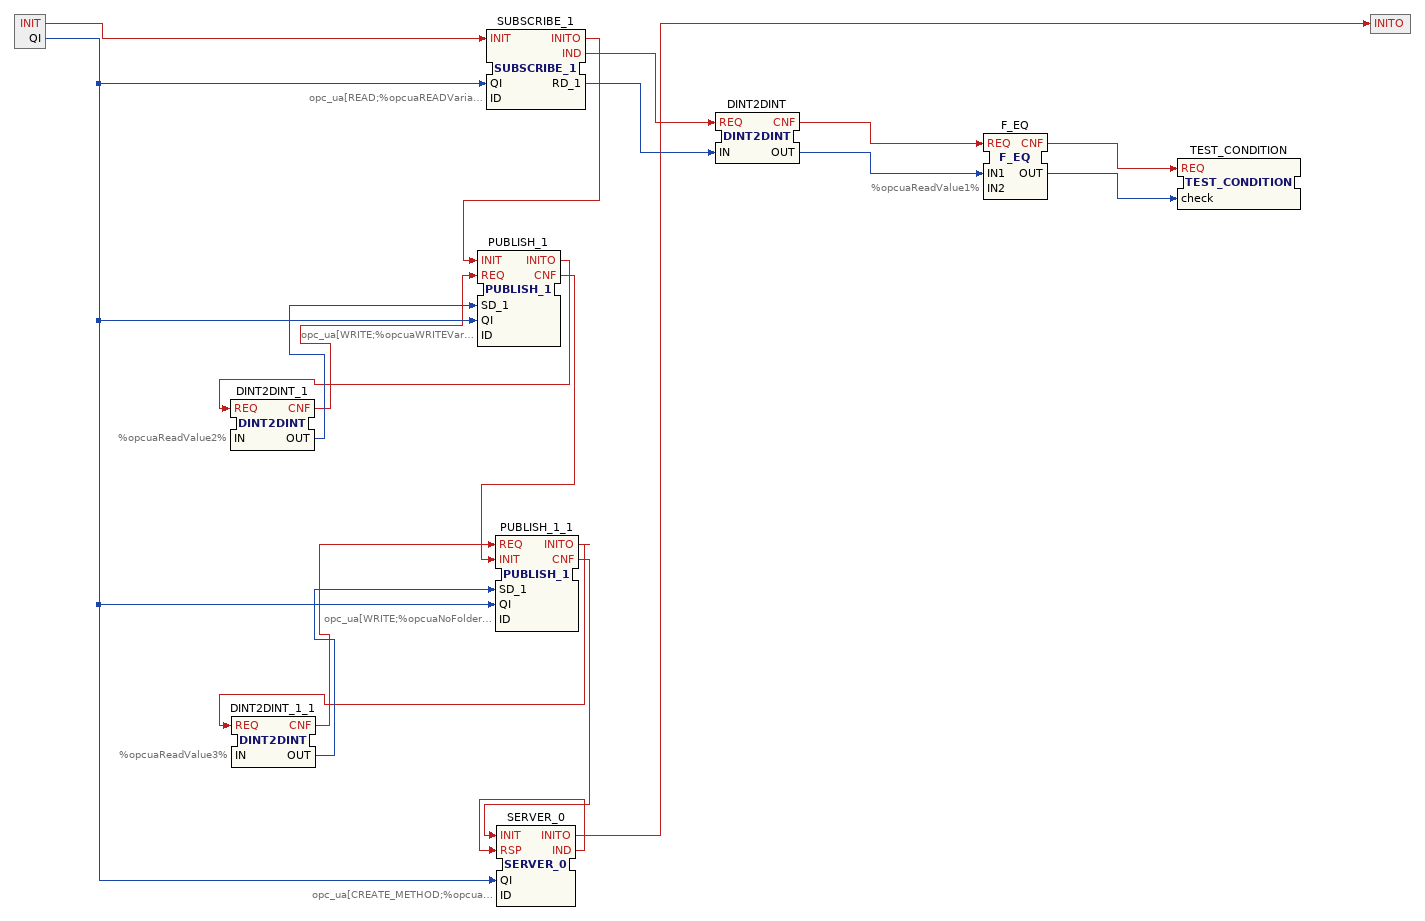
      FBS
        PUBLISH_1 : PUBLISH_1(ID := opc_ua[WRITE;%opcuaWRITEVariable%]);
        F_EQ : F_EQ(IN2 := %opcuaReadValue1%);
        DINT2DINT : DINT2DINT;
        DINT2DINT_1 : DINT2DINT(IN := %opcuaReadValue2%);
        TEST_CONDITION : TEST_CONDITION;
        SUBSCRIBE_1 : SUBSCRIBE_1(ID := opc_ua[READ;%opcuaREADVariable%]);
        DINT2DINT_1_1 : DINT2DINT(IN := %opcuaReadValue3%);
        PUBLISH_1_1 : PUBLISH_1(ID := opc_ua[WRITE;%opcuaNoFolder%]);
        SERVER_0 : SERVER_0(ID := opc_ua[CREATE_METHOD;%opcuaNoFolderMethod%]);
      END_FBS
      EVENT_CONNECTIONS
        SUBSCRIBE_1.INITO TO PUBLISH_1.INIT;
        DINT2DINT_1.CNF TO PUBLISH_1.REQ;
        PUBLISH_1.INITO TO DINT2DINT_1.REQ;
        DINT2DINT.CNF TO F_EQ.REQ;
        F_EQ.CNF TO TEST_CONDITION.REQ;
        SUBSCRIBE_1.IND TO DINT2DINT.REQ;
        INIT TO SUBSCRIBE_1.INIT;
        PUBLISH_1_1.INITO TO DINT2DINT_1_1.REQ;
        DINT2DINT_1_1.CNF TO PUBLISH_1_1.REQ;
        PUBLISH_1.CNF TO PUBLISH_1_1.INIT;
        SERVER_0.INITO TO INITO;
        PUBLISH_1_1.CNF TO SERVER_0.INIT;
        SERVER_0.IND TO SERVER_0.RSP;
      END_CONNECTIONS
      DATA_CONNECTIONS
        DINT2DINT_1.OUT TO PUBLISH_1.SD_1;
        DINT2DINT.OUT TO F_EQ.IN1;
        F_EQ.OUT TO TEST_CONDITION.check;
        SUBSCRIBE_1.RD_1 TO DINT2DINT.IN;
        QI TO SUBSCRIBE_1.QI;
        QI TO PUBLISH_1.QI;
        DINT2DINT_1_1.OUT TO PUBLISH_1_1.SD_1;
        QI TO PUBLISH_1_1.QI;
        QI TO SERVER_0.QI;
      END_CONNECTIONS
    END_SUBAPPLICATION
    SUBAPPLICATION RemoteIsolatedCases
      EVENT_INPUT
        INIT;
        REQ;
      END_EVENT
      EVENT_OUTPUT
        INITO;
        CNF;
      END_EVENT
      VAR_INPUT
        QI : BOOL;
      END_VAR
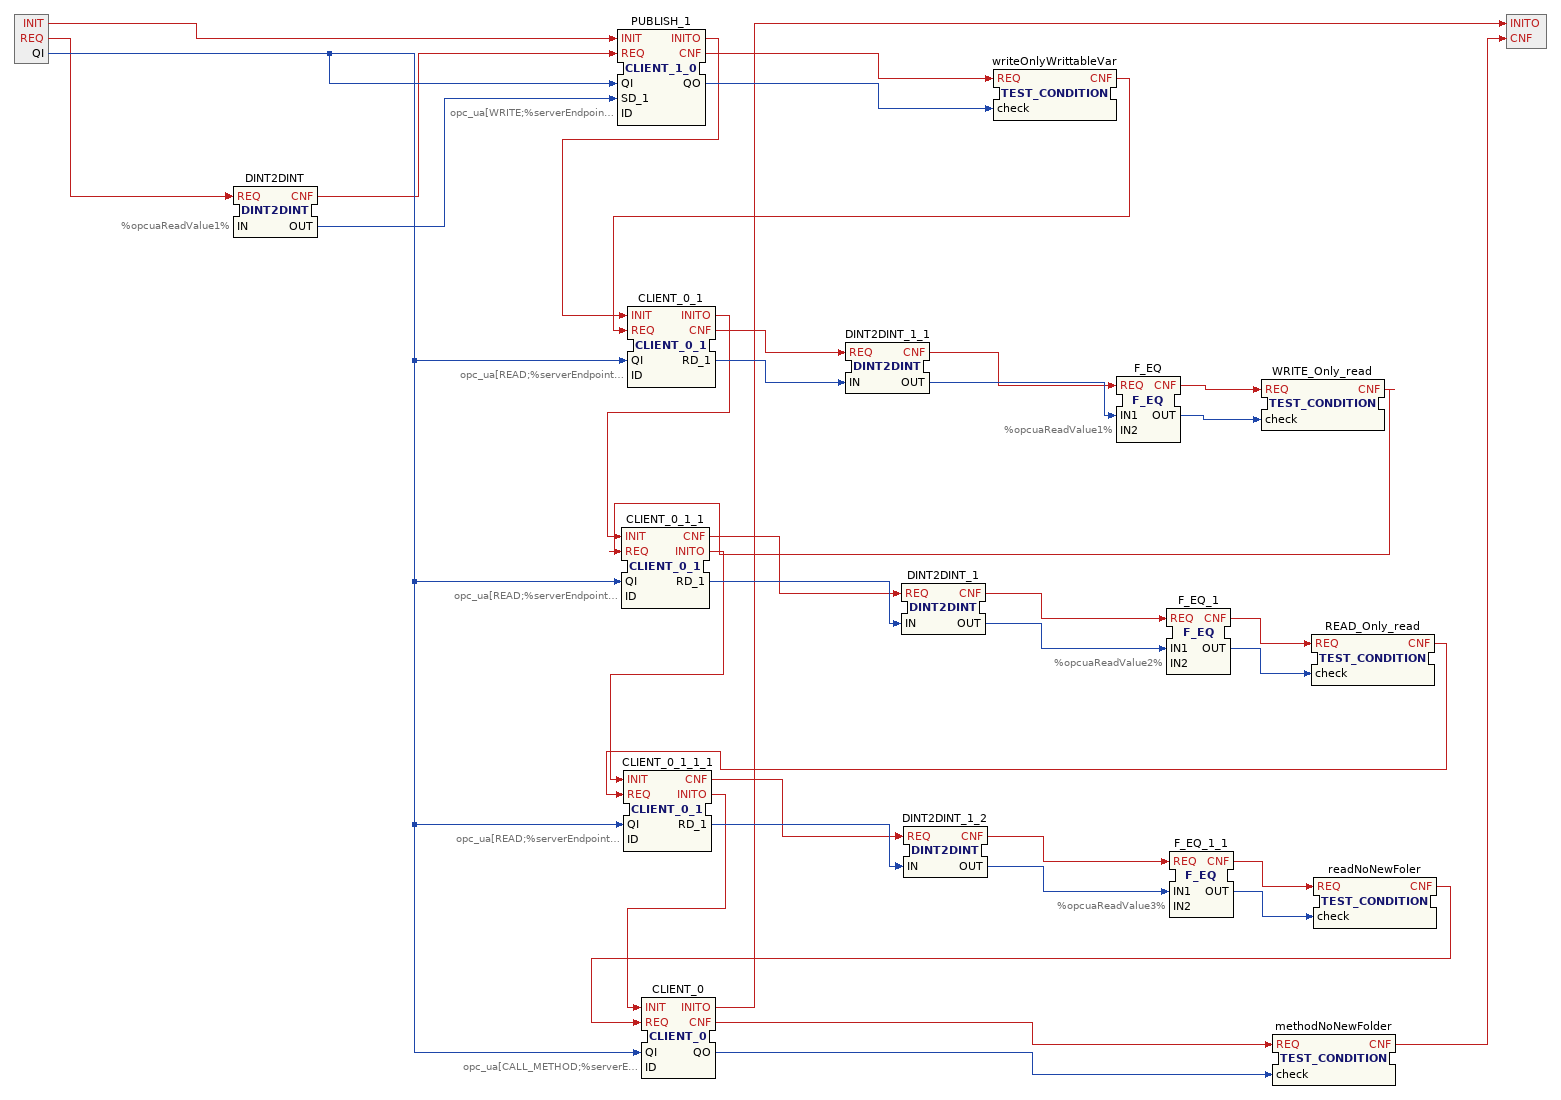
      FBS
        DINT2DINT : DINT2DINT(IN := %opcuaReadValue1%);
        F_EQ_1 : F_EQ(IN2 := %opcuaReadValue2%);
        CLIENT_0_1 : CLIENT_0_1(ID := opc_ua[READ;%serverEndpoint%;%opcuaREADVariable%]);
        WRITE_Only_read : TEST_CONDITION;
        F_EQ : F_EQ(IN2 := %opcuaReadValue1%);
        READ_Only_read : TEST_CONDITION;
        DINT2DINT_1_1 : DINT2DINT;
        DINT2DINT_1 : DINT2DINT;
        CLIENT_0_1_1 : CLIENT_0_1(ID := opc_ua[READ;%serverEndpoint%;%opcuaWRITEVariable%]);
        CLIENT_0_1_1_1 : CLIENT_0_1(ID := opc_ua[READ;%serverEndpoint%;%opcuaNoFolder%]);
        readNoNewFoler : TEST_CONDITION;
        DINT2DINT_1_2 : DINT2DINT;
        F_EQ_1_1 : F_EQ(IN2 := %opcuaReadValue3%);
        CLIENT_0 : CLIENT_0(ID := opc_ua[CALL_METHOD;%serverEndpoint%;%opcuaNoFolderMethod%]);
        methodNoNewFolder : TEST_CONDITION;
        PUBLISH_1 : CLIENT_1_0(ID := opc_ua[WRITE;%serverEndpoint%;%opcuaREADVariable%]);
        writeOnlyWrittableVar : TEST_CONDITION;
      END_FBS
      EVENT_CONNECTIONS
        CLIENT_0_1.INITO TO CLIENT_0_1_1.INIT;
        REQ TO DINT2DINT.REQ;
        CLIENT_0_1.CNF TO DINT2DINT_1_1.REQ;
        DINT2DINT_1_1.CNF TO F_EQ.REQ;
        F_EQ.CNF TO WRITE_Only_read.REQ;
        WRITE_Only_read.CNF TO CLIENT_0_1_1.REQ;
        CLIENT_0_1_1.CNF TO DINT2DINT_1.REQ;
        DINT2DINT_1.CNF TO F_EQ_1.REQ;
        F_EQ_1.CNF TO READ_Only_read.REQ;
        F_EQ_1_1.CNF TO readNoNewFoler.REQ;
        DINT2DINT_1_2.CNF TO F_EQ_1_1.REQ;
        CLIENT_0_1_1_1.CNF TO DINT2DINT_1_2.REQ;
        CLIENT_0_1_1.INITO TO CLIENT_0_1_1_1.INIT;
        READ_Only_read.CNF TO CLIENT_0_1_1_1.REQ;
        CLIENT_0.INITO TO INITO;
        CLIENT_0_1_1_1.INITO TO CLIENT_0.INIT;
        readNoNewFoler.CNF TO CLIENT_0.REQ;
        methodNoNewFolder.CNF TO CNF;
        CLIENT_0.CNF TO methodNoNewFolder.REQ;
        INIT TO PUBLISH_1.INIT;
        DINT2DINT.CNF TO PUBLISH_1.REQ;
        PUBLISH_1.INITO TO CLIENT_0_1.INIT;
        writeOnlyWrittableVar.CNF TO CLIENT_0_1.REQ;
        PUBLISH_1.CNF TO writeOnlyWrittableVar.REQ;
      END_CONNECTIONS
      DATA_CONNECTIONS
        QI TO CLIENT_0_1.QI;
        QI TO CLIENT_0_1_1.QI;
        CLIENT_0_1.RD_1 TO DINT2DINT_1_1.IN;
        CLIENT_0_1_1.RD_1 TO DINT2DINT_1.IN;
        DINT2DINT_1.OUT TO F_EQ_1.IN1;
        F_EQ_1.OUT TO READ_Only_read.check;
        DINT2DINT_1_1.OUT TO F_EQ.IN1;
        F_EQ.OUT TO WRITE_Only_read.check;
        F_EQ_1_1.OUT TO readNoNewFoler.check;
        CLIENT_0_1_1_1.RD_1 TO DINT2DINT_1_2.IN;
        DINT2DINT_1_2.OUT TO F_EQ_1_1.IN1;
        QI TO CLIENT_0_1_1_1.QI;
        QI TO CLIENT_0.QI;
        CLIENT_0.QO TO methodNoNewFolder.check;
        QI TO PUBLISH_1.QI;
        DINT2DINT.OUT TO PUBLISH_1.SD_1;
        PUBLISH_1.QO TO writeOnlyWrittableVar.check;
      END_CONNECTIONS
    END_SUBAPPLICATION
    SUBAPPLICATION WorkingWithoutSubscription
      EVENT_INPUT
        INIT;
      END_EVENT
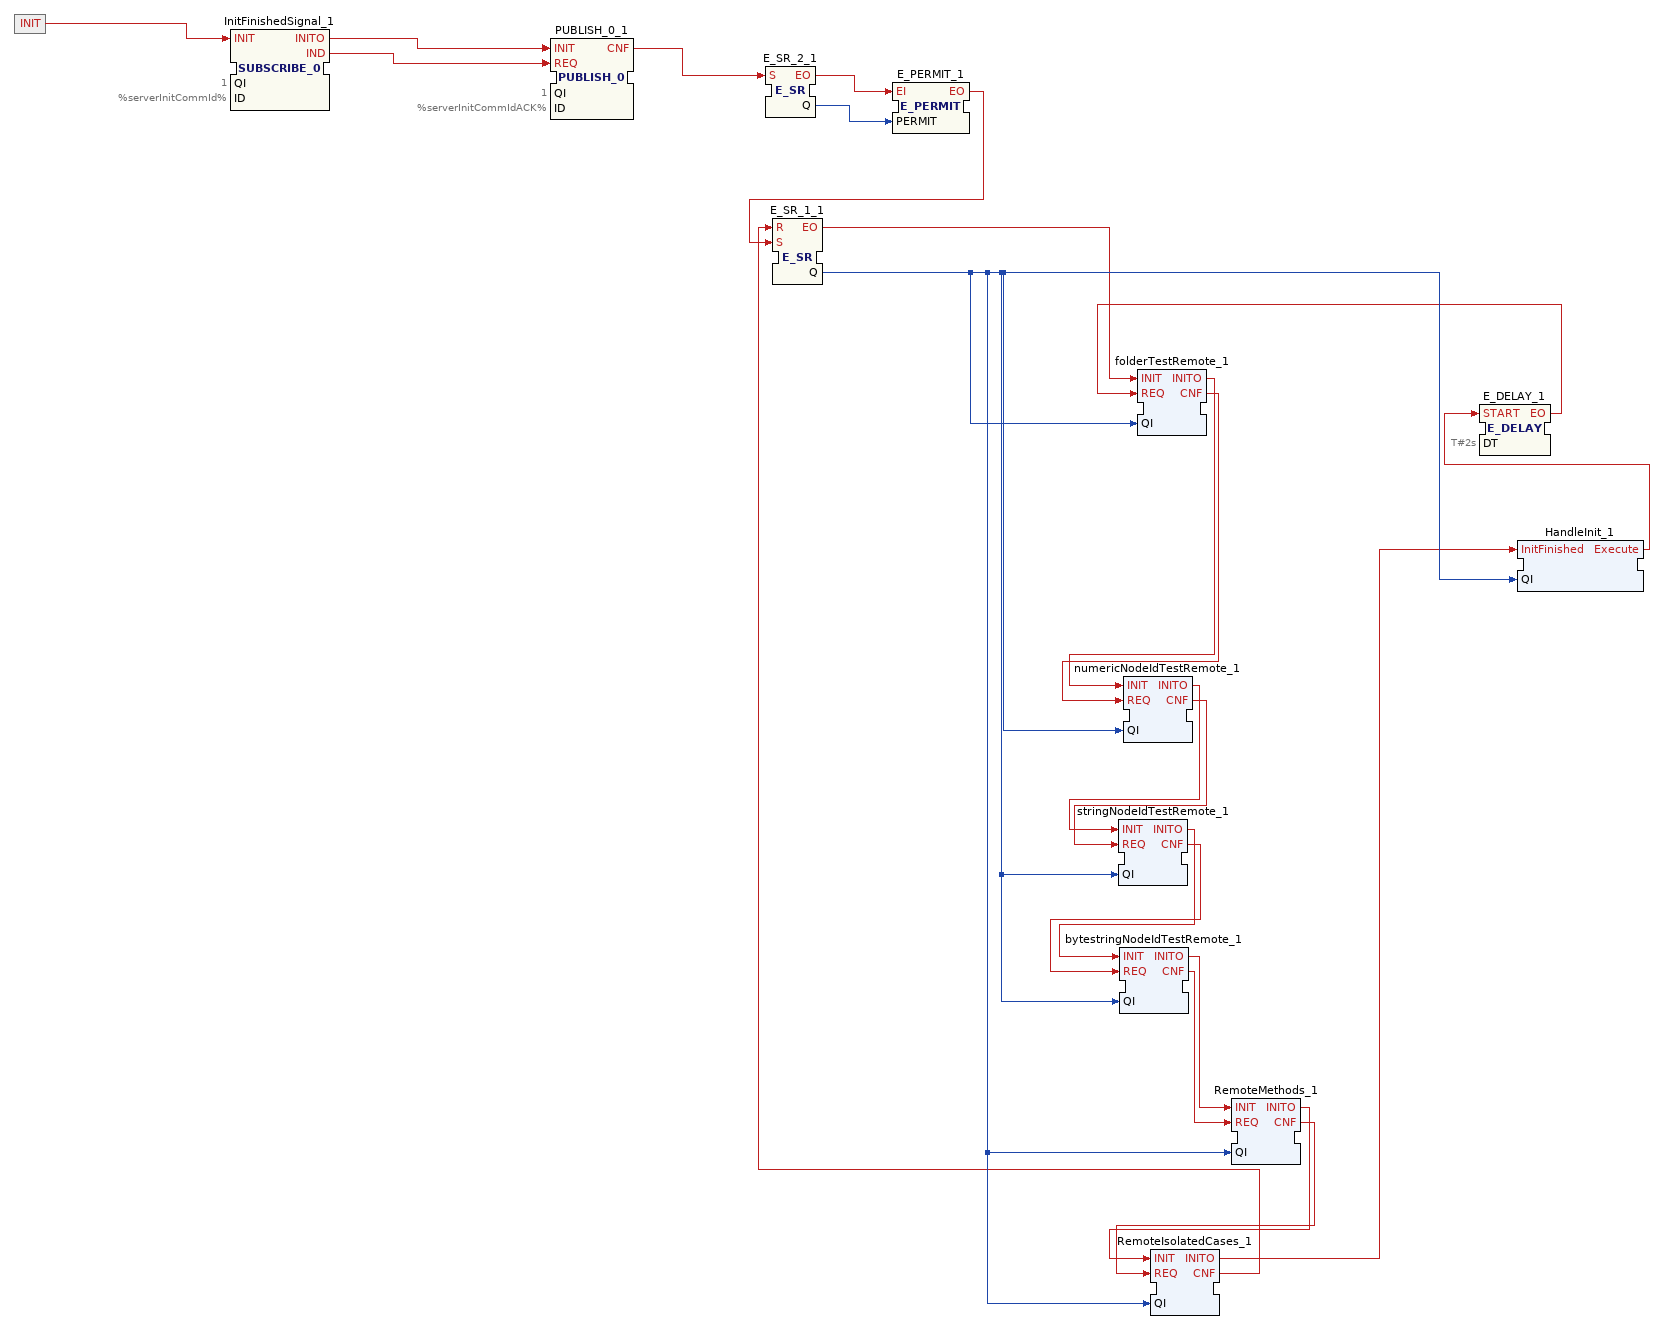
      FBS
        InitFinishedSignal_1 : SUBSCRIBE_0(QI := 1, ID := %serverInitCommId%);
        E_PERMIT_1 : E_PERMIT;
        E_DELAY_1 : E_DELAY(DT := T#2s);
        PUBLISH_0_1 : PUBLISH_0(QI := 1, ID := %serverInitCommIdACK%);
        E_SR_2_1 : E_SR;
        E_SR_1_1 : E_SR;
      END_FBS
      SUBAPPLICATION RemoteIsolatedCases_1
        EVENT_INPUT
          INIT;
          REQ;
        END_EVENT
        EVENT_OUTPUT
          INITO;
          CNF;
        END_EVENT
        VAR_INPUT
          QI : BOOL;
        END_VAR
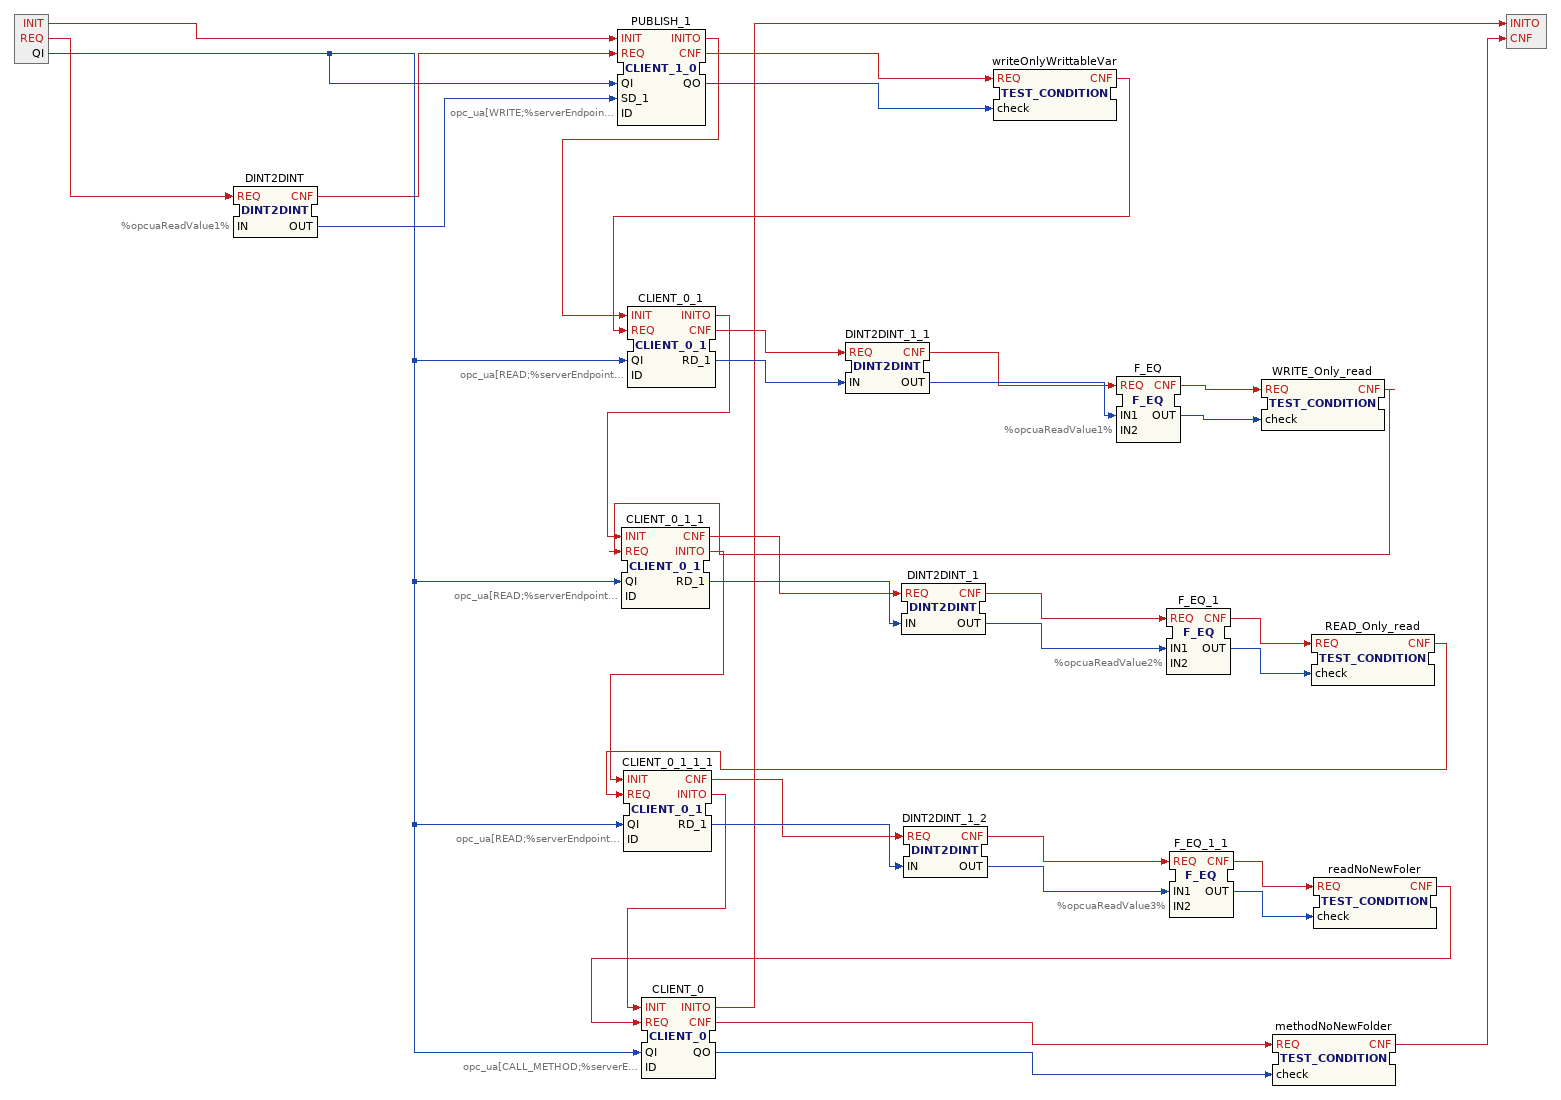
        FBS
          DINT2DINT : DINT2DINT(IN := %opcuaReadValue1%);
          F_EQ_1 : F_EQ(IN2 := %opcuaReadValue2%);
          CLIENT_0_1 : CLIENT_0_1(ID := opc_ua[READ;%serverEndpoint%;%opcuaREADVariable%]);
          WRITE_Only_read : TEST_CONDITION;
          F_EQ : F_EQ(IN2 := %opcuaReadValue1%);
          READ_Only_read : TEST_CONDITION;
          DINT2DINT_1_1 : DINT2DINT;
          DINT2DINT_1 : DINT2DINT;
          CLIENT_0_1_1 : CLIENT_0_1(ID := opc_ua[READ;%serverEndpoint%;%opcuaWRITEVariable%]);
          CLIENT_0_1_1_1 : CLIENT_0_1(ID := opc_ua[READ;%serverEndpoint%;%opcuaNoFolder%]);
          readNoNewFoler : TEST_CONDITION;
          DINT2DINT_1_2 : DINT2DINT;
          F_EQ_1_1 : F_EQ(IN2 := %opcuaReadValue3%);
          CLIENT_0 : CLIENT_0(ID := opc_ua[CALL_METHOD;%serverEndpoint%;%opcuaNoFolderMethod%]);
          methodNoNewFolder : TEST_CONDITION;
          PUBLISH_1 : CLIENT_1_0(ID := opc_ua[WRITE;%serverEndpoint%;%opcuaREADVariable%]);
          writeOnlyWrittableVar : TEST_CONDITION;
        END_FBS
        EVENT_CONNECTIONS
          CLIENT_0_1.INITO TO CLIENT_0_1_1.INIT;
          REQ TO DINT2DINT.REQ;
          CLIENT_0_1.CNF TO DINT2DINT_1_1.REQ;
          DINT2DINT_1_1.CNF TO F_EQ.REQ;
          F_EQ.CNF TO WRITE_Only_read.REQ;
          WRITE_Only_read.CNF TO CLIENT_0_1_1.REQ;
          CLIENT_0_1_1.CNF TO DINT2DINT_1.REQ;
          DINT2DINT_1.CNF TO F_EQ_1.REQ;
          F_EQ_1.CNF TO READ_Only_read.REQ;
          F_EQ_1_1.CNF TO readNoNewFoler.REQ;
          DINT2DINT_1_2.CNF TO F_EQ_1_1.REQ;
          CLIENT_0_1_1_1.CNF TO DINT2DINT_1_2.REQ;
          CLIENT_0_1_1.INITO TO CLIENT_0_1_1_1.INIT;
          READ_Only_read.CNF TO CLIENT_0_1_1_1.REQ;
          CLIENT_0.INITO TO INITO;
          CLIENT_0_1_1_1.INITO TO CLIENT_0.INIT;
          readNoNewFoler.CNF TO CLIENT_0.REQ;
          methodNoNewFolder.CNF TO CNF;
          CLIENT_0.CNF TO methodNoNewFolder.REQ;
          INIT TO PUBLISH_1.INIT;
          DINT2DINT.CNF TO PUBLISH_1.REQ;
          PUBLISH_1.INITO TO CLIENT_0_1.INIT;
          writeOnlyWrittableVar.CNF TO CLIENT_0_1.REQ;
          PUBLISH_1.CNF TO writeOnlyWrittableVar.REQ;
        END_CONNECTIONS
        DATA_CONNECTIONS
          QI TO CLIENT_0_1.QI;
          QI TO CLIENT_0_1_1.QI;
          CLIENT_0_1.RD_1 TO DINT2DINT_1_1.IN;
          CLIENT_0_1_1.RD_1 TO DINT2DINT_1.IN;
          DINT2DINT_1.OUT TO F_EQ_1.IN1;
          F_EQ_1.OUT TO READ_Only_read.check;
          DINT2DINT_1_1.OUT TO F_EQ.IN1;
          F_EQ.OUT TO WRITE_Only_read.check;
          F_EQ_1_1.OUT TO readNoNewFoler.check;
          CLIENT_0_1_1_1.RD_1 TO DINT2DINT_1_2.IN;
          DINT2DINT_1_2.OUT TO F_EQ_1_1.IN1;
          QI TO CLIENT_0_1_1_1.QI;
          QI TO CLIENT_0.QI;
          CLIENT_0.QO TO methodNoNewFolder.check;
          QI TO PUBLISH_1.QI;
          DINT2DINT.OUT TO PUBLISH_1.SD_1;
          PUBLISH_1.QO TO writeOnlyWrittableVar.check;
        END_CONNECTIONS
      END_SUBAPPLICATION
      SUBAPPLICATION numericNodeIdTestRemote_1
        EVENT_INPUT
          INIT;
          REQ;
        END_EVENT
        EVENT_OUTPUT
          INITO;
          CNF;
        END_EVENT
        VAR_INPUT
          QI : BOOL;
        END_VAR
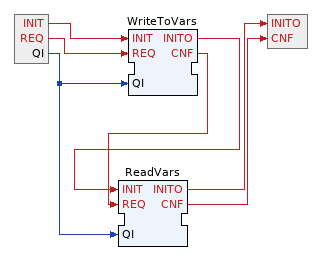
        SUBAPPLICATION WriteToVars
          EVENT_INPUT
            INIT;
            REQ;
          END_EVENT
          EVENT_OUTPUT
            INITO;
            CNF;
          END_EVENT
          VAR_INPUT
            QI : BOOL;
          END_VAR
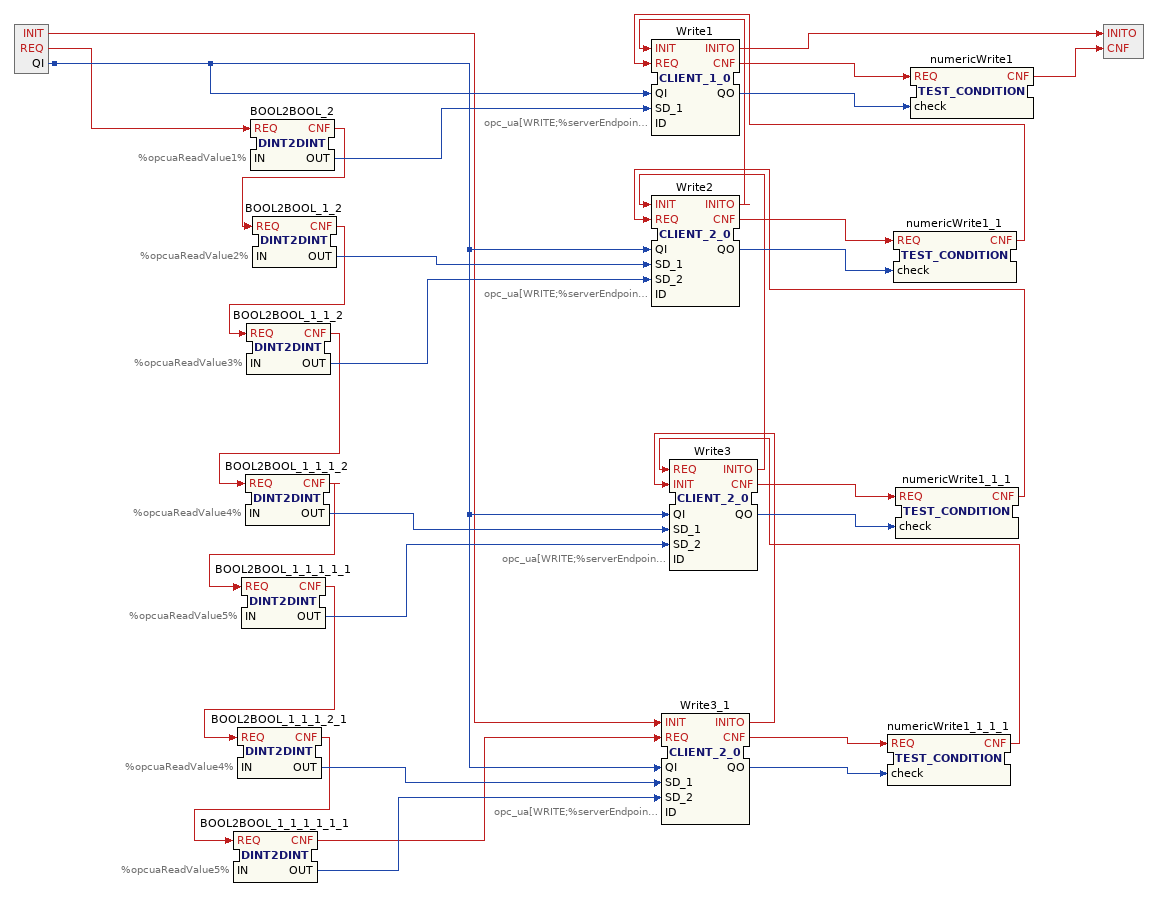
          FBS
            BOOL2BOOL_1_1_2 : DINT2DINT(IN := %opcuaReadValue3%);
            BOOL2BOOL_1_1_1_1_1 : DINT2DINT(IN := %opcuaReadValue5%);
            BOOL2BOOL_1_1_1_2 : DINT2DINT(IN := %opcuaReadValue4%);
            BOOL2BOOL_2 : DINT2DINT(IN := %opcuaReadValue1%);
            BOOL2BOOL_1_2 : DINT2DINT(IN := %opcuaReadValue2%);
            BOOL2BOOL_1_1_1_2_1 : DINT2DINT(IN := %opcuaReadValue4%);
            BOOL2BOOL_1_1_1_1_1_1 : DINT2DINT(IN := %opcuaReadValue5%);
            Write1 : CLIENT_1_0(ID := opc_ua[WRITE;%serverEndpoint%;%opcuaFolderTestWithNodeIdNumeric1%]);
            Write3 : CLIENT_2_0(ID := opc_ua[WRITE;%serverEndpoint%;%opcuaFolderTestWithNodeIdNumeric3%]);
            Write2 : CLIENT_2_0(ID := opc_ua[WRITE;%serverEndpoint%;%opcuaFolderTestWithNodeIdNumeric2%]);
            numericWrite1 : TEST_CONDITION;
            numericWrite1_1 : TEST_CONDITION;
            numericWrite1_1_1 : TEST_CONDITION;
            numericWrite1_1_1_1 : TEST_CONDITION;
            Write3_1 : CLIENT_2_0(ID := opc_ua[WRITE;%serverEndpoint%;,1:i=12348;,1:i=12349]);
          END_FBS
          EVENT_CONNECTIONS
            BOOL2BOOL_1_2.CNF TO BOOL2BOOL_1_1_2.REQ;
            BOOL2BOOL_1_1_2.CNF TO BOOL2BOOL_1_1_1_2.REQ;
            BOOL2BOOL_1_1_1_2.CNF TO BOOL2BOOL_1_1_1_1_1.REQ;
            BOOL2BOOL_2.CNF TO BOOL2BOOL_1_2.REQ;
            REQ TO BOOL2BOOL_2.REQ;
            BOOL2BOOL_1_1_1_2_1.CNF TO BOOL2BOOL_1_1_1_1_1_1.REQ;
            BOOL2BOOL_1_1_1_1_1.CNF TO BOOL2BOOL_1_1_1_2_1.REQ;
            Write1.INITO TO INITO;
            Write3.INITO TO Write2.INIT;
            Write2.INITO TO Write1.INIT;
            numericWrite1_1.CNF TO Write1.REQ;
            numericWrite1.CNF TO CNF;
            Write1.CNF TO numericWrite1.REQ;
            numericWrite1_1_1.CNF TO Write2.REQ;
            Write3.CNF TO numericWrite1_1_1.REQ;
            numericWrite1_1_1_1.CNF TO Write3.REQ;
            INIT TO Write3_1.INIT;
            BOOL2BOOL_1_1_1_1_1_1.CNF TO Write3_1.REQ;
            Write3_1.INITO TO Write3.INIT;
            Write3_1.CNF TO numericWrite1_1_1_1.REQ;
            Write2.CNF TO numericWrite1_1.REQ;
          END_CONNECTIONS
          DATA_CONNECTIONS
            QI TO Write1.QI;
            BOOL2BOOL_2.OUT TO Write1.SD_1;
            QI TO Write3.QI;
            BOOL2BOOL_1_1_1_2.OUT TO Write3.SD_1;
            BOOL2BOOL_1_1_1_1_1.OUT TO Write3.SD_2;
            QI TO Write2.QI;
            BOOL2BOOL_1_2.OUT TO Write2.SD_1;
            BOOL2BOOL_1_1_2.OUT TO Write2.SD_2;
            Write3.QO TO numericWrite1_1_1.check;
            Write1.QO TO numericWrite1.check;
            Write2.QO TO numericWrite1_1.check;
            QI TO Write3_1.QI;
            BOOL2BOOL_1_1_1_2_1.OUT TO Write3_1.SD_1;
            BOOL2BOOL_1_1_1_1_1_1.OUT TO Write3_1.SD_2;
            Write3_1.QO TO numericWrite1_1_1_1.check;
          END_CONNECTIONS
        END_SUBAPPLICATION
        SUBAPPLICATION ReadVars
          EVENT_INPUT
            INIT;
            REQ;
          END_EVENT
          EVENT_OUTPUT
            INITO;
            CNF;
          END_EVENT
          VAR_INPUT
            QI : BOOL;
          END_VAR
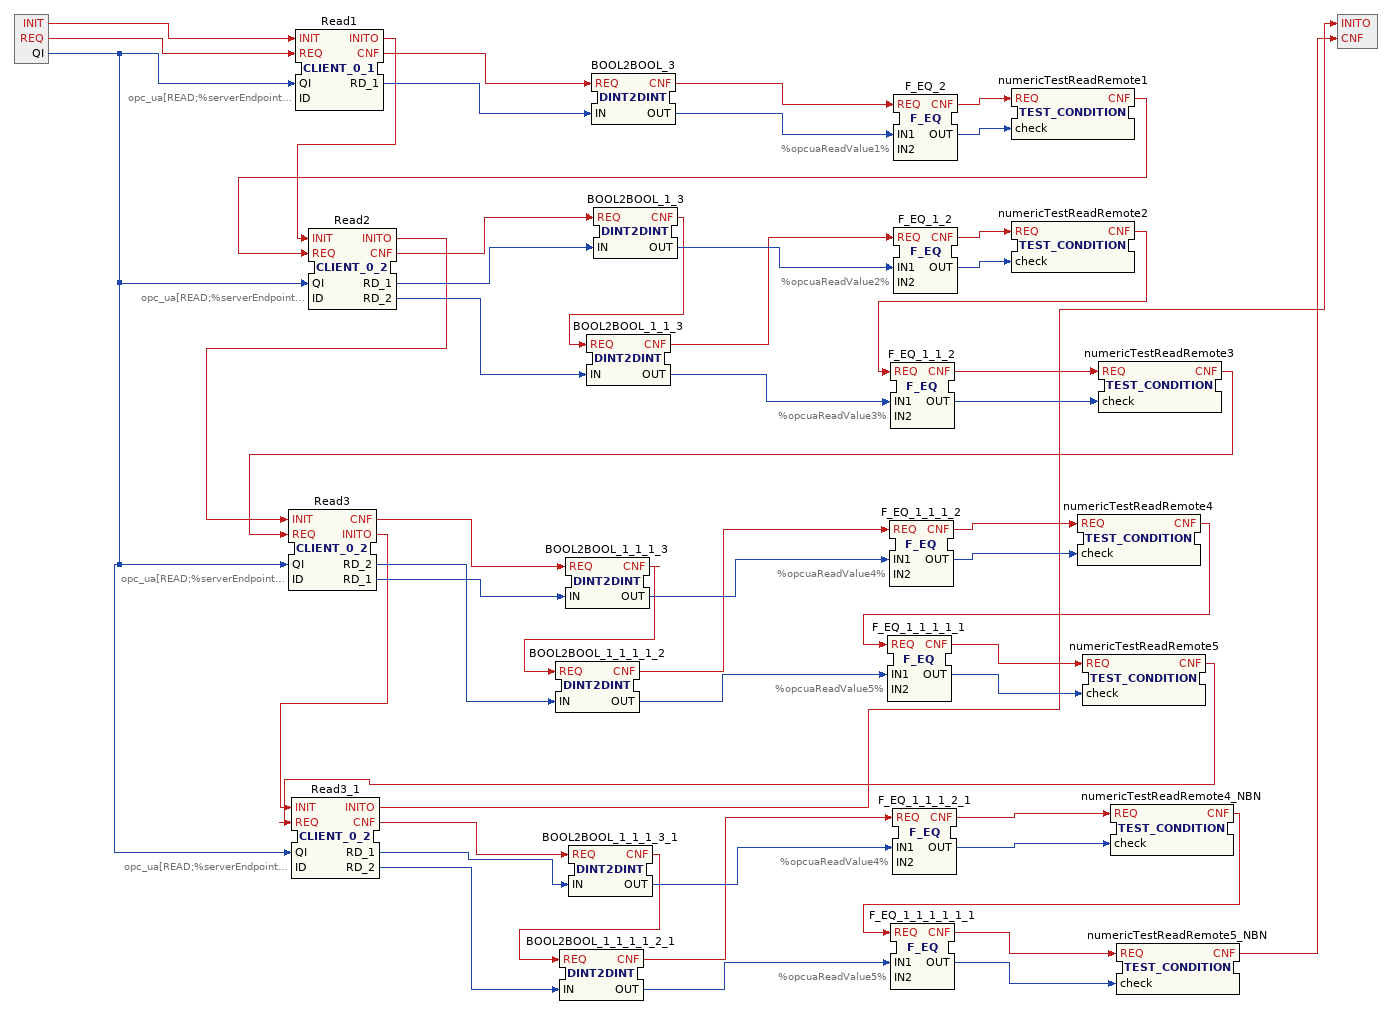
          FBS
            Read1 : CLIENT_0_1(ID := opc_ua[READ;%serverEndpoint%;%opcuaFolderTestWithNodeIdNumeric1%]);
            Read2 : CLIENT_0_2(ID := opc_ua[READ;%serverEndpoint%;%opcuaFolderTestWithNodeIdNumeric2%]);
            F_EQ_1_1_1_2 : F_EQ(IN2 := %opcuaReadValue4%);
            numericTestReadRemote4 : TEST_CONDITION;
            BOOL2BOOL_1_3 : DINT2DINT;
            F_EQ_1_1_1_1_1 : F_EQ(IN2 := %opcuaReadValue5%);
            numericTestReadRemote3 : TEST_CONDITION;
            BOOL2BOOL_1_1_3 : DINT2DINT;
            BOOL2BOOL_1_1_1_1_2 : DINT2DINT;
            BOOL2BOOL_1_1_1_3 : DINT2DINT;
            numericTestReadRemote2 : TEST_CONDITION;
            F_EQ_1_1_2 : F_EQ(IN2 := %opcuaReadValue3%);
            F_EQ_2 : F_EQ(IN2 := %opcuaReadValue1%);
            F_EQ_1_2 : F_EQ(IN2 := %opcuaReadValue2%);
            Read3 : CLIENT_0_2(ID := opc_ua[READ;%serverEndpoint%;%opcuaFolderTestWithNodeIdNumeric3%]);
            numericTestReadRemote5 : TEST_CONDITION;
            numericTestReadRemote1 : TEST_CONDITION;
            BOOL2BOOL_3 : DINT2DINT;
            F_EQ_1_1_1_2_1 : F_EQ(IN2 := %opcuaReadValue4%);
            Read3_1 : CLIENT_0_2(ID := opc_ua[READ;%serverEndpoint%;,1:i=12348;,1:i=12349]);
            F_EQ_1_1_1_1_1_1 : F_EQ(IN2 := %opcuaReadValue5%);
            BOOL2BOOL_1_1_1_1_2_1 : DINT2DINT;
            BOOL2BOOL_1_1_1_3_1 : DINT2DINT;
            numericTestReadRemote4_NBN : TEST_CONDITION;
            numericTestReadRemote5_NBN : TEST_CONDITION;
          END_FBS
          EVENT_CONNECTIONS
            Read1.INITO TO Read2.INIT;
            numericTestReadRemote1.CNF TO Read2.REQ;
            Read2.INITO TO Read3.INIT;
            Read2.CNF TO BOOL2BOOL_1_3.REQ;
            BOOL2BOOL_1_1_1_1_2.CNF TO F_EQ_1_1_1_2.REQ;
            F_EQ_1_1_1_2.CNF TO numericTestReadRemote4.REQ;
            numericTestReadRemote4.CNF TO F_EQ_1_1_1_1_1.REQ;
            BOOL2BOOL_1_3.CNF TO BOOL2BOOL_1_1_3.REQ;
            F_EQ_1_1_1_1_1.CNF TO numericTestReadRemote5.REQ;
            F_EQ_1_1_2.CNF TO numericTestReadRemote3.REQ;
            numericTestReadRemote3.CNF TO Read3.REQ;
            BOOL2BOOL_1_1_3.CNF TO F_EQ_1_2.REQ;
            BOOL2BOOL_1_1_1_3.CNF TO BOOL2BOOL_1_1_1_1_2.REQ;
            Read3.CNF TO BOOL2BOOL_1_1_1_3.REQ;
            F_EQ_1_2.CNF TO numericTestReadRemote2.REQ;
            INIT TO Read1.INIT;
            REQ TO Read1.REQ;
            Read1.CNF TO BOOL2BOOL_3.REQ;
            BOOL2BOOL_3.CNF TO F_EQ_2.REQ;
            F_EQ_2.CNF TO numericTestReadRemote1.REQ;
            numericTestReadRemote2.CNF TO F_EQ_1_1_2.REQ;
            Read3_1.INITO TO INITO;
            Read3.INITO TO Read3_1.INIT;
            Read3_1.CNF TO BOOL2BOOL_1_1_1_3_1.REQ;
            BOOL2BOOL_1_1_1_3_1.CNF TO BOOL2BOOL_1_1_1_1_2_1.REQ;
            BOOL2BOOL_1_1_1_1_2_1.CNF TO F_EQ_1_1_1_2_1.REQ;
            F_EQ_1_1_1_2_1.CNF TO numericTestReadRemote4_NBN.REQ;
            F_EQ_1_1_1_1_1_1.CNF TO numericTestReadRemote5_NBN.REQ;
            numericTestReadRemote4_NBN.CNF TO F_EQ_1_1_1_1_1_1.REQ;
            numericTestReadRemote5_NBN.CNF TO CNF;
            numericTestReadRemote5.CNF TO Read3_1.REQ;
          END_CONNECTIONS
          DATA_CONNECTIONS
            Read1.RD_1 TO BOOL2BOOL_3.IN;
            Read2.RD_1 TO BOOL2BOOL_1_3.IN;
            Read2.RD_2 TO BOOL2BOOL_1_1_3.IN;
            BOOL2BOOL_1_1_1_3.OUT TO F_EQ_1_1_1_2.IN1;
            F_EQ_1_1_1_2.OUT TO numericTestReadRemote4.check;
            BOOL2BOOL_1_3.OUT TO F_EQ_1_2.IN1;
            BOOL2BOOL_1_1_1_1_2.OUT TO F_EQ_1_1_1_1_1.IN1;
            F_EQ_1_1_1_1_1.OUT TO numericTestReadRemote5.check;
            F_EQ_1_1_2.OUT TO numericTestReadRemote3.check;
            BOOL2BOOL_1_1_3.OUT TO F_EQ_1_1_2.IN1;
            Read3.RD_2 TO BOOL2BOOL_1_1_1_1_2.IN;
            Read3.RD_1 TO BOOL2BOOL_1_1_1_3.IN;
            F_EQ_1_2.OUT TO numericTestReadRemote2.check;
            BOOL2BOOL_3.OUT TO F_EQ_2.IN1;
            F_EQ_2.OUT TO numericTestReadRemote1.check;
            QI TO Read1.QI;
            QI TO Read2.QI;
            QI TO Read3.QI;
            Read3_1.RD_1 TO BOOL2BOOL_1_1_1_3_1.IN;
            Read3_1.RD_2 TO BOOL2BOOL_1_1_1_1_2_1.IN;
            BOOL2BOOL_1_1_1_1_2_1.OUT TO F_EQ_1_1_1_1_1_1.IN1;
            BOOL2BOOL_1_1_1_3_1.OUT TO F_EQ_1_1_1_2_1.IN1;
            F_EQ_1_1_1_2_1.OUT TO numericTestReadRemote4_NBN.check;
            F_EQ_1_1_1_1_1_1.OUT TO numericTestReadRemote5_NBN.check;
            QI TO Read3_1.QI;
          END_CONNECTIONS
        END_SUBAPPLICATION
        EVENT_CONNECTIONS
          WriteToVars.INITO TO ReadVars.INIT;
          INIT TO WriteToVars.INIT;
          REQ TO WriteToVars.REQ;
          ReadVars.CNF TO CNF;
          WriteToVars.CNF TO ReadVars.REQ;
          ReadVars.INITO TO INITO;
        END_CONNECTIONS
        DATA_CONNECTIONS
          QI TO ReadVars.QI;
          QI TO WriteToVars.QI;
        END_CONNECTIONS
      END_SUBAPPLICATION
      SUBAPPLICATION folderTestRemote_1
        EVENT_INPUT
          INIT;
          REQ;
        END_EVENT
        EVENT_OUTPUT
          INITO;
          CNF;
        END_EVENT
        VAR_INPUT
          QI : BOOL;
        END_VAR
